REGION Network 90: VARIABLES AUXILIARES - Fin de Reset
   RUNG wire#powerrail
      Contact( #Mx_ET09 )
      wire#w1
      Coil( #EstadoVI.Fin_Reset )
   END_RUNG
   RUNG wire#powerrail
      Contact( #Mx_ET00 )
      Contact( #EstadoZona.PerReset_CBx )
      I_Contact( #pHsMx_1 )
      I_Contact( #pHsMx_2 )
      I_Contact( #pHsMx_3 )
      I_Contact( #pHsMx_4 )
   END_RUNG wire#w1
   // the same network as SCL:
   #EstadoVI.Fin_Reset := #Mx_ET09 OR (#Mx_ET00 AND #EstadoZona.PerReset_CBx AND NOT #pHsMx_1 AND NOT #pHsMx_2 AND NOT #pHsMx_3 AND NOT #pHsMx_4);
END_REGION

REGION Network 91: VARIABLES AUXILIARES - Fin de Paro Blando
   RUNG wire#powerrail
      I_Contact( #Avance_TR1 )
      I_Contact( #Avance_TR2 )
      I_Contact( #Avance_T1 )
      I_Contact( #Avance_T2 )
      I_Contact( #Avance_T3 )
      I_Contact( #Avance_T4 )
      Contact( #EstadoZona.ParoBlando_CBx )
      Coil( #EstadoVI.Fin_Paro_Blando )
   END_RUNG
   // the same network as SCL:
   #EstadoVI.Fin_Paro_Blando := NOT #Avance_TR1 AND NOT #Avance_TR2 AND NOT #Avance_T1 AND NOT #Avance_T2 AND NOT #Avance_T3 AND NOT #Avance_T4 AND #EstadoZona.ParoBlando_CBx;
END_REGION

REGION Network 92: VARIABLES AUXILIARES - Permiso de Entrada - PTF_MAnt_Mx
   RUNG wire#powerrail
      Contact( #Mx_ET20 )
      wire#w1
      Contact( #Avance_TR1 )
      Contact( #Pos_TROK )
      Contact( #Pos_TPOK )
      Contact( #EstadoZona.Marcha_CBx )
      I_Contact( #EstadoVI.Error_Mx )
      I_Contact( #Error_Tx )
      Coil( #PTF_MAnt_Mx )
   END_RUNG
   RUNG wire#powerrail
      Contact( #Mx_ET60 )
      wire#w2
      Contact( #Simultaneo_Mx )
   END_RUNG wire#w1
   RUNG wire#powerrail
      Contact( #Mx_ET61 )
   END_RUNG wire#w2
   // the same network as SCL:
   #PTF_MAnt_Mx := (#Mx_ET20 OR ((#Mx_ET60 OR #Mx_ET61) AND #Simultaneo_Mx)) AND #Avance_TR1 AND #Pos_TROK AND #Pos_TPOK AND #EstadoZona.Marcha_CBx AND NOT #EstadoVI.Error_Mx AND NOT #Error_Tx;
END_REGION

REGION Network 93: INTERLOCK FSS - Permiso de DesCarga E1 - MA_DepositOK_E1
   RUNG wire#powerrail
      Contact( #Mx_ET10 )
      wire#w1
      Contact( #Avance_T1 )
      wire#w2
      Contact( #Pos_TROK )
      Contact( #Pos_TPOK )
      Contact( #EstadoZona.Marcha_CBx )
      I_Contact( #EstadoVI.Error_Mx )
      I_Contact( #Error_Tx )
      Coil( #MA_DepositOK_E1 )
   END_RUNG
   RUNG wire#w1
      Contact( #CNT_pHsMx_E1.QD )
   END_RUNG wire#w2
   RUNG wire#powerrail
      Contact( #Mx_ET11 )
   END_RUNG wire#w2
   RUNG wire#powerrail
      Contact( #Mx_ET01 )
      I_Contact( #Selec_E3 )
      I_Contact( #pHsMx_1 )
      I_Contact( #pHsMx_2 )
      I_Contact( #pHsMx_3 )
      I_Contact( #pHsMx_4 )
      Contact( #ConfigFB.NoEntrar_E1 )
   END_RUNG wire#w2
   // the same network as SCL:
   #MA_DepositOK_E1 := ((#Mx_ET10 AND (#Avance_T1 OR #CNT_pHsMx_E1.QD)) OR #Mx_ET11 OR (#Mx_ET01 AND NOT #Selec_E3 AND NOT #pHsMx_1 AND NOT #pHsMx_2 AND NOT #pHsMx_3 AND NOT #pHsMx_4 AND #ConfigFB.NoEntrar_E1)) AND #Pos_TROK AND #Pos_TPOK AND #EstadoZona.Marcha_CBx AND NOT #EstadoVI.Error_Mx AND NOT #Error_Tx;
END_REGION

REGION Network 94: INTERLOCK FSS - Permiso de DesCarga E1 - MA_DepositOK_E3
   RUNG wire#powerrail
      Contact( #Mx_ET30 )
      wire#w1
      Contact( #Avance_T1 )
      wire#w2
      Contact( #Pos_TROK )
      Contact( #Pos_TPOK )
      Contact( #EstadoZona.Marcha_CBx )
      I_Contact( #EstadoVI.Error_Mx )
      I_Contact( #Error_Tx )
      Coil( #MA_DepositOK_E3 )
   END_RUNG
   RUNG wire#w1
      Contact( #CNT_pHsMx_E3.QD )
   END_RUNG wire#w2
   RUNG wire#powerrail
      Contact( #Mx_ET31 )
   END_RUNG wire#w2
   RUNG wire#powerrail
      Contact( #Mx_ET01 )
      I_Contact( #Selec_E1 )
      I_Contact( #pHsMx_1 )
      I_Contact( #pHsMx_2 )
      I_Contact( #pHsMx_3 )
      I_Contact( #pHsMx_4 )
      Contact( #ConfigFB.NoEntrar_E3 )
   END_RUNG wire#w2
   // the same network as SCL:
   #MA_DepositOK_E3 := ((#Mx_ET30 AND (#Avance_T1 OR #CNT_pHsMx_E3.QD)) OR #Mx_ET31 OR (#Mx_ET01 AND NOT #Selec_E1 AND NOT #pHsMx_1 AND NOT #pHsMx_2 AND NOT #pHsMx_3 AND NOT #pHsMx_4 AND #ConfigFB.NoEntrar_E3)) AND #Pos_TROK AND #Pos_TPOK AND #EstadoZona.Marcha_CBx AND NOT #EstadoVI.Error_Mx AND NOT #Error_Tx;
END_REGION

REGION Network 95: VARIABLES AUXILIARES - Aviso de Salida - AVTF_Mx_MSig - Grande y Pequeña
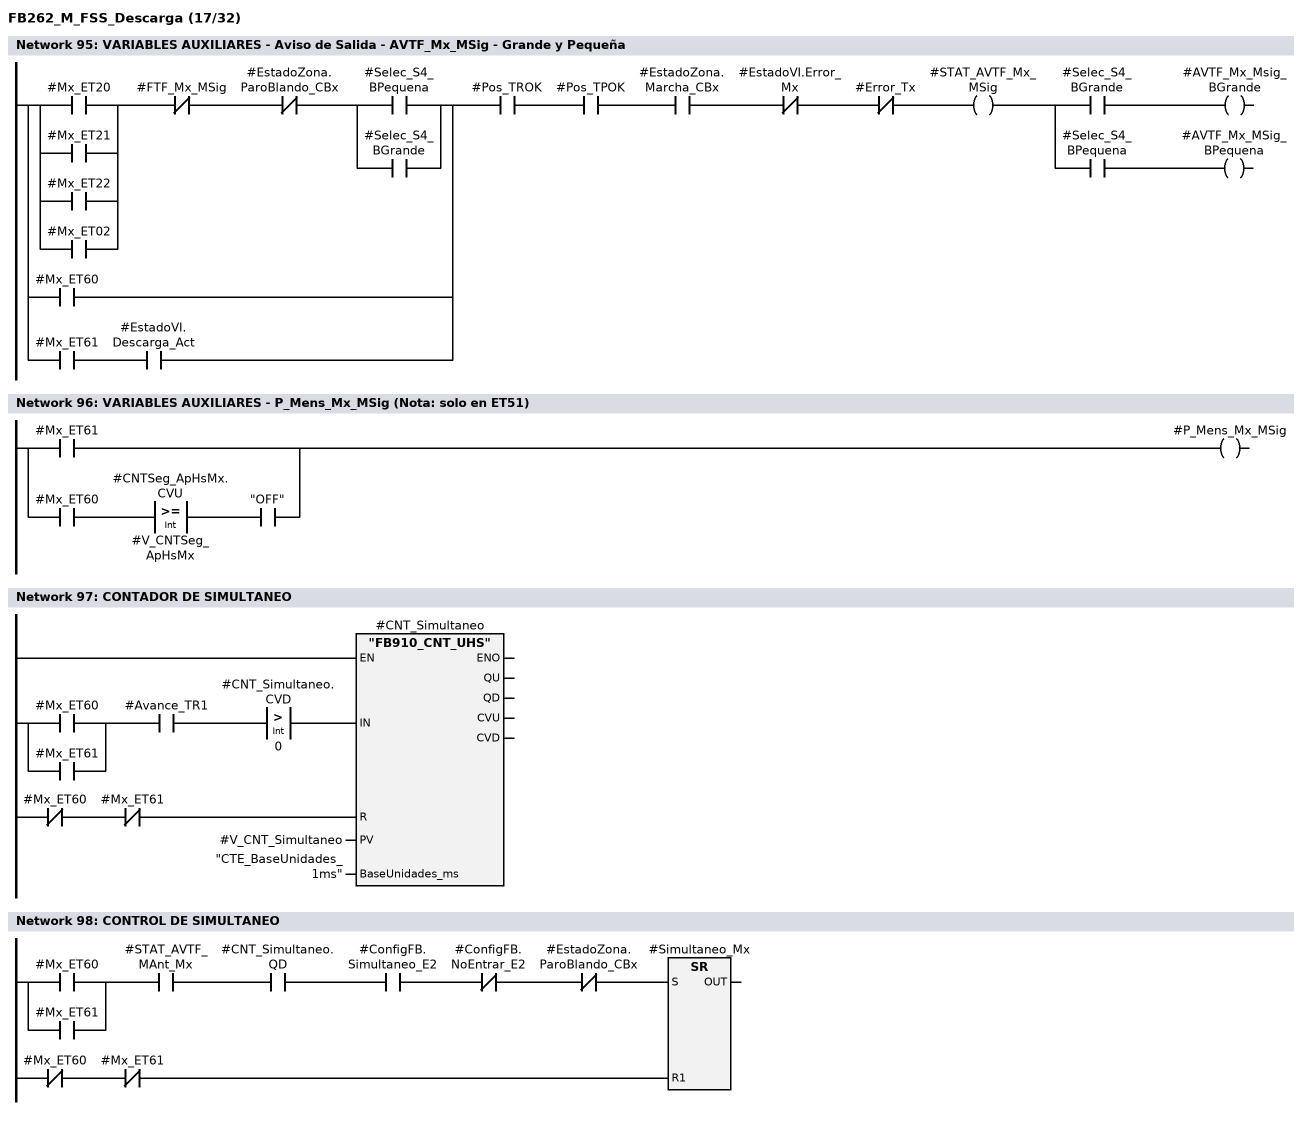
   RUNG wire#powerrail
      Contact( #Mx_ET20 )
      wire#w1
      I_Contact( #FTF_Mx_MSig )
      I_Contact( #EstadoZona.ParoBlando_CBx )
      wire#w2
      Contact( #Selec_S4_BPequena )
      wire#w3
      Contact( #Pos_TROK )
      Contact( #Pos_TPOK )
      Contact( #EstadoZona.Marcha_CBx )
      I_Contact( #EstadoVI.Error_Mx )
      I_Contact( #Error_Tx )
      Coil( #STAT_AVTF_Mx_MSig )
      wire#w4
      Contact( #Selec_S4_BGrande )
      Coil( #AVTF_Mx_Msig_BGrande )
   END_RUNG
   RUNG wire#powerrail
      Contact( #Mx_ET21 )
   END_RUNG wire#w1
   RUNG wire#powerrail
      Contact( #Mx_ET22 )
   END_RUNG wire#w1
   RUNG wire#powerrail
      Contact( #Mx_ET02 )
   END_RUNG wire#w1
   RUNG wire#w2
      Contact( #Selec_S4_BGrande )
   END_RUNG wire#w3
   RUNG wire#powerrail
      Contact( #Mx_ET60 )
   END_RUNG wire#w3
   RUNG wire#powerrail
      Contact( #Mx_ET61 )
      Contact( #EstadoVI.Descarga_Act )
   END_RUNG wire#w3
   RUNG wire#w4
      Contact( #Selec_S4_BPequena )
      Coil( #AVTF_Mx_MSig_BPequena )
   END_RUNG
   // the same network as SCL:
   #STAT_AVTF_Mx_MSig := (((#Mx_ET20 OR #Mx_ET21 OR #Mx_ET22 OR #Mx_ET02) AND NOT #FTF_Mx_MSig AND NOT #EstadoZona.ParoBlando_CBx AND (#Selec_S4_BPequena OR #Selec_S4_BGrande)) OR #Mx_ET60 OR (#Mx_ET61 AND #EstadoVI.Descarga_Act)) AND #Pos_TROK AND #Pos_TPOK AND #EstadoZona.Marcha_CBx AND NOT #EstadoVI.Error_Mx AND NOT #Error_Tx;
   #AVTF_Mx_Msig_BGrande := #STAT_AVTF_Mx_MSig AND #Selec_S4_BGrande;
   #AVTF_Mx_MSig_BPequena := #STAT_AVTF_Mx_MSig AND #Selec_S4_BPequena;
END_REGION

REGION Network 96: VARIABLES AUXILIARES - P_Mens_Mx_MSig (Nota: solo en ET51)
   RUNG wire#powerrail
      Contact( #Mx_ET61 )
      wire#w1
      Coil( #P_Mens_Mx_MSig )
   END_RUNG
   RUNG wire#powerrail
      Contact( #Mx_ET60 )
      { S7_Templates := "SrcType := Int" } GE_Contact(in1 := #CNTSeg_ApHsMx.CVU, in2 := #V_CNTSeg_ApHsMx)
      Contact( "OFF" )
   END_RUNG wire#w1
   // the same network as SCL:
   #P_Mens_Mx_MSig := #Mx_ET61 OR (#Mx_ET60 AND (#CNTSeg_ApHsMx.CVU >= #V_CNTSeg_ApHsMx) AND "OFF");
END_REGION

REGION Network 97: CONTADOR DE SIMULTANEO
   RUNG wire#powerrail
      #CNT_Simultaneo(IN := wire#w2, R := wire#w3, PV := #V_CNT_Simultaneo, BaseUnidades_ms := "CTE_BaseUnidades_1ms", QU =>, QD =>, CVU =>, CVD =>)
   END_RUNG
   RUNG wire#powerrail
      Contact( #Mx_ET60 )
      wire#w1
      Contact( #Avance_TR1 )
      { S7_Templates := "SrcType := Int" } GT_Contact(in1 := #CNT_Simultaneo.CVD, in2 := 0)
   END_RUNG wire#w2
   RUNG wire#powerrail
      Contact( #Mx_ET61 )
   END_RUNG wire#w1
   RUNG wire#powerrail
      I_Contact( #Mx_ET60 )
      I_Contact( #Mx_ET61 )
   END_RUNG wire#w3
   // the same network as SCL:
   #CNT_Simultaneo(IN := (#Mx_ET60 OR #Mx_ET61) AND #Avance_TR1 AND (#CNT_Simultaneo.CVD > 0),   // "FB910_CNT_UHS"
                   R := NOT #Mx_ET60 AND NOT #Mx_ET61,
                   PV := #V_CNT_Simultaneo,
                   BaseUnidades_ms := "CTE_BaseUnidades_1ms");
END_REGION

REGION Network 98: CONTROL DE SIMULTANEO
   RUNG wire#powerrail
      Contact( #Mx_ET60 )
      wire#w1
      Contact( #STAT_AVTF_MAnt_Mx )
      Contact( #CNT_Simultaneo.QD )
      Contact( #ConfigFB.Simultaneo_E2 )
      I_Contact( #ConfigFB.NoEntrar_E2 )
      I_Contact( #EstadoZona.ParoBlando_CBx )
      S_SR(operand := #Simultaneo_Mx, r1 := wire#w2)
   END_RUNG
   RUNG wire#powerrail
      Contact( #Mx_ET61 )
   END_RUNG wire#w1
   RUNG wire#powerrail
      I_Contact( #Mx_ET60 )
      I_Contact( #Mx_ET61 )
   END_RUNG wire#w2
   // the same network as SCL:
   IF (#Mx_ET60 OR #Mx_ET61) AND #STAT_AVTF_MAnt_Mx AND #CNT_Simultaneo.QD AND #ConfigFB.Simultaneo_E2 AND NOT #ConfigFB.NoEntrar_E2 AND NOT #EstadoZona.ParoBlando_CBx THEN
       #Simultaneo_Mx := TRUE;   // SR flip-flop
   END_IF;
   IF NOT #Mx_ET60 AND NOT #Mx_ET61 THEN #Simultaneo_Mx := FALSE; END_IF;
END_REGION

REGION Network 99: MENSAJES - PRESENCIA
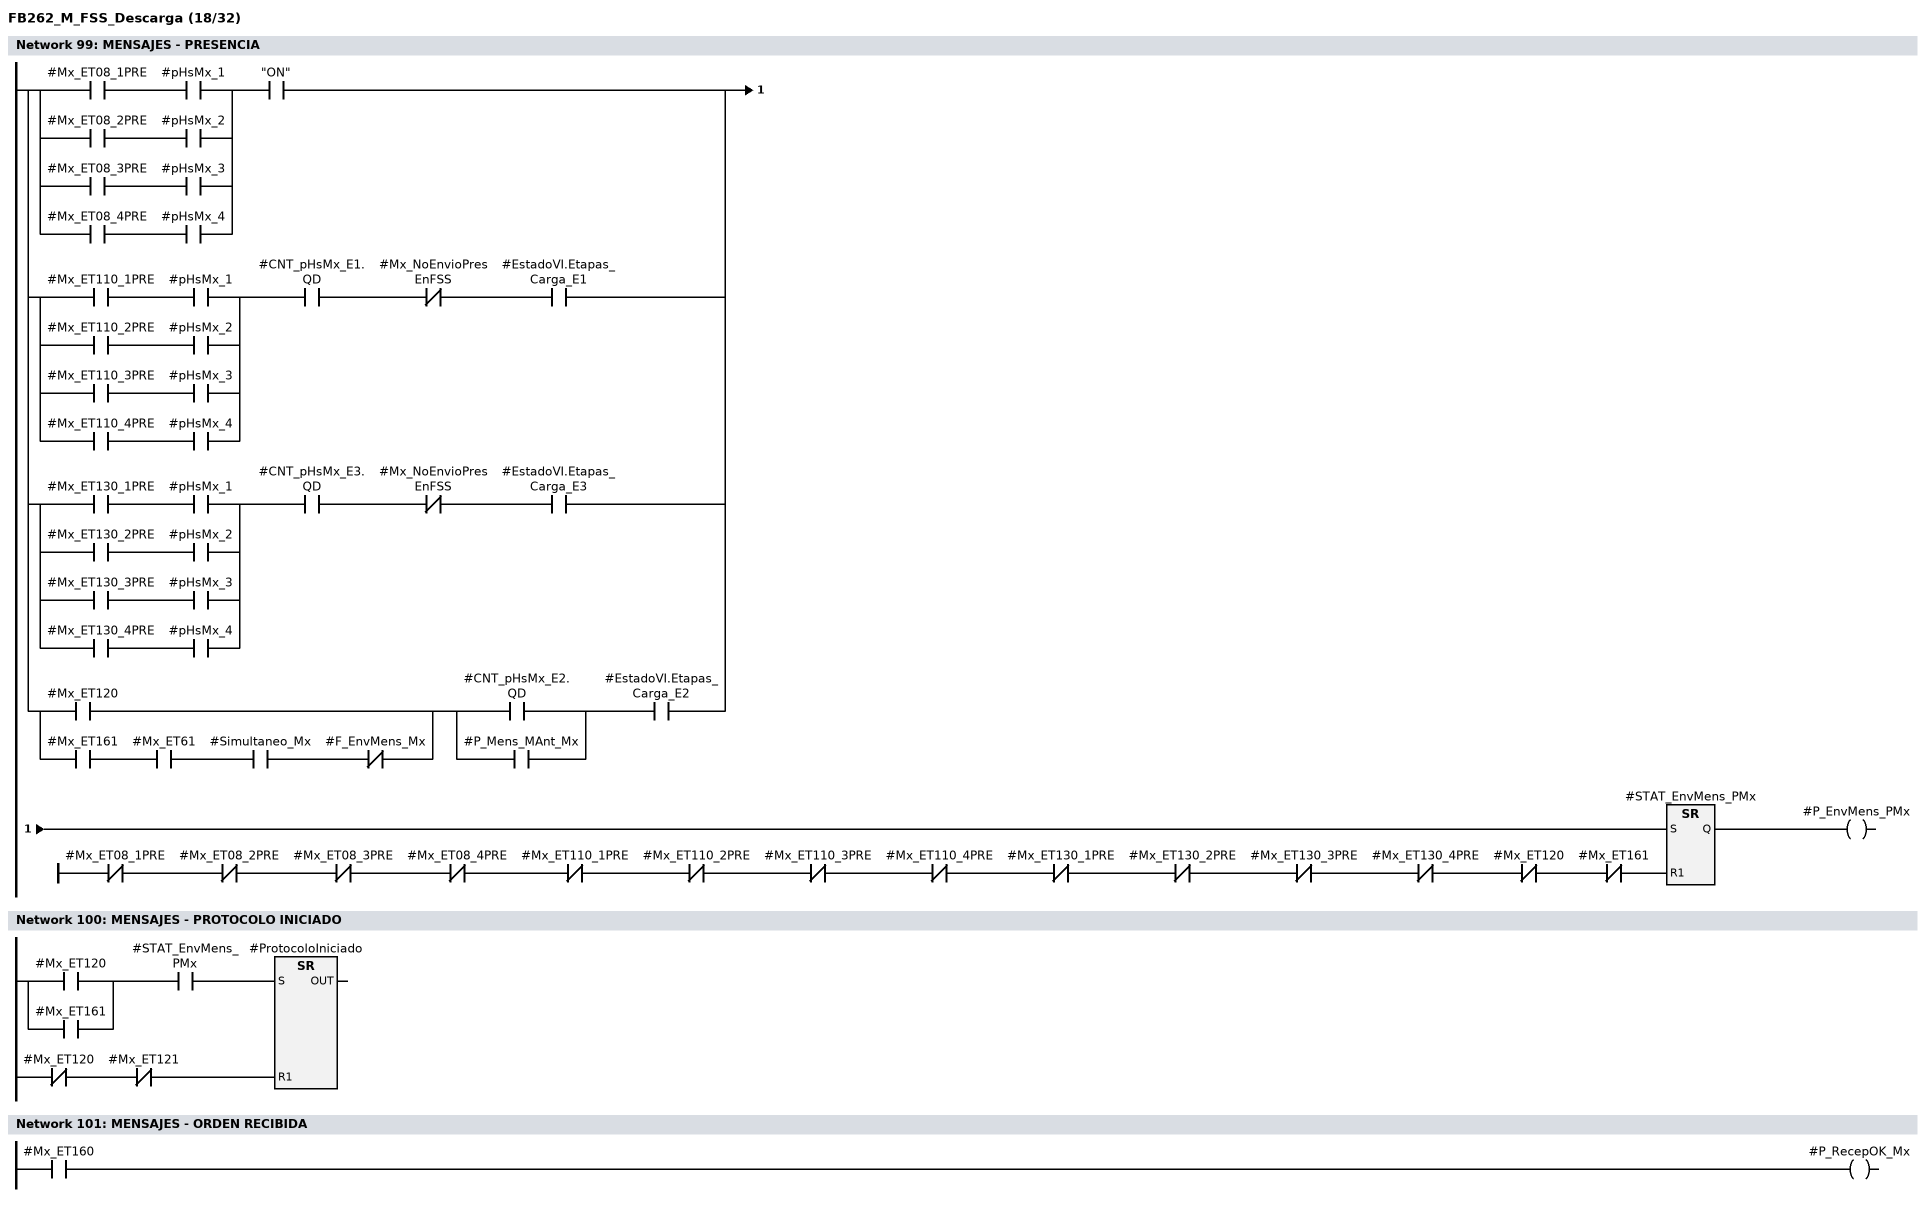
   RUNG wire#powerrail
      Contact( #Mx_ET08_1PRE )
      Contact( #pHsMx_1 )
      wire#w1
      Contact( "ON" )
      wire#w2
      S_SR(operand := #STAT_EnvMens_PMx, r1 := wire#w7)
      Coil( #P_EnvMens_PMx )
   END_RUNG
   RUNG wire#powerrail
      Contact( #Mx_ET08_2PRE )
      Contact( #pHsMx_2 )
   END_RUNG wire#w1
   RUNG wire#powerrail
      Contact( #Mx_ET08_3PRE )
      Contact( #pHsMx_3 )
   END_RUNG wire#w1
   RUNG wire#powerrail
      Contact( #Mx_ET08_4PRE )
      Contact( #pHsMx_4 )
   END_RUNG wire#w1
   RUNG wire#powerrail
      Contact( #Mx_ET110_1PRE )
      Contact( #pHsMx_1 )
      wire#w3
      Contact( #CNT_pHsMx_E1.QD )
      I_Contact( #Mx_NoEnvioPresEnFSS )
      Contact( #EstadoVI.Etapas_Carga_E1 )
   END_RUNG wire#w2
   RUNG wire#powerrail
      Contact( #Mx_ET110_2PRE )
      Contact( #pHsMx_2 )
   END_RUNG wire#w3
   RUNG wire#powerrail
      Contact( #Mx_ET110_3PRE )
      Contact( #pHsMx_3 )
   END_RUNG wire#w3
   RUNG wire#powerrail
      Contact( #Mx_ET110_4PRE )
      Contact( #pHsMx_4 )
   END_RUNG wire#w3
   RUNG wire#powerrail
      Contact( #Mx_ET130_1PRE )
      Contact( #pHsMx_1 )
      wire#w4
      Contact( #CNT_pHsMx_E3.QD )
      I_Contact( #Mx_NoEnvioPresEnFSS )
      Contact( #EstadoVI.Etapas_Carga_E3 )
   END_RUNG wire#w2
   RUNG wire#powerrail
      Contact( #Mx_ET130_2PRE )
      Contact( #pHsMx_2 )
   END_RUNG wire#w4
   RUNG wire#powerrail
      Contact( #Mx_ET130_3PRE )
      Contact( #pHsMx_3 )
   END_RUNG wire#w4
   RUNG wire#powerrail
      Contact( #Mx_ET130_4PRE )
      Contact( #pHsMx_4 )
   END_RUNG wire#w4
   RUNG wire#powerrail
      Contact( #Mx_ET120 )
      wire#w5
      Contact( #CNT_pHsMx_E2.QD )
      wire#w6
      Contact( #EstadoVI.Etapas_Carga_E2 )
   END_RUNG wire#w2
   RUNG wire#powerrail
      Contact( #Mx_ET161 )
      Contact( #Mx_ET61 )
      Contact( #Simultaneo_Mx )
      I_Contact( #F_EnvMens_Mx )
   END_RUNG wire#w5
   RUNG wire#w5
      Contact( #P_Mens_MAnt_Mx )
   END_RUNG wire#w6
   RUNG wire#powerrail
      I_Contact( #Mx_ET08_1PRE )
      I_Contact( #Mx_ET08_2PRE )
      I_Contact( #Mx_ET08_3PRE )
      I_Contact( #Mx_ET08_4PRE )
      I_Contact( #Mx_ET110_1PRE )
      I_Contact( #Mx_ET110_2PRE )
      I_Contact( #Mx_ET110_3PRE )
      I_Contact( #Mx_ET110_4PRE )
      I_Contact( #Mx_ET130_1PRE )
      I_Contact( #Mx_ET130_2PRE )
      I_Contact( #Mx_ET130_3PRE )
      I_Contact( #Mx_ET130_4PRE )
      I_Contact( #Mx_ET120 )
      I_Contact( #Mx_ET161 )
   END_RUNG wire#w7
   // the same network as SCL:
   IF (((#Mx_ET08_1PRE AND #pHsMx_1) OR (#Mx_ET08_2PRE AND #pHsMx_2) OR (#Mx_ET08_3PRE AND #pHsMx_3) OR (#Mx_ET08_4PRE AND #pHsMx_4)) AND "ON") OR (((#Mx_ET110_1PRE AND #pHsMx_1) OR (#Mx_ET110_2PRE AND #pHsMx_2) OR (#Mx_ET110_3PRE AND #pHsMx_3) OR (#Mx_ET110_4PRE AND #pHsMx_4)) AND #CNT_pHsMx_E1.QD AND NOT #Mx_NoEnvioPresEnFSS AND #EstadoVI.Etapas_Carga_E1) OR (((#Mx_ET130_1PRE AND #pHsMx_1) OR (#Mx_ET130_2PRE AND #pHsMx_2) OR (#Mx_ET130_3PRE AND #pHsMx_3) OR (#Mx_ET130_4PRE AND #pHsMx_4)) AND #CNT_pHsMx_E3.QD AND NOT #Mx_NoEnvioPresEnFSS AND #EstadoVI.Etapas_Carga_E3) OR ((#Mx_ET120 OR (#Mx_ET161 AND #Mx_ET61 AND #Simultaneo_Mx AND NOT #F_EnvMens_Mx)) AND (#CNT_pHsMx_E2.QD OR #P_Mens_MAnt_Mx) AND #EstadoVI.Etapas_Carga_E2) THEN
       #STAT_EnvMens_PMx := TRUE;   // SR flip-flop
   END_IF;
   IF NOT #Mx_ET08_1PRE AND NOT #Mx_ET08_2PRE AND NOT #Mx_ET08_3PRE AND NOT #Mx_ET08_4PRE AND NOT #Mx_ET110_1PRE AND NOT #Mx_ET110_2PRE AND NOT #Mx_ET110_3PRE AND NOT #Mx_ET110_4PRE AND NOT #Mx_ET130_1PRE AND NOT #Mx_ET130_2PRE AND NOT #Mx_ET130_3PRE AND NOT #Mx_ET130_4PRE AND NOT #Mx_ET120 AND NOT #Mx_ET161 THEN
       #STAT_EnvMens_PMx := FALSE;
   END_IF;
   #P_EnvMens_PMx := #STAT_EnvMens_PMx;
END_REGION

REGION Network 100: MENSAJES - PROTOCOLO INICIADO
   RUNG wire#powerrail
      Contact( #Mx_ET120 )
      wire#w1
      Contact( #STAT_EnvMens_PMx )
      S_SR(operand := #ProtocoloIniciado, r1 := wire#w2)
   END_RUNG
   RUNG wire#powerrail
      Contact( #Mx_ET161 )
   END_RUNG wire#w1
   RUNG wire#powerrail
      I_Contact( #Mx_ET120 )
      I_Contact( #Mx_ET121 )
   END_RUNG wire#w2
   // the same network as SCL:
   IF (#Mx_ET120 OR #Mx_ET161) AND #STAT_EnvMens_PMx THEN
       #ProtocoloIniciado := TRUE;   // SR flip-flop
   END_IF;
   IF NOT #Mx_ET120 AND NOT #Mx_ET121 THEN #ProtocoloIniciado := FALSE; END_IF;
END_REGION

REGION Network 101: MENSAJES - ORDEN RECIBIDA
   RUNG wire#powerrail
      Contact( #Mx_ET160 )
      Coil( #P_RecepOK_Mx )
   END_RUNG
   // the same network as SCL:
   #P_RecepOK_Mx := #Mx_ET160;
END_REGION

REGION Network 102: VARIABLES INTERNAS - AVANCE DE CARGA >> DESDE FSS
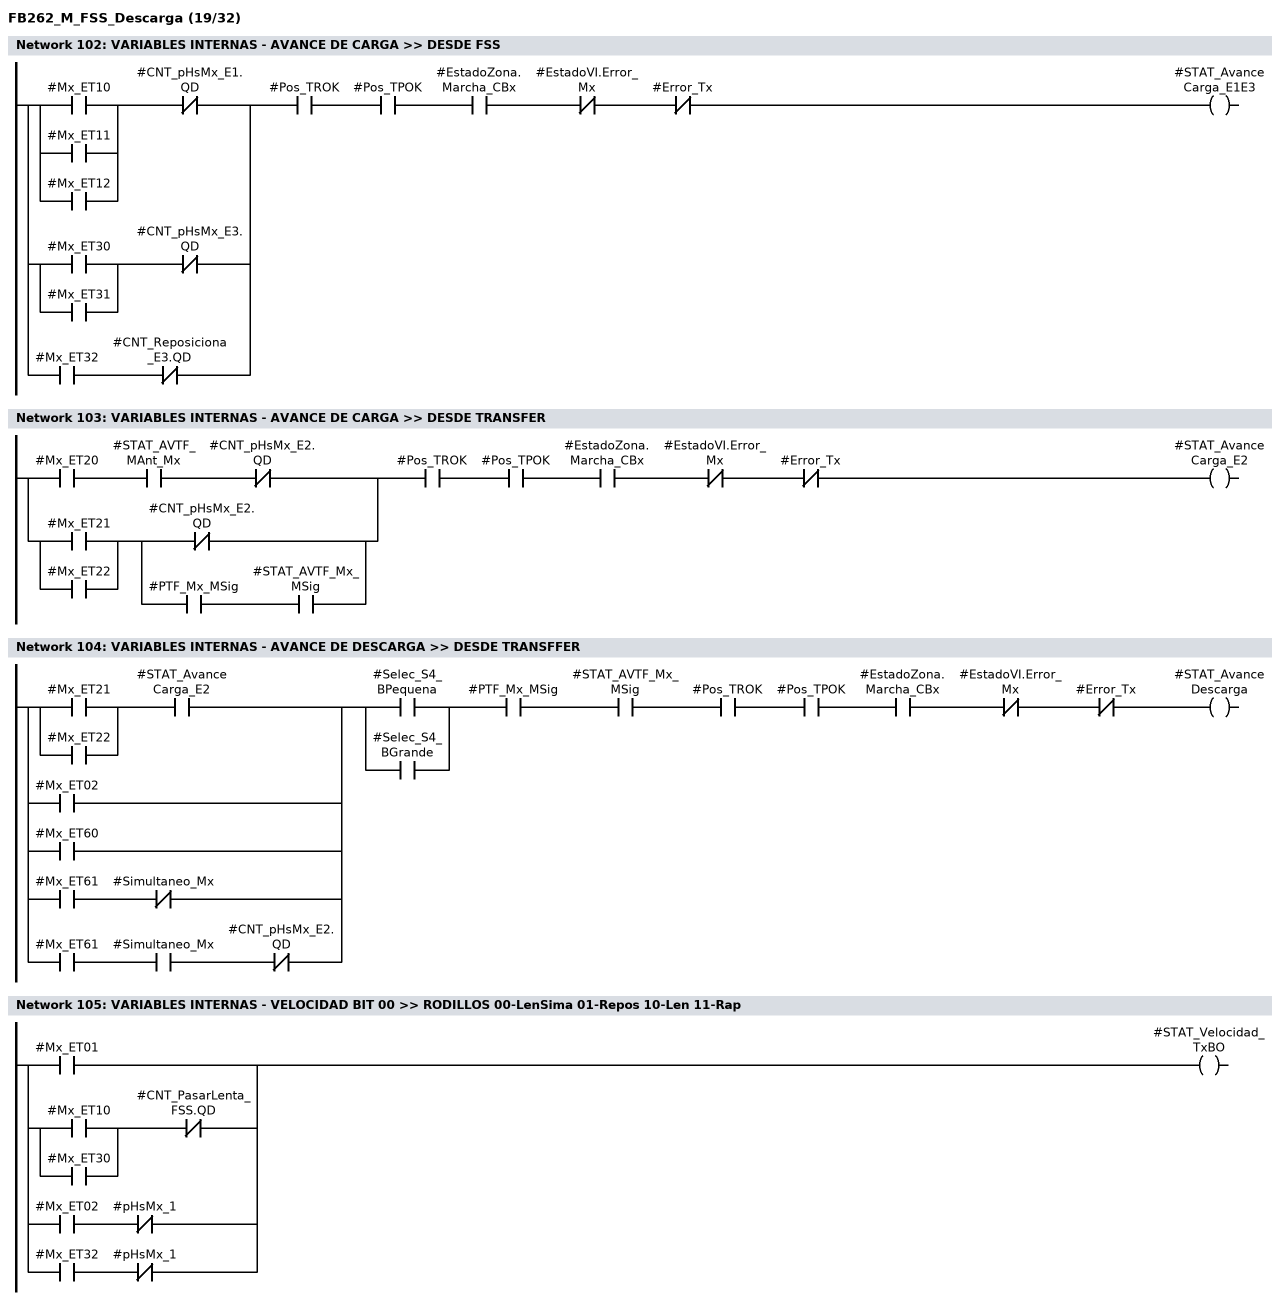
   RUNG wire#powerrail
      Contact( #Mx_ET10 )
      wire#w1
      I_Contact( #CNT_pHsMx_E1.QD )
      wire#w2
      Contact( #Pos_TROK )
      Contact( #Pos_TPOK )
      Contact( #EstadoZona.Marcha_CBx )
      I_Contact( #EstadoVI.Error_Mx )
      I_Contact( #Error_Tx )
      Coil( #STAT_AvanceCarga_E1E3 )
   END_RUNG
   RUNG wire#powerrail
      Contact( #Mx_ET11 )
   END_RUNG wire#w1
   RUNG wire#powerrail
      Contact( #Mx_ET12 )
   END_RUNG wire#w1
   RUNG wire#powerrail
      Contact( #Mx_ET30 )
      wire#w3
      I_Contact( #CNT_pHsMx_E3.QD )
   END_RUNG wire#w2
   RUNG wire#powerrail
      Contact( #Mx_ET31 )
   END_RUNG wire#w3
   RUNG wire#powerrail
      Contact( #Mx_ET32 )
      I_Contact( #CNT_Reposiciona_E3.QD )
   END_RUNG wire#w2
   // the same network as SCL:
   #STAT_AvanceCarga_E1E3 := (((#Mx_ET10 OR #Mx_ET11 OR #Mx_ET12) AND NOT #CNT_pHsMx_E1.QD) OR ((#Mx_ET30 OR #Mx_ET31) AND NOT #CNT_pHsMx_E3.QD) OR (#Mx_ET32 AND NOT #CNT_Reposiciona_E3.QD)) AND #Pos_TROK AND #Pos_TPOK AND #EstadoZona.Marcha_CBx AND NOT #EstadoVI.Error_Mx AND NOT #Error_Tx;
END_REGION

REGION Network 103: VARIABLES INTERNAS - AVANCE DE CARGA >> DESDE TRANSFER
   RUNG wire#powerrail
      Contact( #Mx_ET20 )
      Contact( #STAT_AVTF_MAnt_Mx )
      I_Contact( #CNT_pHsMx_E2.QD )
      wire#w1
      Contact( #Pos_TROK )
      Contact( #Pos_TPOK )
      Contact( #EstadoZona.Marcha_CBx )
      I_Contact( #EstadoVI.Error_Mx )
      I_Contact( #Error_Tx )
      Coil( #STAT_AvanceCarga_E2 )
   END_RUNG
   RUNG wire#powerrail
      Contact( #Mx_ET21 )
      wire#w2
      I_Contact( #CNT_pHsMx_E2.QD )
   END_RUNG wire#w1
   RUNG wire#powerrail
      Contact( #Mx_ET22 )
   END_RUNG wire#w2
   RUNG wire#w2
      Contact( #PTF_Mx_MSig )
      Contact( #STAT_AVTF_Mx_MSig )
   END_RUNG wire#w1
   // the same network as SCL:
   #STAT_AvanceCarga_E2 := ((#Mx_ET20 AND #STAT_AVTF_MAnt_Mx AND NOT #CNT_pHsMx_E2.QD) OR ((#Mx_ET21 OR #Mx_ET22) AND (NOT #CNT_pHsMx_E2.QD OR (#PTF_Mx_MSig AND #STAT_AVTF_Mx_MSig)))) AND #Pos_TROK AND #Pos_TPOK AND #EstadoZona.Marcha_CBx AND NOT #EstadoVI.Error_Mx AND NOT #Error_Tx;
END_REGION

REGION Network 104: VARIABLES INTERNAS - AVANCE DE DESCARGA >> DESDE TRANSFFER
   RUNG wire#powerrail
      Contact( #Mx_ET21 )
      wire#w1
      Contact( #STAT_AvanceCarga_E2 )
      wire#w2
      Contact( #Selec_S4_BPequena )
      wire#w3
      Contact( #PTF_Mx_MSig )
      Contact( #STAT_AVTF_Mx_MSig )
      Contact( #Pos_TROK )
      Contact( #Pos_TPOK )
      Contact( #EstadoZona.Marcha_CBx )
      I_Contact( #EstadoVI.Error_Mx )
      I_Contact( #Error_Tx )
      Coil( #STAT_AvanceDescarga )
   END_RUNG
   RUNG wire#powerrail
      Contact( #Mx_ET22 )
   END_RUNG wire#w1
   RUNG wire#powerrail
      Contact( #Mx_ET02 )
   END_RUNG wire#w2
   RUNG wire#powerrail
      Contact( #Mx_ET60 )
   END_RUNG wire#w2
   RUNG wire#powerrail
      Contact( #Mx_ET61 )
      I_Contact( #Simultaneo_Mx )
   END_RUNG wire#w2
   RUNG wire#powerrail
      Contact( #Mx_ET61 )
      Contact( #Simultaneo_Mx )
      I_Contact( #CNT_pHsMx_E2.QD )
   END_RUNG wire#w2
   RUNG wire#w2
      Contact( #Selec_S4_BGrande )
   END_RUNG wire#w3
   // the same network as SCL:
   #STAT_AvanceDescarga := (((#Mx_ET21 OR #Mx_ET22) AND #STAT_AvanceCarga_E2) OR #Mx_ET02 OR #Mx_ET60 OR (#Mx_ET61 AND NOT #Simultaneo_Mx) OR (#Mx_ET61 AND #Simultaneo_Mx AND NOT #CNT_pHsMx_E2.QD)) AND (#Selec_S4_BPequena OR #Selec_S4_BGrande) AND #PTF_Mx_MSig AND #STAT_AVTF_Mx_MSig AND #Pos_TROK AND #Pos_TPOK AND #EstadoZona.Marcha_CBx AND NOT #EstadoVI.Error_Mx AND NOT #Error_Tx;
END_REGION

REGION Network 105: VARIABLES INTERNAS - VELOCIDAD BIT 00 >> RODILLOS 00-LenSima 01-Repos 10-Len 11-Rap
   RUNG wire#powerrail
      Contact( #Mx_ET01 )
      wire#w1
      Coil( #STAT_Velocidad_TxBO )
   END_RUNG
   RUNG wire#powerrail
      Contact( #Mx_ET10 )
      wire#w2
      I_Contact( #CNT_PasarLenta_FSS.QD )
   END_RUNG wire#w1
   RUNG wire#powerrail
      Contact( #Mx_ET30 )
   END_RUNG wire#w2
   RUNG wire#powerrail
      Contact( #Mx_ET02 )
      I_Contact( #pHsMx_1 )
   END_RUNG wire#w1
   RUNG wire#powerrail
      Contact( #Mx_ET32 )
      I_Contact( #pHsMx_1 )
   END_RUNG wire#w1
   // the same network as SCL:
   #STAT_Velocidad_TxBO := #Mx_ET01 OR ((#Mx_ET10 OR #Mx_ET30) AND NOT #CNT_PasarLenta_FSS.QD) OR (#Mx_ET02 AND NOT #pHsMx_1) OR (#Mx_ET32 AND NOT #pHsMx_1);
END_REGION

REGION Network 106: VARIABLES INTERNAS - VELOCIDAD BIT 01 >> RODILLOS 00-LenSima 01-Repos 10-Len 11-Rap
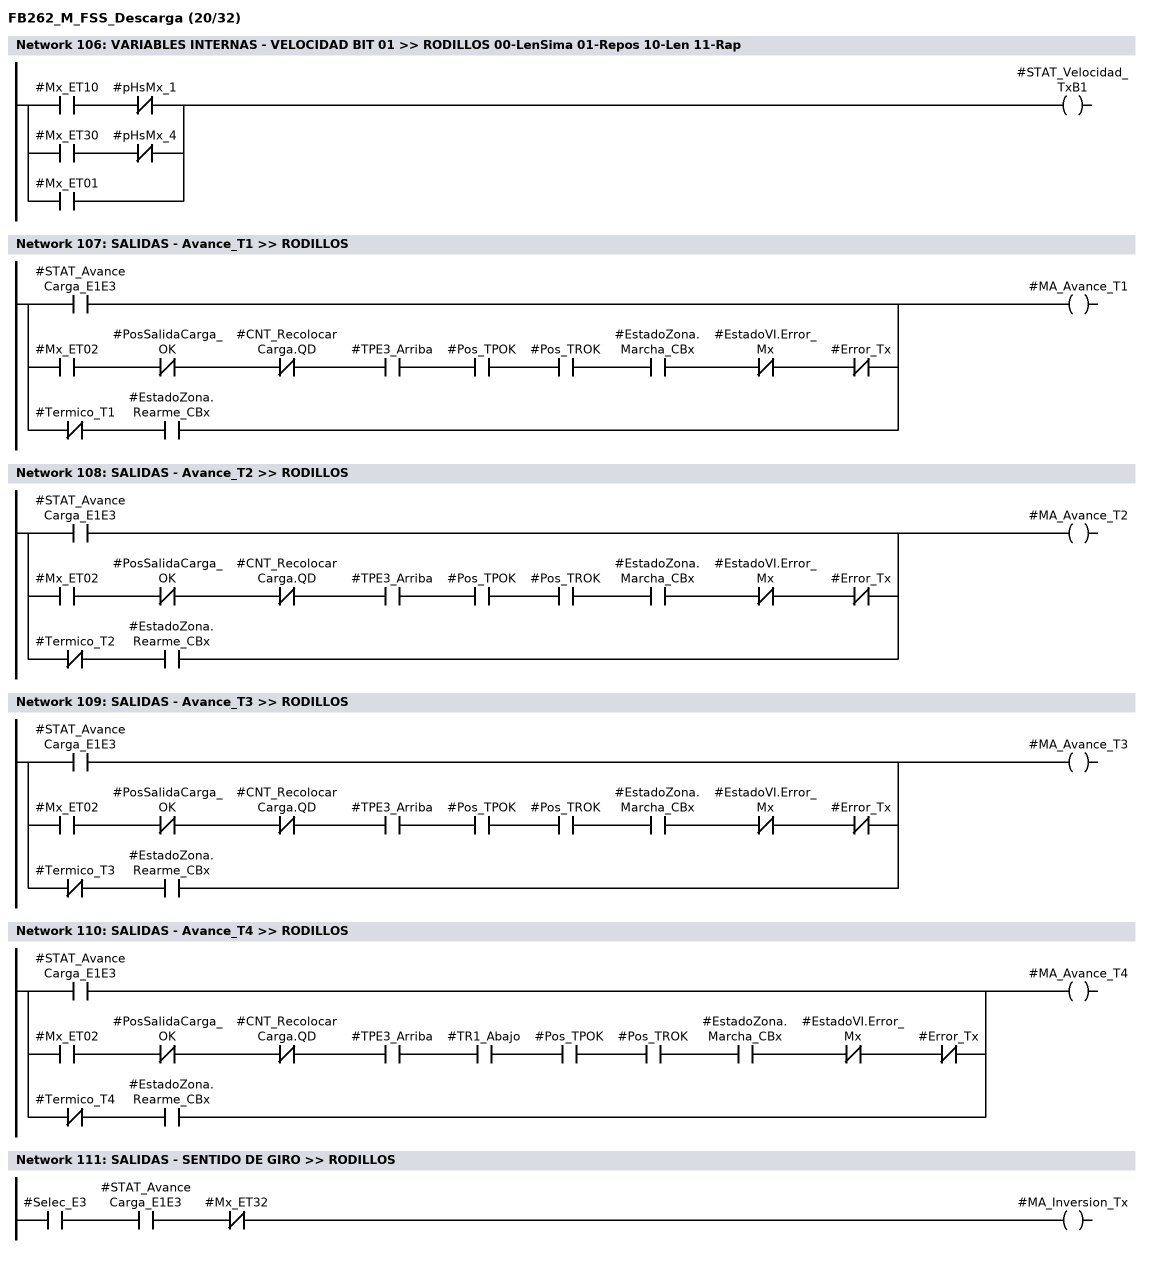
   RUNG wire#powerrail
      Contact( #Mx_ET10 )
      I_Contact( #pHsMx_1 )
      wire#w1
      Coil( #STAT_Velocidad_TxB1 )
   END_RUNG
   RUNG wire#powerrail
      Contact( #Mx_ET30 )
      I_Contact( #pHsMx_4 )
   END_RUNG wire#w1
   RUNG wire#powerrail
      Contact( #Mx_ET01 )
   END_RUNG wire#w1
   // the same network as SCL:
   #STAT_Velocidad_TxB1 := (#Mx_ET10 AND NOT #pHsMx_1) OR (#Mx_ET30 AND NOT #pHsMx_4) OR #Mx_ET01;
END_REGION

REGION Network 107: SALIDAS - Avance_T1 >> RODILLOS
   RUNG wire#powerrail
      Contact( #STAT_AvanceCarga_E1E3 )
      wire#w1
      Coil( #MA_Avance_T1 )
   END_RUNG
   RUNG wire#powerrail
      Contact( #Mx_ET02 )
      I_Contact( #PosSalidaCarga_OK )
      I_Contact( #CNT_RecolocarCarga.QD )
      Contact( #TPE3_Arriba )
      Contact( #Pos_TPOK )
      Contact( #Pos_TROK )
      Contact( #EstadoZona.Marcha_CBx )
      I_Contact( #EstadoVI.Error_Mx )
      I_Contact( #Error_Tx )
   END_RUNG wire#w1
   RUNG wire#powerrail
      I_Contact( #Termico_T1 )
      Contact( #EstadoZona.Rearme_CBx )
   END_RUNG wire#w1
   // the same network as SCL:
   #MA_Avance_T1 := #STAT_AvanceCarga_E1E3 OR (#Mx_ET02 AND NOT #PosSalidaCarga_OK AND NOT #CNT_RecolocarCarga.QD AND #TPE3_Arriba AND #Pos_TPOK AND #Pos_TROK AND #EstadoZona.Marcha_CBx AND NOT #EstadoVI.Error_Mx AND NOT #Error_Tx) OR (NOT #Termico_T1 AND #EstadoZona.Rearme_CBx);
END_REGION

REGION Network 108: SALIDAS - Avance_T2 >> RODILLOS
   RUNG wire#powerrail
      Contact( #STAT_AvanceCarga_E1E3 )
      wire#w1
      Coil( #MA_Avance_T2 )
   END_RUNG
   RUNG wire#powerrail
      Contact( #Mx_ET02 )
      I_Contact( #PosSalidaCarga_OK )
      I_Contact( #CNT_RecolocarCarga.QD )
      Contact( #TPE3_Arriba )
      Contact( #Pos_TPOK )
      Contact( #Pos_TROK )
      Contact( #EstadoZona.Marcha_CBx )
      I_Contact( #EstadoVI.Error_Mx )
      I_Contact( #Error_Tx )
   END_RUNG wire#w1
   RUNG wire#powerrail
      I_Contact( #Termico_T2 )
      Contact( #EstadoZona.Rearme_CBx )
   END_RUNG wire#w1
   // the same network as SCL:
   #MA_Avance_T2 := #STAT_AvanceCarga_E1E3 OR (#Mx_ET02 AND NOT #PosSalidaCarga_OK AND NOT #CNT_RecolocarCarga.QD AND #TPE3_Arriba AND #Pos_TPOK AND #Pos_TROK AND #EstadoZona.Marcha_CBx AND NOT #EstadoVI.Error_Mx AND NOT #Error_Tx) OR (NOT #Termico_T2 AND #EstadoZona.Rearme_CBx);
END_REGION

REGION Network 109: SALIDAS - Avance_T3 >> RODILLOS
   RUNG wire#powerrail
      Contact( #STAT_AvanceCarga_E1E3 )
      wire#w1
      Coil( #MA_Avance_T3 )
   END_RUNG
   RUNG wire#powerrail
      Contact( #Mx_ET02 )
      I_Contact( #PosSalidaCarga_OK )
      I_Contact( #CNT_RecolocarCarga.QD )
      Contact( #TPE3_Arriba )
      Contact( #Pos_TPOK )
      Contact( #Pos_TROK )
      Contact( #EstadoZona.Marcha_CBx )
      I_Contact( #EstadoVI.Error_Mx )
      I_Contact( #Error_Tx )
   END_RUNG wire#w1
   RUNG wire#powerrail
      I_Contact( #Termico_T3 )
      Contact( #EstadoZona.Rearme_CBx )
   END_RUNG wire#w1
   // the same network as SCL:
   #MA_Avance_T3 := #STAT_AvanceCarga_E1E3 OR (#Mx_ET02 AND NOT #PosSalidaCarga_OK AND NOT #CNT_RecolocarCarga.QD AND #TPE3_Arriba AND #Pos_TPOK AND #Pos_TROK AND #EstadoZona.Marcha_CBx AND NOT #EstadoVI.Error_Mx AND NOT #Error_Tx) OR (NOT #Termico_T3 AND #EstadoZona.Rearme_CBx);
END_REGION

REGION Network 110: SALIDAS - Avance_T4 >> RODILLOS
   RUNG wire#powerrail
      Contact( #STAT_AvanceCarga_E1E3 )
      wire#w1
      Coil( #MA_Avance_T4 )
   END_RUNG
   RUNG wire#powerrail
      Contact( #Mx_ET02 )
      I_Contact( #PosSalidaCarga_OK )
      I_Contact( #CNT_RecolocarCarga.QD )
      Contact( #TPE3_Arriba )
      Contact( #TR1_Abajo )
      Contact( #Pos_TPOK )
      Contact( #Pos_TROK )
      Contact( #EstadoZona.Marcha_CBx )
      I_Contact( #EstadoVI.Error_Mx )
      I_Contact( #Error_Tx )
   END_RUNG wire#w1
   RUNG wire#powerrail
      I_Contact( #Termico_T4 )
      Contact( #EstadoZona.Rearme_CBx )
   END_RUNG wire#w1
   // the same network as SCL:
   #MA_Avance_T4 := #STAT_AvanceCarga_E1E3 OR (#Mx_ET02 AND NOT #PosSalidaCarga_OK AND NOT #CNT_RecolocarCarga.QD AND #TPE3_Arriba AND #TR1_Abajo AND #Pos_TPOK AND #Pos_TROK AND #EstadoZona.Marcha_CBx AND NOT #EstadoVI.Error_Mx AND NOT #Error_Tx) OR (NOT #Termico_T4 AND #EstadoZona.Rearme_CBx);
END_REGION

REGION Network 111: SALIDAS - SENTIDO DE GIRO >> RODILLOS
   RUNG wire#powerrail
      Contact( #Selec_E3 )
      Contact( #STAT_AvanceCarga_E1E3 )
      I_Contact( #Mx_ET32 )
      Coil( #MA_Inversion_Tx )
   END_RUNG
   // the same network as SCL:
   #MA_Inversion_Tx := #Selec_E3 AND #STAT_AvanceCarga_E1E3 AND NOT #Mx_ET32;
END_REGION

REGION Network 112: SALIDAS - VELOCIDAD ANALOGICA >> RODILLOS
   // 25T229A_03 
   // Plantilla_Avance_E1S3_SinVariador_1Mesas.
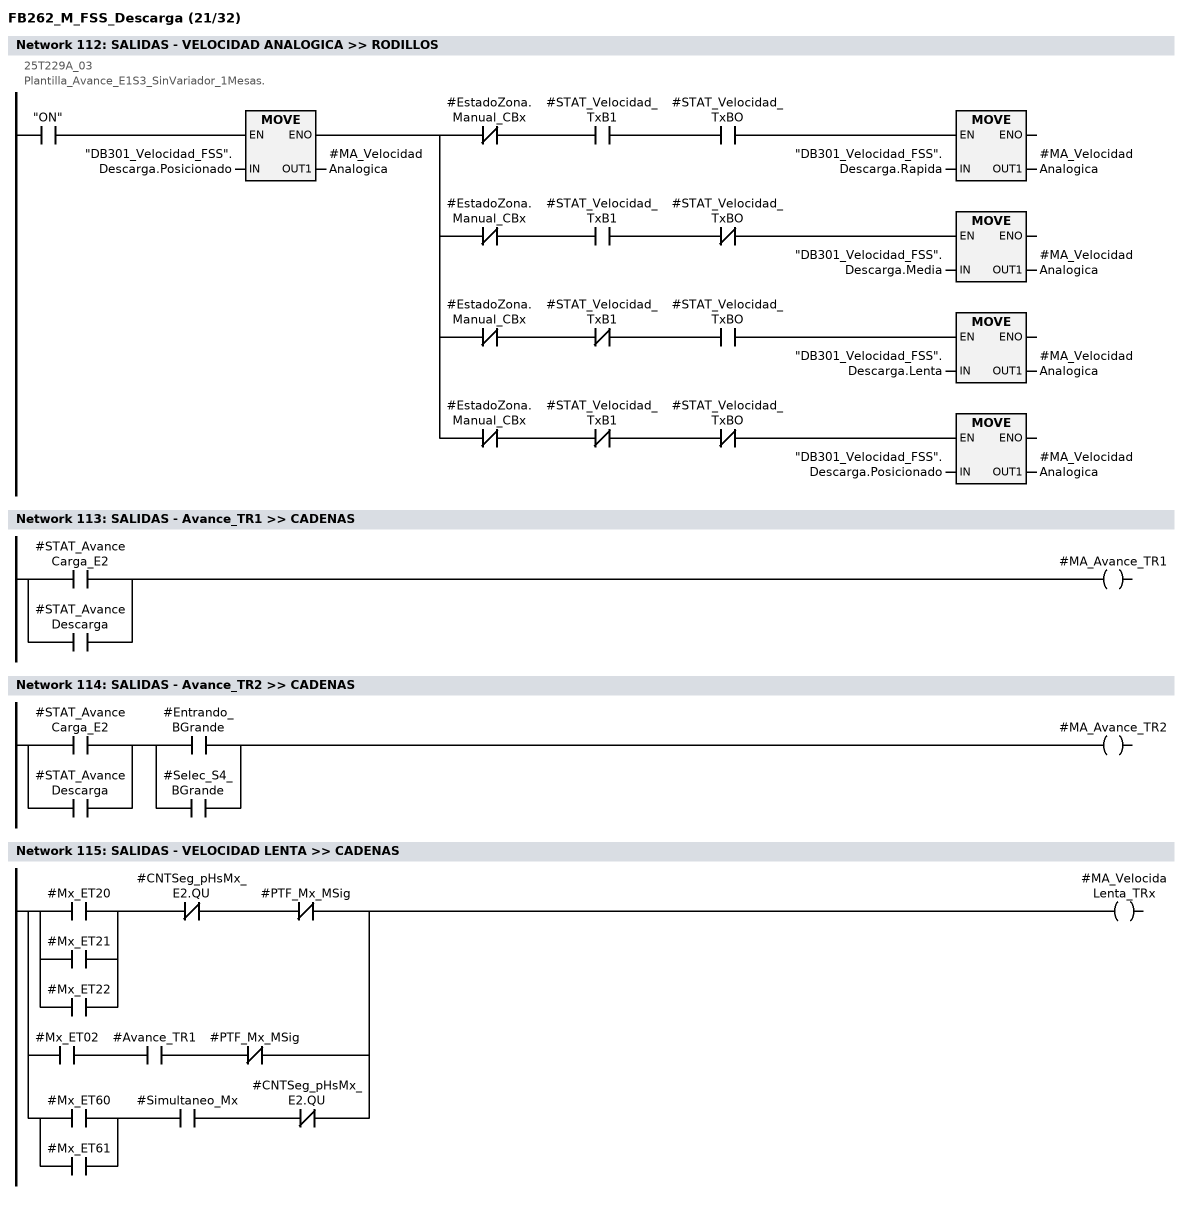
   RUNG wire#powerrail
      Contact( "ON" )
      { S7_GenerateENO := "TRUE" } Move(in := "DB301_Velocidad_FSS".Descarga.Posicionado, out1 => #MA_VelocidadAnalogica)
      wire#w1
      I_Contact( #EstadoZona.Manual_CBx )
      Contact( #STAT_Velocidad_TxB1 )
      Contact( #STAT_Velocidad_TxBO )
      { S7_GenerateENO := "TRUE" } Move(in := "DB301_Velocidad_FSS".Descarga.Rapida, out1 => #MA_VelocidadAnalogica)
   END_RUNG
   RUNG wire#w1
      I_Contact( #EstadoZona.Manual_CBx )
      Contact( #STAT_Velocidad_TxB1 )
      I_Contact( #STAT_Velocidad_TxBO )
      { S7_GenerateENO := "TRUE" } Move(in := "DB301_Velocidad_FSS".Descarga.Media, out1 => #MA_VelocidadAnalogica)
   END_RUNG
   RUNG wire#w1
      I_Contact( #EstadoZona.Manual_CBx )
      I_Contact( #STAT_Velocidad_TxB1 )
      Contact( #STAT_Velocidad_TxBO )
      { S7_GenerateENO := "TRUE" } Move(in := "DB301_Velocidad_FSS".Descarga.Lenta, out1 => #MA_VelocidadAnalogica)
   END_RUNG
   RUNG wire#w1
      I_Contact( #EstadoZona.Manual_CBx )
      I_Contact( #STAT_Velocidad_TxB1 )
      I_Contact( #STAT_Velocidad_TxBO )
      { S7_GenerateENO := "TRUE" } Move(in := "DB301_Velocidad_FSS".Descarga.Posicionado, out1 => #MA_VelocidadAnalogica)
   END_RUNG
   // the same network as SCL:
   // ENO of a box is taken as its EN; it also drops when the box reports an error
   IF "ON" THEN #MA_VelocidadAnalogica := "DB301_Velocidad_FSS".Descarga.Posicionado; END_IF;
   IF "ON" AND NOT #EstadoZona.Manual_CBx AND #STAT_Velocidad_TxB1 AND #STAT_Velocidad_TxBO THEN
       #MA_VelocidadAnalogica := "DB301_Velocidad_FSS".Descarga.Rapida;
   END_IF;
   IF "ON" AND NOT #EstadoZona.Manual_CBx AND #STAT_Velocidad_TxB1 AND NOT #STAT_Velocidad_TxBO THEN
       #MA_VelocidadAnalogica := "DB301_Velocidad_FSS".Descarga.Media;
   END_IF;
   IF "ON" AND NOT #EstadoZona.Manual_CBx AND NOT #STAT_Velocidad_TxB1 AND #STAT_Velocidad_TxBO THEN
       #MA_VelocidadAnalogica := "DB301_Velocidad_FSS".Descarga.Lenta;
   END_IF;
   IF "ON" AND NOT #EstadoZona.Manual_CBx AND NOT #STAT_Velocidad_TxB1 AND NOT #STAT_Velocidad_TxBO THEN
       #MA_VelocidadAnalogica := "DB301_Velocidad_FSS".Descarga.Posicionado;
   END_IF;
END_REGION

REGION Network 113: SALIDAS - Avance_TR1 >> CADENAS
   RUNG wire#powerrail
      Contact( #STAT_AvanceCarga_E2 )
      wire#w1
      Coil( #MA_Avance_TR1 )
   END_RUNG
   RUNG wire#powerrail
      Contact( #STAT_AvanceDescarga )
   END_RUNG wire#w1
   // the same network as SCL:
   #MA_Avance_TR1 := #STAT_AvanceCarga_E2 OR #STAT_AvanceDescarga;
END_REGION

REGION Network 114: SALIDAS - Avance_TR2 >> CADENAS
   RUNG wire#powerrail
      Contact( #STAT_AvanceCarga_E2 )
      wire#w1
      Contact( #Entrando_BGrande )
      wire#w2
      Coil( #MA_Avance_TR2 )
   END_RUNG
   RUNG wire#powerrail
      Contact( #STAT_AvanceDescarga )
   END_RUNG wire#w1
   RUNG wire#w1
      Contact( #Selec_S4_BGrande )
   END_RUNG wire#w2
   // the same network as SCL:
   #MA_Avance_TR2 := (#STAT_AvanceCarga_E2 OR #STAT_AvanceDescarga) AND (#Entrando_BGrande OR #Selec_S4_BGrande);
END_REGION

REGION Network 115: SALIDAS - VELOCIDAD LENTA >> CADENAS
   RUNG wire#powerrail
      Contact( #Mx_ET20 )
      wire#w1
      I_Contact( #CNTSeg_pHsMx_E2.QU )
      I_Contact( #PTF_Mx_MSig )
      wire#w2
      Coil( #MA_VelocidaLenta_TRx )
   END_RUNG
   RUNG wire#powerrail
      Contact( #Mx_ET21 )
   END_RUNG wire#w1
   RUNG wire#powerrail
      Contact( #Mx_ET22 )
   END_RUNG wire#w1
   RUNG wire#powerrail
      Contact( #Mx_ET02 )
      Contact( #Avance_TR1 )
      I_Contact( #PTF_Mx_MSig )
   END_RUNG wire#w2
   RUNG wire#powerrail
      Contact( #Mx_ET60 )
      wire#w3
      Contact( #Simultaneo_Mx )
      I_Contact( #CNTSeg_pHsMx_E2.QU )
   END_RUNG wire#w2
   RUNG wire#powerrail
      Contact( #Mx_ET61 )
   END_RUNG wire#w3
   // the same network as SCL:
   #MA_VelocidaLenta_TRx := ((#Mx_ET20 OR #Mx_ET21 OR #Mx_ET22) AND NOT #CNTSeg_pHsMx_E2.QU AND NOT #PTF_Mx_MSig) OR (#Mx_ET02 AND #Avance_TR1 AND NOT #PTF_Mx_MSig) OR ((#Mx_ET60 OR #Mx_ET61) AND #Simultaneo_Mx AND NOT #CNTSeg_pHsMx_E2.QU);
END_REGION

REGION Network 116: SALIDAS - SUBIR TRANSTER TR1 (Neumatica)
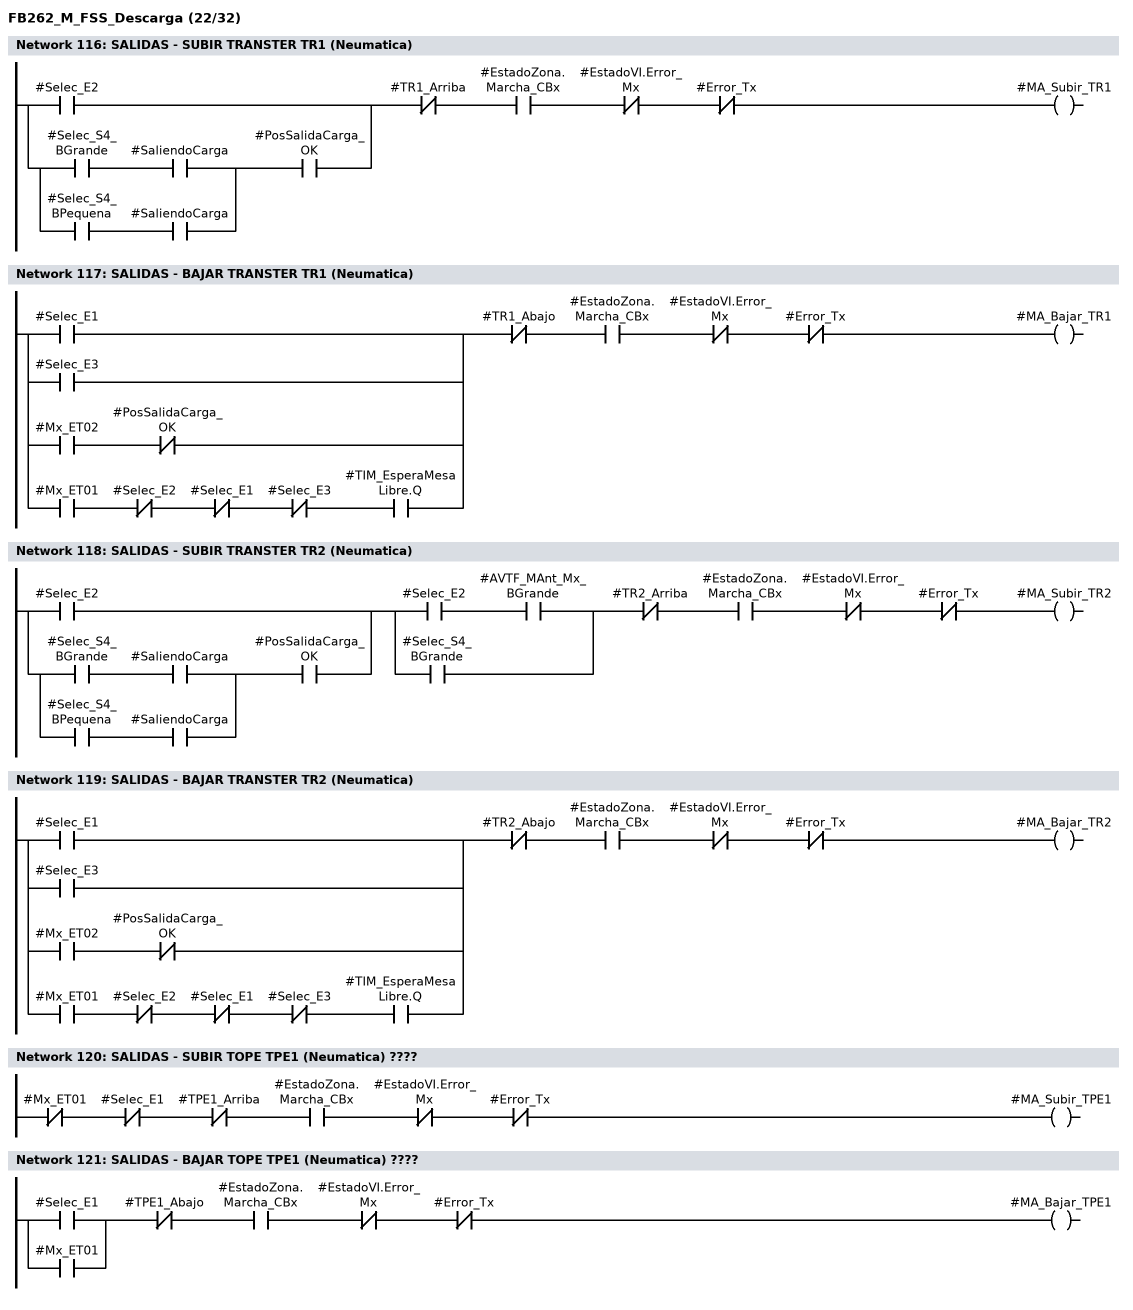
   RUNG wire#powerrail
      Contact( #Selec_E2 )
      wire#w1
      I_Contact( #TR1_Arriba )
      Contact( #EstadoZona.Marcha_CBx )
      I_Contact( #EstadoVI.Error_Mx )
      I_Contact( #Error_Tx )
      Coil( #MA_Subir_TR1 )
   END_RUNG
   RUNG wire#powerrail
      Contact( #Selec_S4_BGrande )
      Contact( #SaliendoCarga )
      wire#w2
      Contact( #PosSalidaCarga_OK )
   END_RUNG wire#w1
   RUNG wire#powerrail
      Contact( #Selec_S4_BPequena )
      Contact( #SaliendoCarga )
   END_RUNG wire#w2
   // the same network as SCL:
   #MA_Subir_TR1 := (#Selec_E2 OR (((#Selec_S4_BGrande AND #SaliendoCarga) OR (#Selec_S4_BPequena AND #SaliendoCarga)) AND #PosSalidaCarga_OK)) AND NOT #TR1_Arriba AND #EstadoZona.Marcha_CBx AND NOT #EstadoVI.Error_Mx AND NOT #Error_Tx;
END_REGION

REGION Network 117: SALIDAS - BAJAR TRANSTER TR1 (Neumatica)
   RUNG wire#powerrail
      Contact( #Selec_E1 )
      wire#w1
      I_Contact( #TR1_Abajo )
      Contact( #EstadoZona.Marcha_CBx )
      I_Contact( #EstadoVI.Error_Mx )
      I_Contact( #Error_Tx )
      Coil( #MA_Bajar_TR1 )
   END_RUNG
   RUNG wire#powerrail
      Contact( #Selec_E3 )
   END_RUNG wire#w1
   RUNG wire#powerrail
      Contact( #Mx_ET02 )
      I_Contact( #PosSalidaCarga_OK )
   END_RUNG wire#w1
   RUNG wire#powerrail
      Contact( #Mx_ET01 )
      I_Contact( #Selec_E2 )
      I_Contact( #Selec_E1 )
      I_Contact( #Selec_E3 )
      Contact( #TIM_EsperaMesaLibre.Q )
   END_RUNG wire#w1
   // the same network as SCL:
   #MA_Bajar_TR1 := (#Selec_E1 OR #Selec_E3 OR (#Mx_ET02 AND NOT #PosSalidaCarga_OK) OR (#Mx_ET01 AND NOT #Selec_E2 AND NOT #Selec_E1 AND NOT #Selec_E3 AND #TIM_EsperaMesaLibre.Q)) AND NOT #TR1_Abajo AND #EstadoZona.Marcha_CBx AND NOT #EstadoVI.Error_Mx AND NOT #Error_Tx;
END_REGION

REGION Network 118: SALIDAS - SUBIR TRANSTER TR2 (Neumatica)
   RUNG wire#powerrail
      Contact( #Selec_E2 )
      wire#w1
      Contact( #Selec_E2 )
      Contact( #AVTF_MAnt_Mx_BGrande )
      wire#w3
      I_Contact( #TR2_Arriba )
      Contact( #EstadoZona.Marcha_CBx )
      I_Contact( #EstadoVI.Error_Mx )
      I_Contact( #Error_Tx )
      Coil( #MA_Subir_TR2 )
   END_RUNG
   RUNG wire#powerrail
      Contact( #Selec_S4_BGrande )
      Contact( #SaliendoCarga )
      wire#w2
      Contact( #PosSalidaCarga_OK )
   END_RUNG wire#w1
   RUNG wire#powerrail
      Contact( #Selec_S4_BPequena )
      Contact( #SaliendoCarga )
   END_RUNG wire#w2
   RUNG wire#w1
      Contact( #Selec_S4_BGrande )
   END_RUNG wire#w3
   // the same network as SCL:
   #MA_Subir_TR2 := (#Selec_E2 OR (((#Selec_S4_BGrande AND #SaliendoCarga) OR (#Selec_S4_BPequena AND #SaliendoCarga)) AND #PosSalidaCarga_OK)) AND ((#Selec_E2 AND #AVTF_MAnt_Mx_BGrande) OR #Selec_S4_BGrande) AND NOT #TR2_Arriba AND #EstadoZona.Marcha_CBx AND NOT #EstadoVI.Error_Mx AND NOT #Error_Tx;
END_REGION

REGION Network 119: SALIDAS - BAJAR TRANSTER TR2 (Neumatica)
   RUNG wire#powerrail
      Contact( #Selec_E1 )
      wire#w1
      I_Contact( #TR2_Abajo )
      Contact( #EstadoZona.Marcha_CBx )
      I_Contact( #EstadoVI.Error_Mx )
      I_Contact( #Error_Tx )
      Coil( #MA_Bajar_TR2 )
   END_RUNG
   RUNG wire#powerrail
      Contact( #Selec_E3 )
   END_RUNG wire#w1
   RUNG wire#powerrail
      Contact( #Mx_ET02 )
      I_Contact( #PosSalidaCarga_OK )
   END_RUNG wire#w1
   RUNG wire#powerrail
      Contact( #Mx_ET01 )
      I_Contact( #Selec_E2 )
      I_Contact( #Selec_E1 )
      I_Contact( #Selec_E3 )
      Contact( #TIM_EsperaMesaLibre.Q )
   END_RUNG wire#w1
   // the same network as SCL:
   #MA_Bajar_TR2 := (#Selec_E1 OR #Selec_E3 OR (#Mx_ET02 AND NOT #PosSalidaCarga_OK) OR (#Mx_ET01 AND NOT #Selec_E2 AND NOT #Selec_E1 AND NOT #Selec_E3 AND #TIM_EsperaMesaLibre.Q)) AND NOT #TR2_Abajo AND #EstadoZona.Marcha_CBx AND NOT #EstadoVI.Error_Mx AND NOT #Error_Tx;
END_REGION

REGION Network 120: SALIDAS - SUBIR TOPE TPE1 (Neumatica) ????
   RUNG wire#powerrail
      I_Contact( #Mx_ET01 )
      I_Contact( #Selec_E1 )
      I_Contact( #TPE1_Arriba )
      Contact( #EstadoZona.Marcha_CBx )
      I_Contact( #EstadoVI.Error_Mx )
      I_Contact( #Error_Tx )
      Coil( #MA_Subir_TPE1 )
   END_RUNG
   // the same network as SCL:
   #MA_Subir_TPE1 := NOT #Mx_ET01 AND NOT #Selec_E1 AND NOT #TPE1_Arriba AND #EstadoZona.Marcha_CBx AND NOT #EstadoVI.Error_Mx AND NOT #Error_Tx;
END_REGION

REGION Network 121: SALIDAS - BAJAR TOPE TPE1 (Neumatica) ????
   RUNG wire#powerrail
      Contact( #Selec_E1 )
      wire#w1
      I_Contact( #TPE1_Abajo )
      Contact( #EstadoZona.Marcha_CBx )
      I_Contact( #EstadoVI.Error_Mx )
      I_Contact( #Error_Tx )
      Coil( #MA_Bajar_TPE1 )
   END_RUNG
   RUNG wire#powerrail
      Contact( #Mx_ET01 )
   END_RUNG wire#w1
   // the same network as SCL:
   #MA_Bajar_TPE1 := (#Selec_E1 OR #Mx_ET01) AND NOT #TPE1_Abajo AND #EstadoZona.Marcha_CBx AND NOT #EstadoVI.Error_Mx AND NOT #Error_Tx;
END_REGION

REGION Network 122: SALIDAS - SUBIR TOPE TPE3 (Neumatica) ????
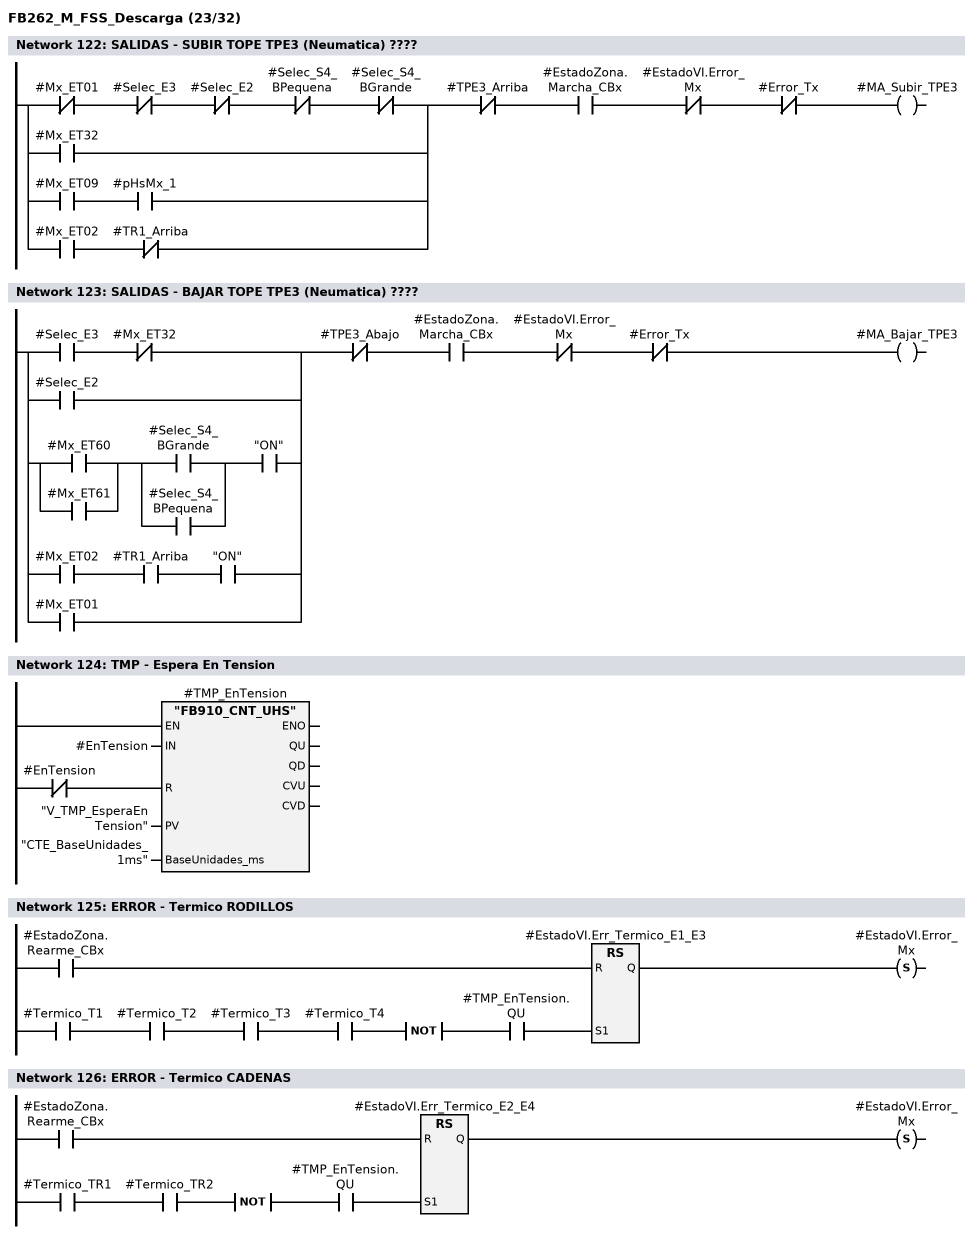
   RUNG wire#powerrail
      I_Contact( #Mx_ET01 )
      I_Contact( #Selec_E3 )
      I_Contact( #Selec_E2 )
      I_Contact( #Selec_S4_BPequena )
      I_Contact( #Selec_S4_BGrande )
      wire#w1
      I_Contact( #TPE3_Arriba )
      Contact( #EstadoZona.Marcha_CBx )
      I_Contact( #EstadoVI.Error_Mx )
      I_Contact( #Error_Tx )
      Coil( #MA_Subir_TPE3 )
   END_RUNG
   RUNG wire#powerrail
      Contact( #Mx_ET32 )
   END_RUNG wire#w1
   RUNG wire#powerrail
      Contact( #Mx_ET09 )
      Contact( #pHsMx_1 )
   END_RUNG wire#w1
   RUNG wire#powerrail
      Contact( #Mx_ET02 )
      I_Contact( #TR1_Arriba )
   END_RUNG wire#w1
   // the same network as SCL:
   #MA_Subir_TPE3 := ((NOT #Mx_ET01 AND NOT #Selec_E3 AND NOT #Selec_E2 AND NOT #Selec_S4_BPequena AND NOT #Selec_S4_BGrande) OR #Mx_ET32 OR (#Mx_ET09 AND #pHsMx_1) OR (#Mx_ET02 AND NOT #TR1_Arriba)) AND NOT #TPE3_Arriba AND #EstadoZona.Marcha_CBx AND NOT #EstadoVI.Error_Mx AND NOT #Error_Tx;
END_REGION

REGION Network 123: SALIDAS - BAJAR TOPE TPE3 (Neumatica) ????
   RUNG wire#powerrail
      Contact( #Selec_E3 )
      I_Contact( #Mx_ET32 )
      wire#w1
      I_Contact( #TPE3_Abajo )
      Contact( #EstadoZona.Marcha_CBx )
      I_Contact( #EstadoVI.Error_Mx )
      I_Contact( #Error_Tx )
      Coil( #MA_Bajar_TPE3 )
   END_RUNG
   RUNG wire#powerrail
      Contact( #Selec_E2 )
   END_RUNG wire#w1
   RUNG wire#powerrail
      Contact( #Mx_ET60 )
      wire#w2
      Contact( #Selec_S4_BGrande )
      wire#w3
      Contact( "ON" )
   END_RUNG wire#w1
   RUNG wire#powerrail
      Contact( #Mx_ET61 )
   END_RUNG wire#w2
   RUNG wire#w2
      Contact( #Selec_S4_BPequena )
   END_RUNG wire#w3
   RUNG wire#powerrail
      Contact( #Mx_ET02 )
      Contact( #TR1_Arriba )
      Contact( "ON" )
   END_RUNG wire#w1
   RUNG wire#powerrail
      Contact( #Mx_ET01 )
   END_RUNG wire#w1
   // the same network as SCL:
   #MA_Bajar_TPE3 := ((#Selec_E3 AND NOT #Mx_ET32) OR #Selec_E2 OR ((#Mx_ET60 OR #Mx_ET61) AND (#Selec_S4_BGrande OR #Selec_S4_BPequena) AND "ON") OR (#Mx_ET02 AND #TR1_Arriba AND "ON") OR #Mx_ET01) AND NOT #TPE3_Abajo AND #EstadoZona.Marcha_CBx AND NOT #EstadoVI.Error_Mx AND NOT #Error_Tx;
END_REGION

REGION Network 124: TMP - Espera En Tension
   RUNG wire#powerrail
      #TMP_EnTension(R := wire#w1, IN := #EnTension, PV := "V_TMP_EsperaEnTension", BaseUnidades_ms := "CTE_BaseUnidades_1ms", QU =>, QD =>, CVU =>, CVD =>)
   END_RUNG
   RUNG wire#powerrail
      I_Contact( #EnTension )
   END_RUNG wire#w1
   // the same network as SCL:
   #TMP_EnTension(IN := #EnTension,   // "FB910_CNT_UHS"
                  R := NOT #EnTension,
                  PV := "V_TMP_EsperaEnTension",
                  BaseUnidades_ms := "CTE_BaseUnidades_1ms");
END_REGION

REGION Network 125: ERROR - Termico RODILLOS
   RUNG wire#powerrail
      Contact( #EstadoZona.Rearme_CBx )
      S_RS(operand := #EstadoVI.Err_Termico_E1_E3, s1 := wire#w1)
      S_Coil( #EstadoVI.Error_Mx )
   END_RUNG
   RUNG wire#powerrail
      Contact( #Termico_T1 )
      Contact( #Termico_T2 )
      Contact( #Termico_T3 )
      Contact( #Termico_T4 )
      Not()
      Contact( #TMP_EnTension.QU )
   END_RUNG wire#w1
   // the same network as SCL:
   IF #EstadoZona.Rearme_CBx THEN
       #EstadoVI.Err_Termico_E1_E3 := FALSE;   // RS flip-flop
   END_IF;
   IF NOT (#Termico_T1 AND #Termico_T2 AND #Termico_T3 AND #Termico_T4) AND #TMP_EnTension.QU THEN
       #EstadoVI.Err_Termico_E1_E3 := TRUE;
   END_IF;
   IF #EstadoVI.Err_Termico_E1_E3 THEN #EstadoVI.Error_Mx := TRUE; END_IF;
END_REGION

REGION Network 126: ERROR - Termico CADENAS
   RUNG wire#powerrail
      Contact( #EstadoZona.Rearme_CBx )
      S_RS(operand := #EstadoVI.Err_Termico_E2_E4, s1 := wire#w1)
      S_Coil( #EstadoVI.Error_Mx )
   END_RUNG
   RUNG wire#powerrail
      Contact( #Termico_TR1 )
      Contact( #Termico_TR2 )
      Not()
      Contact( #TMP_EnTension.QU )
   END_RUNG wire#w1
   // the same network as SCL:
   IF #EstadoZona.Rearme_CBx THEN
       #EstadoVI.Err_Termico_E2_E4 := FALSE;   // RS flip-flop
   END_IF;
   IF NOT (#Termico_TR1 AND #Termico_TR2) AND #TMP_EnTension.QU THEN
       #EstadoVI.Err_Termico_E2_E4 := TRUE;
   END_IF;
   IF #EstadoVI.Err_Termico_E2_E4 THEN #EstadoVI.Error_Mx := TRUE; END_IF;
END_REGION

REGION Network 127: ERROR - Mesa Ocupada
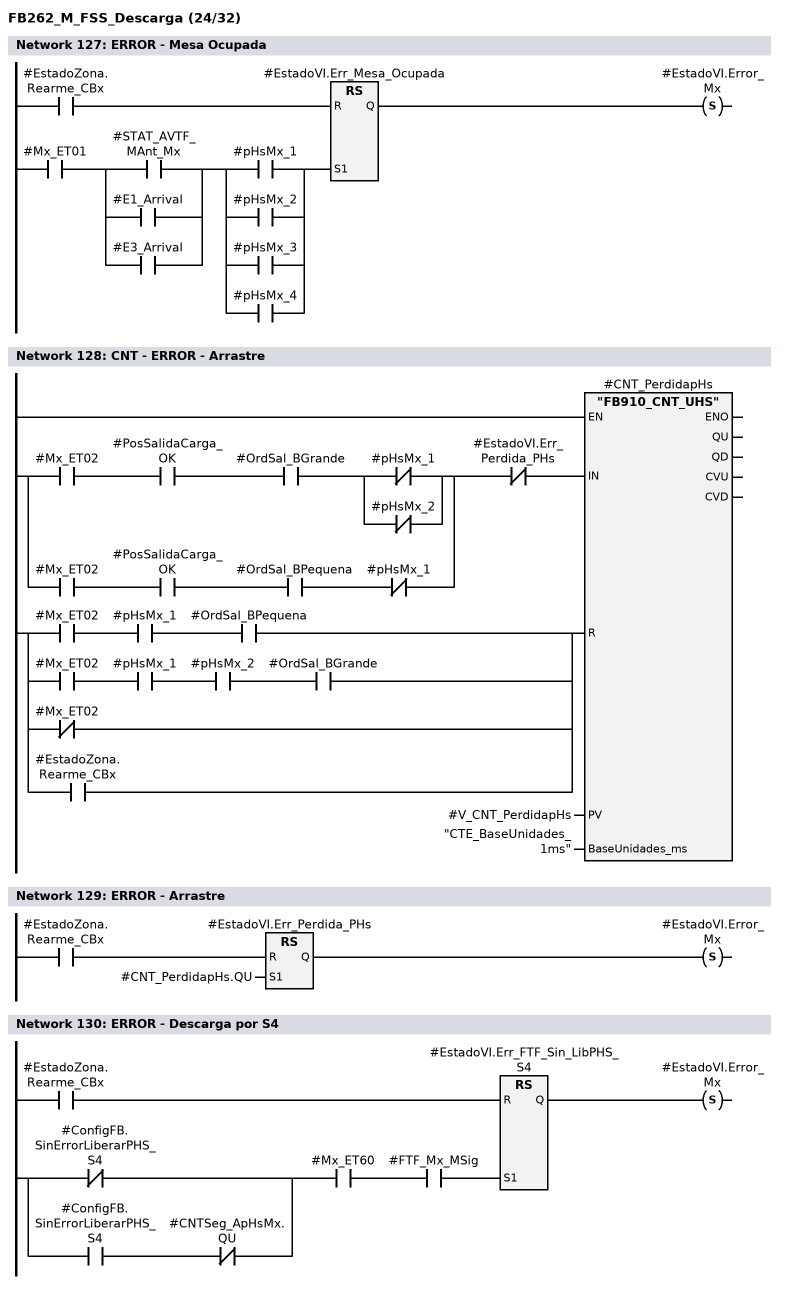
   RUNG wire#powerrail
      Contact( #EstadoZona.Rearme_CBx )
      S_RS(operand := #EstadoVI.Err_Mesa_Ocupada, s1 := wire#w3)
      S_Coil( #EstadoVI.Error_Mx )
   END_RUNG
   RUNG wire#powerrail
      Contact( #Mx_ET01 )
      wire#w1
      Contact( #STAT_AVTF_MAnt_Mx )
      wire#w2
      Contact( #pHsMx_1 )
   END_RUNG wire#w3
   RUNG wire#w1
      Contact( #E1_Arrival )
   END_RUNG wire#w2
   RUNG wire#w1
      Contact( #E3_Arrival )
   END_RUNG wire#w2
   RUNG wire#w2
      Contact( #pHsMx_2 )
   END_RUNG wire#w3
   RUNG wire#w2
      Contact( #pHsMx_3 )
   END_RUNG wire#w3
   RUNG wire#w2
      Contact( #pHsMx_4 )
   END_RUNG wire#w3
   // the same network as SCL:
   IF #EstadoZona.Rearme_CBx THEN
       #EstadoVI.Err_Mesa_Ocupada := FALSE;   // RS flip-flop
   END_IF;
   IF #Mx_ET01 AND (#STAT_AVTF_MAnt_Mx OR #E1_Arrival OR #E3_Arrival) AND (#pHsMx_1 OR #pHsMx_2 OR #pHsMx_3 OR #pHsMx_4) THEN
       #EstadoVI.Err_Mesa_Ocupada := TRUE;
   END_IF;
   IF #EstadoVI.Err_Mesa_Ocupada THEN #EstadoVI.Error_Mx := TRUE; END_IF;
END_REGION

REGION Network 128: CNT - ERROR - Arrastre
   RUNG wire#powerrail
      #CNT_PerdidapHs(IN := wire#w3, R := wire#w4, PV := #V_CNT_PerdidapHs, BaseUnidades_ms := "CTE_BaseUnidades_1ms", QU =>, QD =>, CVU =>, CVD =>)
   END_RUNG
   RUNG wire#powerrail
      Contact( #Mx_ET02 )
      Contact( #PosSalidaCarga_OK )
      Contact( #OrdSal_BGrande )
      wire#w1
      I_Contact( #pHsMx_1 )
      wire#w2
      I_Contact( #EstadoVI.Err_Perdida_PHs )
   END_RUNG wire#w3
   RUNG wire#w1
      I_Contact( #pHsMx_2 )
   END_RUNG wire#w2
   RUNG wire#powerrail
      Contact( #Mx_ET02 )
      Contact( #PosSalidaCarga_OK )
      Contact( #OrdSal_BPequena )
      I_Contact( #pHsMx_1 )
   END_RUNG wire#w2
   RUNG wire#powerrail
      Contact( #Mx_ET02 )
      Contact( #pHsMx_1 )
      Contact( #OrdSal_BPequena )
   END_RUNG wire#w4
   RUNG wire#powerrail
      Contact( #Mx_ET02 )
      Contact( #pHsMx_1 )
      Contact( #pHsMx_2 )
      Contact( #OrdSal_BGrande )
   END_RUNG wire#w4
   RUNG wire#powerrail
      I_Contact( #Mx_ET02 )
   END_RUNG wire#w4
   RUNG wire#powerrail
      Contact( #EstadoZona.Rearme_CBx )
   END_RUNG wire#w4
   // the same network as SCL:
   #CNT_PerdidapHs(IN := ((#Mx_ET02 AND #PosSalidaCarga_OK AND #OrdSal_BGrande AND (NOT #pHsMx_1 OR NOT #pHsMx_2)) OR (#Mx_ET02 AND #PosSalidaCarga_OK AND #OrdSal_BPequena AND NOT #pHsMx_1)) AND NOT #EstadoVI.Err_Perdida_PHs,   // "FB910_CNT_UHS"
                   R := (#Mx_ET02 AND #pHsMx_1 AND #OrdSal_BPequena) OR (#Mx_ET02 AND #pHsMx_1 AND #pHsMx_2 AND #OrdSal_BGrande) OR NOT #Mx_ET02 OR #EstadoZona.Rearme_CBx,
                   PV := #V_CNT_PerdidapHs,
                   BaseUnidades_ms := "CTE_BaseUnidades_1ms");
END_REGION

REGION Network 129: ERROR - Arrastre
   RUNG wire#powerrail
      Contact( #EstadoZona.Rearme_CBx )
      S_RS(operand := #EstadoVI.Err_Perdida_PHs, s1 := #CNT_PerdidapHs.QU)
      S_Coil( #EstadoVI.Error_Mx )
   END_RUNG
   // the same network as SCL:
   IF #EstadoZona.Rearme_CBx THEN
       #EstadoVI.Err_Perdida_PHs := FALSE;   // RS flip-flop
   END_IF;
   IF #CNT_PerdidapHs.QU THEN #EstadoVI.Err_Perdida_PHs := TRUE; END_IF;
   IF #EstadoVI.Err_Perdida_PHs THEN #EstadoVI.Error_Mx := TRUE; END_IF;
END_REGION

REGION Network 130: ERROR - Descarga por S4
   RUNG wire#powerrail
      Contact( #EstadoZona.Rearme_CBx )
      S_RS(operand := #EstadoVI.Err_FTF_Sin_LibPHS_S4, s1 := wire#w2)
      S_Coil( #EstadoVI.Error_Mx )
   END_RUNG
   RUNG wire#powerrail
      I_Contact( #ConfigFB.SinErrorLiberarPHS_S4 )
      wire#w1
      Contact( #Mx_ET60 )
      Contact( #FTF_Mx_MSig )
   END_RUNG wire#w2
   RUNG wire#powerrail
      Contact( #ConfigFB.SinErrorLiberarPHS_S4 )
      I_Contact( #CNTSeg_ApHsMx.QU )
   END_RUNG wire#w1
   // the same network as SCL:
   IF #EstadoZona.Rearme_CBx THEN
       #EstadoVI.Err_FTF_Sin_LibPHS_S4 := FALSE;   // RS flip-flop
   END_IF;
   IF (NOT #ConfigFB.SinErrorLiberarPHS_S4 OR (#ConfigFB.SinErrorLiberarPHS_S4 AND NOT #CNTSeg_ApHsMx.QU)) AND #Mx_ET60 AND #FTF_Mx_MSig THEN
       #EstadoVI.Err_FTF_Sin_LibPHS_S4 := TRUE;
   END_IF;
   IF #EstadoVI.Err_FTF_Sin_LibPHS_S4 THEN #EstadoVI.Error_Mx := TRUE; END_IF;
END_REGION

REGION Network 131: TMP - ERROR - TimeOut Avance Tx >>> DESCARGA FSS Y REPOSICONADO
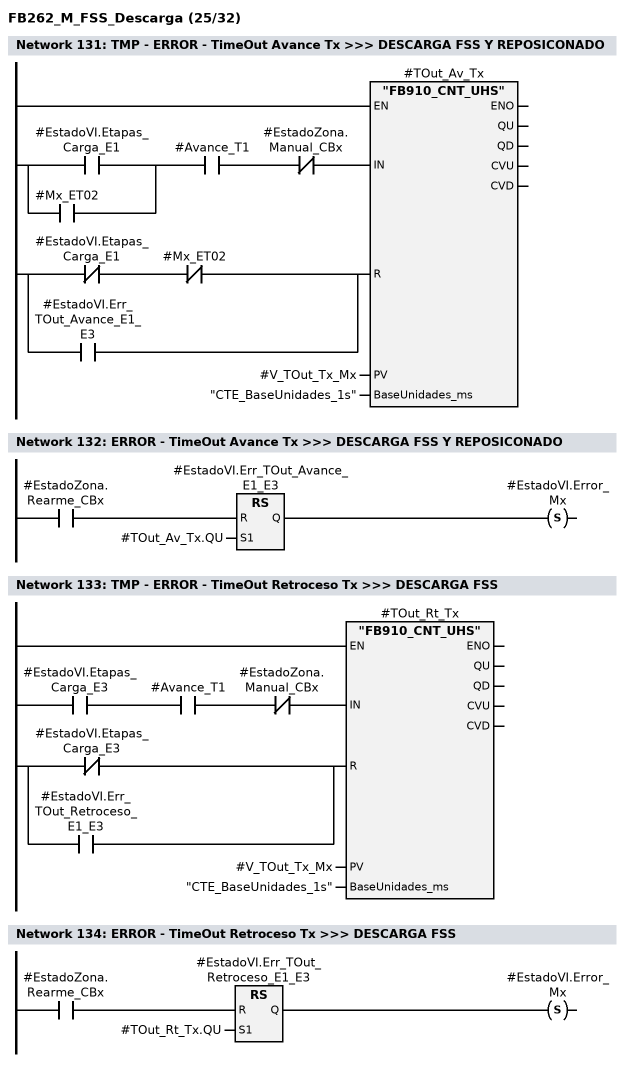
   RUNG wire#powerrail
      #TOut_Av_Tx(IN := wire#w2, R := wire#w3, PV := #V_TOut_Tx_Mx, BaseUnidades_ms := "CTE_BaseUnidades_1s", QU =>, QD =>, CVU =>, CVD =>)
   END_RUNG
   RUNG wire#powerrail
      Contact( #EstadoVI.Etapas_Carga_E1 )
      wire#w1
      Contact( #Avance_T1 )
      I_Contact( #EstadoZona.Manual_CBx )
   END_RUNG wire#w2
   RUNG wire#powerrail
      Contact( #Mx_ET02 )
   END_RUNG wire#w1
   RUNG wire#powerrail
      I_Contact( #EstadoVI.Etapas_Carga_E1 )
      I_Contact( #Mx_ET02 )
   END_RUNG wire#w3
   RUNG wire#powerrail
      Contact( #EstadoVI.Err_TOut_Avance_E1_E3 )
   END_RUNG wire#w3
   // the same network as SCL:
   #TOut_Av_Tx(IN := (#EstadoVI.Etapas_Carga_E1 OR #Mx_ET02) AND #Avance_T1 AND NOT #EstadoZona.Manual_CBx,   // "FB910_CNT_UHS"
               R := (NOT #EstadoVI.Etapas_Carga_E1 AND NOT #Mx_ET02) OR #EstadoVI.Err_TOut_Avance_E1_E3,
               PV := #V_TOut_Tx_Mx,
               BaseUnidades_ms := "CTE_BaseUnidades_1s");
END_REGION

REGION Network 132: ERROR - TimeOut Avance Tx >>> DESCARGA FSS Y REPOSICONADO
   RUNG wire#powerrail
      Contact( #EstadoZona.Rearme_CBx )
      S_RS(operand := #EstadoVI.Err_TOut_Avance_E1_E3, s1 := #TOut_Av_Tx.QU)
      S_Coil( #EstadoVI.Error_Mx )
   END_RUNG
   // the same network as SCL:
   IF #EstadoZona.Rearme_CBx THEN
       #EstadoVI.Err_TOut_Avance_E1_E3 := FALSE;   // RS flip-flop
   END_IF;
   IF #TOut_Av_Tx.QU THEN #EstadoVI.Err_TOut_Avance_E1_E3 := TRUE; END_IF;
   IF #EstadoVI.Err_TOut_Avance_E1_E3 THEN #EstadoVI.Error_Mx := TRUE; END_IF;
END_REGION

REGION Network 133: TMP - ERROR - TimeOut Retroceso Tx >>> DESCARGA FSS
   RUNG wire#powerrail
      #TOut_Rt_Tx(IN := wire#w1, R := wire#w2, PV := #V_TOut_Tx_Mx, BaseUnidades_ms := "CTE_BaseUnidades_1s", QU =>, QD =>, CVU =>, CVD =>)
   END_RUNG
   RUNG wire#powerrail
      Contact( #EstadoVI.Etapas_Carga_E3 )
      Contact( #Avance_T1 )
      I_Contact( #EstadoZona.Manual_CBx )
   END_RUNG wire#w1
   RUNG wire#powerrail
      I_Contact( #EstadoVI.Etapas_Carga_E3 )
   END_RUNG wire#w2
   RUNG wire#powerrail
      Contact( #EstadoVI.Err_TOut_Retroceso_E1_E3 )
   END_RUNG wire#w2
   // the same network as SCL:
   #TOut_Rt_Tx(IN := #EstadoVI.Etapas_Carga_E3 AND #Avance_T1 AND NOT #EstadoZona.Manual_CBx,   // "FB910_CNT_UHS"
               R := NOT #EstadoVI.Etapas_Carga_E3 OR #EstadoVI.Err_TOut_Retroceso_E1_E3,
               PV := #V_TOut_Tx_Mx,
               BaseUnidades_ms := "CTE_BaseUnidades_1s");
END_REGION

REGION Network 134: ERROR - TimeOut Retroceso Tx >>> DESCARGA FSS
   RUNG wire#powerrail
      Contact( #EstadoZona.Rearme_CBx )
      S_RS(operand := #EstadoVI.Err_TOut_Retroceso_E1_E3, s1 := #TOut_Rt_Tx.QU)
      S_Coil( #EstadoVI.Error_Mx )
   END_RUNG
   // the same network as SCL:
   IF #EstadoZona.Rearme_CBx THEN
       #EstadoVI.Err_TOut_Retroceso_E1_E3 := FALSE;   // RS flip-flop
   END_IF;
   IF #TOut_Rt_Tx.QU THEN #EstadoVI.Err_TOut_Retroceso_E1_E3 := TRUE; END_IF;
   IF #EstadoVI.Err_TOut_Retroceso_E1_E3 THEN #EstadoVI.Error_Mx := TRUE; END_IF;
END_REGION

REGION Network 135: TMP - ERROR - TimeOut Avance TRx >>> ENTRADA
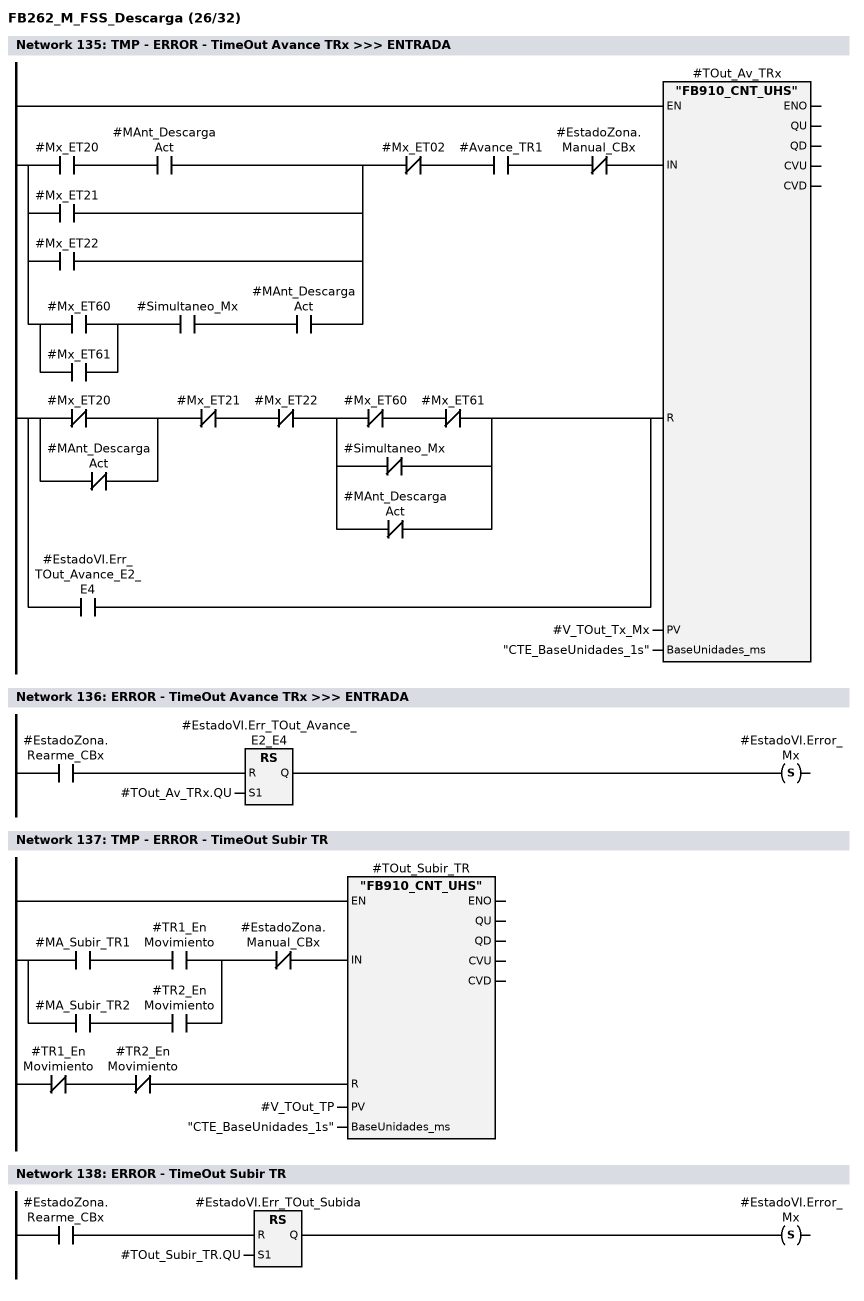
   RUNG wire#powerrail
      #TOut_Av_TRx(IN := wire#w3, R := wire#w6, PV := #V_TOut_Tx_Mx, BaseUnidades_ms := "CTE_BaseUnidades_1s", QU =>, QD =>, CVU =>, CVD =>)
   END_RUNG
   RUNG wire#powerrail
      Contact( #Mx_ET20 )
      Contact( #MAnt_DescargaAct )
      wire#w1
      I_Contact( #Mx_ET02 )
      Contact( #Avance_TR1 )
      I_Contact( #EstadoZona.Manual_CBx )
   END_RUNG wire#w3
   RUNG wire#powerrail
      Contact( #Mx_ET21 )
   END_RUNG wire#w1
   RUNG wire#powerrail
      Contact( #Mx_ET22 )
   END_RUNG wire#w1
   RUNG wire#powerrail
      Contact( #Mx_ET60 )
      wire#w2
      Contact( #Simultaneo_Mx )
      Contact( #MAnt_DescargaAct )
   END_RUNG wire#w1
   RUNG wire#powerrail
      Contact( #Mx_ET61 )
   END_RUNG wire#w2
   RUNG wire#powerrail
      I_Contact( #Mx_ET20 )
      wire#w4
      I_Contact( #Mx_ET21 )
      I_Contact( #Mx_ET22 )
      wire#w5
      I_Contact( #Mx_ET60 )
      I_Contact( #Mx_ET61 )
   END_RUNG wire#w6
   RUNG wire#powerrail
      I_Contact( #MAnt_DescargaAct )
   END_RUNG wire#w4
   RUNG wire#w5
      I_Contact( #Simultaneo_Mx )
   END_RUNG wire#w6
   RUNG wire#w5
      I_Contact( #MAnt_DescargaAct )
   END_RUNG wire#w6
   RUNG wire#powerrail
      Contact( #EstadoVI.Err_TOut_Avance_E2_E4 )
   END_RUNG wire#w6
   // the same network as SCL:
   #TOut_Av_TRx(IN := ((#Mx_ET20 AND #MAnt_DescargaAct) OR #Mx_ET21 OR #Mx_ET22 OR ((#Mx_ET60 OR #Mx_ET61) AND #Simultaneo_Mx AND #MAnt_DescargaAct)) AND NOT #Mx_ET02 AND #Avance_TR1 AND NOT #EstadoZona.Manual_CBx,   // "FB910_CNT_UHS"
                R := ((NOT #Mx_ET20 OR NOT #MAnt_DescargaAct) AND NOT #Mx_ET21 AND NOT #Mx_ET22 AND ((NOT #Mx_ET60 AND NOT #Mx_ET61) OR NOT #Simultaneo_Mx OR NOT #MAnt_DescargaAct)) OR #EstadoVI.Err_TOut_Avance_E2_E4,
                PV := #V_TOut_Tx_Mx,
                BaseUnidades_ms := "CTE_BaseUnidades_1s");
END_REGION

REGION Network 136: ERROR - TimeOut Avance TRx >>> ENTRADA
   RUNG wire#powerrail
      Contact( #EstadoZona.Rearme_CBx )
      S_RS(operand := #EstadoVI.Err_TOut_Avance_E2_E4, s1 := #TOut_Av_TRx.QU)
      S_Coil( #EstadoVI.Error_Mx )
   END_RUNG
   // the same network as SCL:
   IF #EstadoZona.Rearme_CBx THEN
       #EstadoVI.Err_TOut_Avance_E2_E4 := FALSE;   // RS flip-flop
   END_IF;
   IF #TOut_Av_TRx.QU THEN #EstadoVI.Err_TOut_Avance_E2_E4 := TRUE; END_IF;
   IF #EstadoVI.Err_TOut_Avance_E2_E4 THEN #EstadoVI.Error_Mx := TRUE; END_IF;
END_REGION

REGION Network 137: TMP - ERROR - TimeOut Subir TR
   RUNG wire#powerrail
      #TOut_Subir_TR(IN := wire#w2, R := wire#w3, PV := #V_TOut_TP, BaseUnidades_ms := "CTE_BaseUnidades_1s", QU =>, QD =>, CVU =>, CVD =>)
   END_RUNG
   RUNG wire#powerrail
      Contact( #MA_Subir_TR1 )
      Contact( #TR1_EnMovimiento )
      wire#w1
      I_Contact( #EstadoZona.Manual_CBx )
   END_RUNG wire#w2
   RUNG wire#powerrail
      Contact( #MA_Subir_TR2 )
      Contact( #TR2_EnMovimiento )
   END_RUNG wire#w1
   RUNG wire#powerrail
      I_Contact( #TR1_EnMovimiento )
      I_Contact( #TR2_EnMovimiento )
   END_RUNG wire#w3
   // the same network as SCL:
   #TOut_Subir_TR(IN := ((#MA_Subir_TR1 AND #TR1_EnMovimiento) OR (#MA_Subir_TR2 AND #TR2_EnMovimiento)) AND NOT #EstadoZona.Manual_CBx,   // "FB910_CNT_UHS"
                  R := NOT #TR1_EnMovimiento AND NOT #TR2_EnMovimiento,
                  PV := #V_TOut_TP,
                  BaseUnidades_ms := "CTE_BaseUnidades_1s");
END_REGION

REGION Network 138: ERROR - TimeOut Subir TR
   RUNG wire#powerrail
      Contact( #EstadoZona.Rearme_CBx )
      S_RS(operand := #EstadoVI.Err_TOut_Subida, s1 := #TOut_Subir_TR.QU)
      S_Coil( #EstadoVI.Error_Mx )
   END_RUNG
   // the same network as SCL:
   IF #EstadoZona.Rearme_CBx THEN
       #EstadoVI.Err_TOut_Subida := FALSE;   // RS flip-flop
   END_IF;
   IF #TOut_Subir_TR.QU THEN #EstadoVI.Err_TOut_Subida := TRUE; END_IF;
   IF #EstadoVI.Err_TOut_Subida THEN #EstadoVI.Error_Mx := TRUE; END_IF;
END_REGION

REGION Network 139: TMP - ERROR - TimeOut Bajar TR
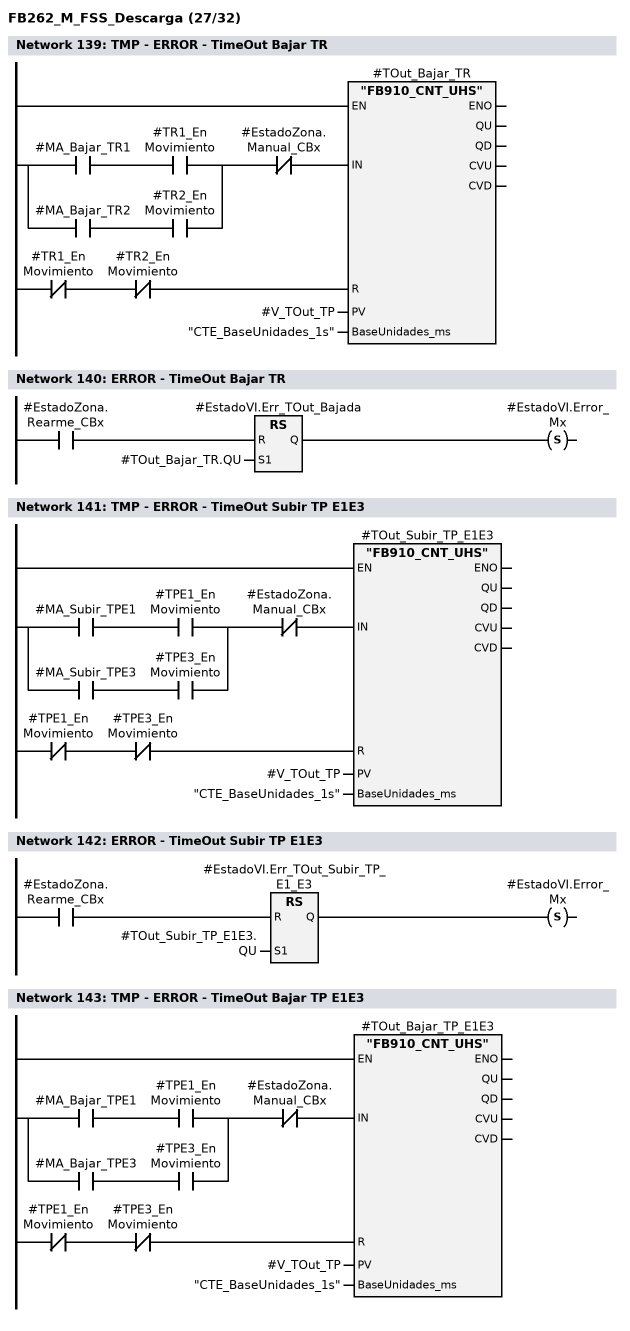
   RUNG wire#powerrail
      #TOut_Bajar_TR(IN := wire#w2, R := wire#w3, PV := #V_TOut_TP, BaseUnidades_ms := "CTE_BaseUnidades_1s", QU =>, QD =>, CVU =>, CVD =>)
   END_RUNG
   RUNG wire#powerrail
      Contact( #MA_Bajar_TR1 )
      Contact( #TR1_EnMovimiento )
      wire#w1
      I_Contact( #EstadoZona.Manual_CBx )
   END_RUNG wire#w2
   RUNG wire#powerrail
      Contact( #MA_Bajar_TR2 )
      Contact( #TR2_EnMovimiento )
   END_RUNG wire#w1
   RUNG wire#powerrail
      I_Contact( #TR1_EnMovimiento )
      I_Contact( #TR2_EnMovimiento )
   END_RUNG wire#w3
   // the same network as SCL:
   #TOut_Bajar_TR(IN := ((#MA_Bajar_TR1 AND #TR1_EnMovimiento) OR (#MA_Bajar_TR2 AND #TR2_EnMovimiento)) AND NOT #EstadoZona.Manual_CBx,   // "FB910_CNT_UHS"
                  R := NOT #TR1_EnMovimiento AND NOT #TR2_EnMovimiento,
                  PV := #V_TOut_TP,
                  BaseUnidades_ms := "CTE_BaseUnidades_1s");
END_REGION

REGION Network 140: ERROR - TimeOut Bajar TR
   RUNG wire#powerrail
      Contact( #EstadoZona.Rearme_CBx )
      S_RS(operand := #EstadoVI.Err_TOut_Bajada, s1 := #TOut_Bajar_TR.QU)
      S_Coil( #EstadoVI.Error_Mx )
   END_RUNG
   // the same network as SCL:
   IF #EstadoZona.Rearme_CBx THEN
       #EstadoVI.Err_TOut_Bajada := FALSE;   // RS flip-flop
   END_IF;
   IF #TOut_Bajar_TR.QU THEN #EstadoVI.Err_TOut_Bajada := TRUE; END_IF;
   IF #EstadoVI.Err_TOut_Bajada THEN #EstadoVI.Error_Mx := TRUE; END_IF;
END_REGION

REGION Network 141: TMP - ERROR - TimeOut Subir TP E1E3
   RUNG wire#powerrail
      #TOut_Subir_TP_E1E3(IN := wire#w2, R := wire#w3, PV := #V_TOut_TP, BaseUnidades_ms := "CTE_BaseUnidades_1s", QU =>, QD =>, CVU =>, CVD =>)
   END_RUNG
   RUNG wire#powerrail
      Contact( #MA_Subir_TPE1 )
      Contact( #TPE1_EnMovimiento )
      wire#w1
      I_Contact( #EstadoZona.Manual_CBx )
   END_RUNG wire#w2
   RUNG wire#powerrail
      Contact( #MA_Subir_TPE3 )
      Contact( #TPE3_EnMovimiento )
   END_RUNG wire#w1
   RUNG wire#powerrail
      I_Contact( #TPE1_EnMovimiento )
      I_Contact( #TPE3_EnMovimiento )
   END_RUNG wire#w3
   // the same network as SCL:
   #TOut_Subir_TP_E1E3(IN := ((#MA_Subir_TPE1 AND #TPE1_EnMovimiento) OR (#MA_Subir_TPE3 AND #TPE3_EnMovimiento)) AND NOT #EstadoZona.Manual_CBx,   // "FB910_CNT_UHS"
                       R := NOT #TPE1_EnMovimiento AND NOT #TPE3_EnMovimiento,
                       PV := #V_TOut_TP,
                       BaseUnidades_ms := "CTE_BaseUnidades_1s");
END_REGION

REGION Network 142: ERROR - TimeOut Subir TP E1E3
   RUNG wire#powerrail
      Contact( #EstadoZona.Rearme_CBx )
      S_RS(operand := #EstadoVI.Err_TOut_Subir_TP_E1_E3, s1 := #TOut_Subir_TP_E1E3.QU)
      S_Coil( #EstadoVI.Error_Mx )
   END_RUNG
   // the same network as SCL:
   IF #EstadoZona.Rearme_CBx THEN
       #EstadoVI.Err_TOut_Subir_TP_E1_E3 := FALSE;   // RS flip-flop
   END_IF;
   IF #TOut_Subir_TP_E1E3.QU THEN #EstadoVI.Err_TOut_Subir_TP_E1_E3 := TRUE; END_IF;
   IF #EstadoVI.Err_TOut_Subir_TP_E1_E3 THEN #EstadoVI.Error_Mx := TRUE; END_IF;
END_REGION

REGION Network 143: TMP - ERROR - TimeOut Bajar TP E1E3
   RUNG wire#powerrail
      #TOut_Bajar_TP_E1E3(IN := wire#w2, R := wire#w3, PV := #V_TOut_TP, BaseUnidades_ms := "CTE_BaseUnidades_1s", QU =>, QD =>, CVU =>, CVD =>)
   END_RUNG
   RUNG wire#powerrail
      Contact( #MA_Bajar_TPE1 )
      Contact( #TPE1_EnMovimiento )
      wire#w1
      I_Contact( #EstadoZona.Manual_CBx )
   END_RUNG wire#w2
   RUNG wire#powerrail
      Contact( #MA_Bajar_TPE3 )
      Contact( #TPE3_EnMovimiento )
   END_RUNG wire#w1
   RUNG wire#powerrail
      I_Contact( #TPE1_EnMovimiento )
      I_Contact( #TPE3_EnMovimiento )
   END_RUNG wire#w3
   // the same network as SCL:
   #TOut_Bajar_TP_E1E3(IN := ((#MA_Bajar_TPE1 AND #TPE1_EnMovimiento) OR (#MA_Bajar_TPE3 AND #TPE3_EnMovimiento)) AND NOT #EstadoZona.Manual_CBx,   // "FB910_CNT_UHS"
                       R := NOT #TPE1_EnMovimiento AND NOT #TPE3_EnMovimiento,
                       PV := #V_TOut_TP,
                       BaseUnidades_ms := "CTE_BaseUnidades_1s");
END_REGION

REGION Network 144: ERROR - TimeOut Bajar TP E1E3
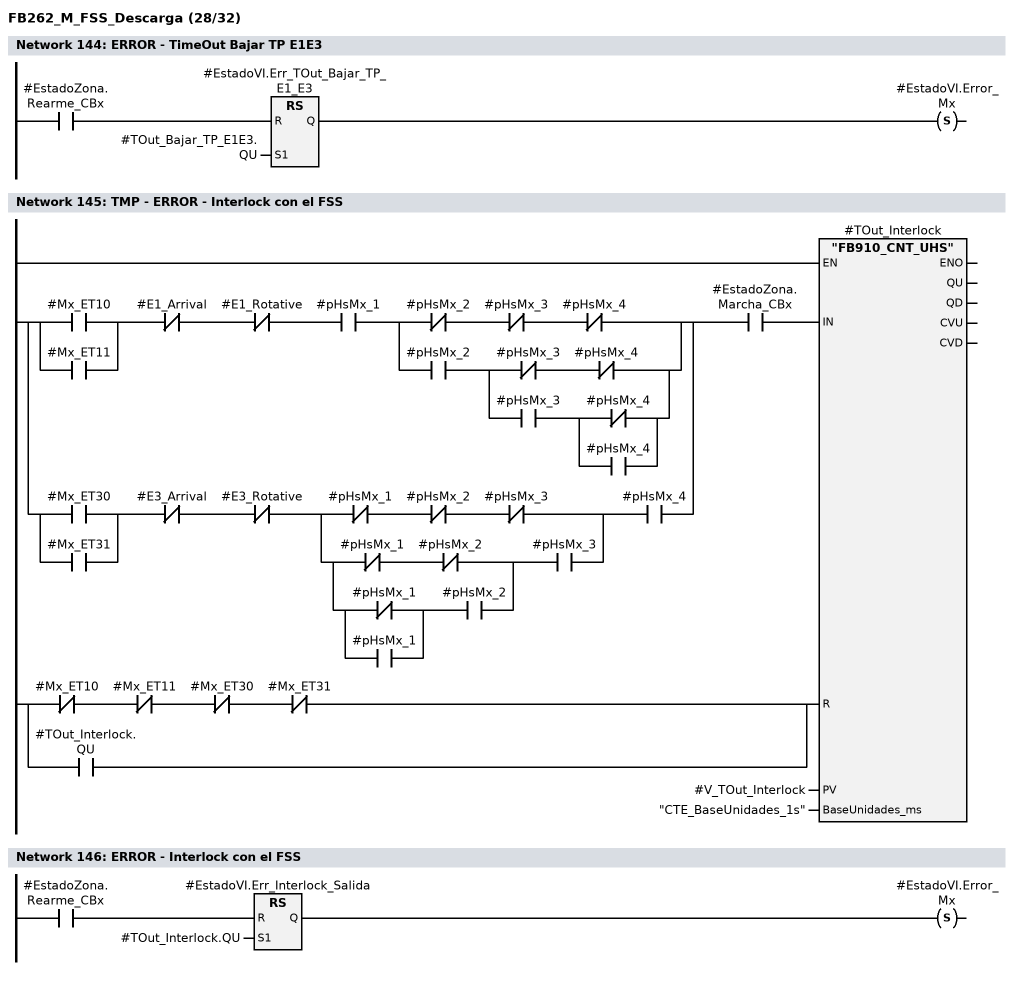
   RUNG wire#powerrail
      Contact( #EstadoZona.Rearme_CBx )
      S_RS(operand := #EstadoVI.Err_TOut_Bajar_TP_E1_E3, s1 := #TOut_Bajar_TP_E1E3.QU)
      S_Coil( #EstadoVI.Error_Mx )
   END_RUNG
   // the same network as SCL:
   IF #EstadoZona.Rearme_CBx THEN
       #EstadoVI.Err_TOut_Bajar_TP_E1_E3 := FALSE;   // RS flip-flop
   END_IF;
   IF #TOut_Bajar_TP_E1E3.QU THEN #EstadoVI.Err_TOut_Bajar_TP_E1_E3 := TRUE; END_IF;
   IF #EstadoVI.Err_TOut_Bajar_TP_E1_E3 THEN #EstadoVI.Error_Mx := TRUE; END_IF;
END_REGION

REGION Network 145: TMP - ERROR - Interlock con el FSS
   RUNG wire#powerrail
      #TOut_Interlock(IN := wire#w11, R := wire#w12, PV := #V_TOut_Interlock, BaseUnidades_ms := "CTE_BaseUnidades_1s", QU =>, QD =>, CVU =>, CVD =>)
   END_RUNG
   RUNG wire#powerrail
      Contact( #Mx_ET10 )
      wire#w1
      I_Contact( #E1_Arrival )
      I_Contact( #E1_Rotative )
      Contact( #pHsMx_1 )
      wire#w2
      I_Contact( #pHsMx_2 )
      I_Contact( #pHsMx_3 )
      I_Contact( #pHsMx_4 )
      wire#w3
      Contact( #EstadoZona.Marcha_CBx )
   END_RUNG wire#w11
   RUNG wire#powerrail
      Contact( #Mx_ET11 )
   END_RUNG wire#w1
   RUNG wire#w2
      Contact( #pHsMx_2 )
      wire#w4
      I_Contact( #pHsMx_3 )
      I_Contact( #pHsMx_4 )
   END_RUNG wire#w3
   RUNG wire#w4
      Contact( #pHsMx_3 )
      wire#w5
      I_Contact( #pHsMx_4 )
   END_RUNG wire#w3
   RUNG wire#w5
      Contact( #pHsMx_4 )
   END_RUNG wire#w3
   RUNG wire#powerrail
      Contact( #Mx_ET30 )
      wire#w6
      I_Contact( #E3_Arrival )
      I_Contact( #E3_Rotative )
      wire#w7
      I_Contact( #pHsMx_1 )
      I_Contact( #pHsMx_2 )
      I_Contact( #pHsMx_3 )
      wire#w8
      Contact( #pHsMx_4 )
   END_RUNG wire#w3
   RUNG wire#powerrail
      Contact( #Mx_ET31 )
   END_RUNG wire#w6
   RUNG wire#w7
      I_Contact( #pHsMx_1 )
      I_Contact( #pHsMx_2 )
      wire#w9
      Contact( #pHsMx_3 )
   END_RUNG wire#w8
   RUNG wire#w7
      I_Contact( #pHsMx_1 )
      wire#w10
      Contact( #pHsMx_2 )
   END_RUNG wire#w9
   RUNG wire#w7
      Contact( #pHsMx_1 )
   END_RUNG wire#w10
   RUNG wire#powerrail
      I_Contact( #Mx_ET10 )
      I_Contact( #Mx_ET11 )
      I_Contact( #Mx_ET30 )
      I_Contact( #Mx_ET31 )
   END_RUNG wire#w12
   RUNG wire#powerrail
      Contact( #TOut_Interlock.QU )
   END_RUNG wire#w12
   // the same network as SCL:
   #TOut_Interlock(IN := (((#Mx_ET10 OR #Mx_ET11) AND NOT #E1_Arrival AND NOT #E1_Rotative AND #pHsMx_1 AND ((NOT #pHsMx_2 AND NOT #pHsMx_3 AND NOT #pHsMx_4) OR (#pHsMx_2 AND ((NOT #pHsMx_3 AND NOT #pHsMx_4) OR (#pHsMx_3 AND (NOT #pHsMx_4 OR #pHsMx_4)))))) OR ((#Mx_ET30 OR #Mx_ET31) AND NOT #E3_Arrival AND NOT #E3_Rotative AND ((NOT #pHsMx_1 AND NOT #pHsMx_2 AND NOT #pHsMx_3) OR (((NOT #pHsMx_1 AND NOT #pHsMx_2) OR ((NOT #pHsMx_1 OR #pHsMx_1) AND #pHsMx_2)) AND #pHsMx_3)) AND #pHsMx_4)) AND #EstadoZona.Marcha_CBx,   // "FB910_CNT_UHS"
                   R := (NOT #Mx_ET10 AND NOT #Mx_ET11 AND NOT #Mx_ET30 AND NOT #Mx_ET31) OR #TOut_Interlock.QU,
                   PV := #V_TOut_Interlock,
                   BaseUnidades_ms := "CTE_BaseUnidades_1s");
END_REGION

REGION Network 146: ERROR - Interlock con el FSS
   RUNG wire#powerrail
      Contact( #EstadoZona.Rearme_CBx )
      S_RS(operand := #EstadoVI.Err_Interlock_Salida, s1 := #TOut_Interlock.QU)
      S_Coil( #EstadoVI.Error_Mx )
   END_RUNG
   // the same network as SCL:
   IF #EstadoZona.Rearme_CBx THEN
       #EstadoVI.Err_Interlock_Salida := FALSE;   // RS flip-flop
   END_IF;
   IF #TOut_Interlock.QU THEN #EstadoVI.Err_Interlock_Salida := TRUE; END_IF;
   IF #EstadoVI.Err_Interlock_Salida THEN #EstadoVI.Error_Mx := TRUE; END_IF;
END_REGION

REGION Network 147: ESTADOS DE LA MESA
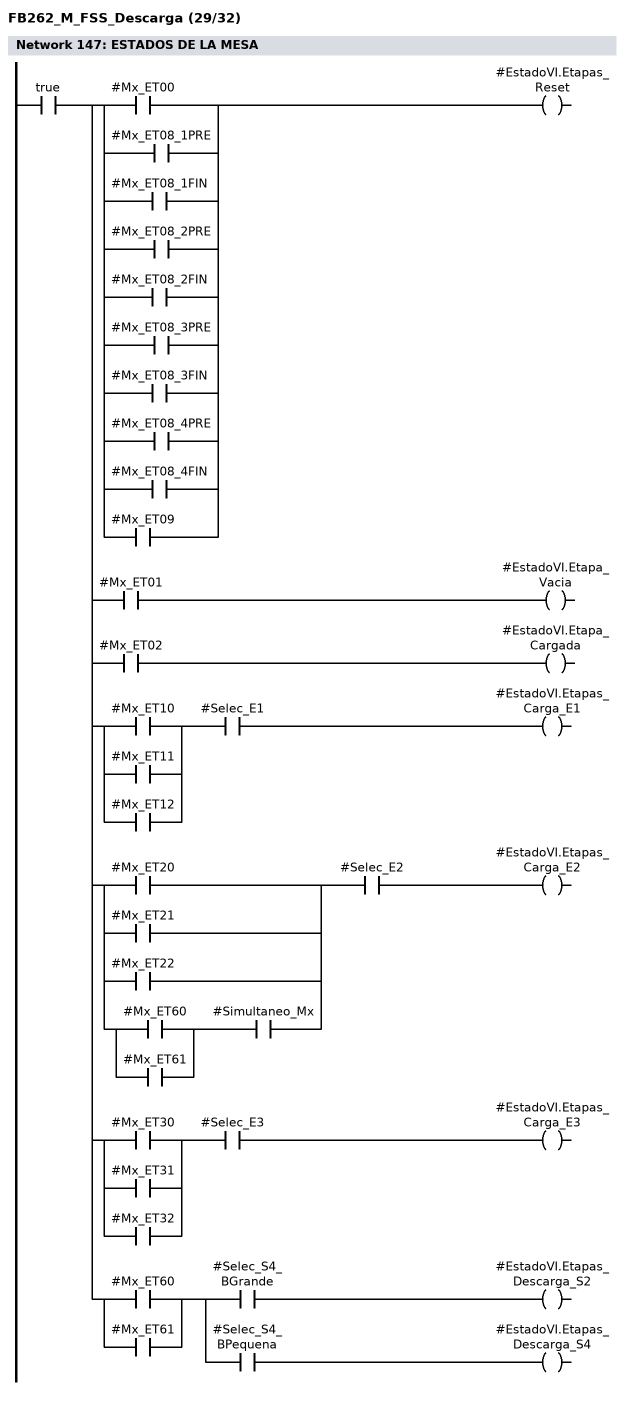
   RUNG wire#powerrail
      Contact( true )
      wire#w1
      Contact( #Mx_ET00 )
      wire#w2
      Coil( #EstadoVI.Etapas_Reset )
   END_RUNG
   RUNG wire#w1
      Contact( #Mx_ET08_1PRE )
   END_RUNG wire#w2
   RUNG wire#w1
      Contact( #Mx_ET08_1FIN )
   END_RUNG wire#w2
   RUNG wire#w1
      Contact( #Mx_ET08_2PRE )
   END_RUNG wire#w2
   RUNG wire#w1
      Contact( #Mx_ET08_2FIN )
   END_RUNG wire#w2
   RUNG wire#w1
      Contact( #Mx_ET08_3PRE )
   END_RUNG wire#w2
   RUNG wire#w1
      Contact( #Mx_ET08_3FIN )
   END_RUNG wire#w2
   RUNG wire#w1
      Contact( #Mx_ET08_4PRE )
   END_RUNG wire#w2
   RUNG wire#w1
      Contact( #Mx_ET08_4FIN )
   END_RUNG wire#w2
   RUNG wire#w1
      Contact( #Mx_ET09 )
   END_RUNG wire#w2
   RUNG wire#w1
      Contact( #Mx_ET01 )
      Coil( #EstadoVI.Etapa_Vacia )
   END_RUNG
   RUNG wire#w1
      Contact( #Mx_ET02 )
      Coil( #EstadoVI.Etapa_Cargada )
   END_RUNG
   RUNG wire#w1
      Contact( #Mx_ET10 )
      wire#w3
      Contact( #Selec_E1 )
      Coil( #EstadoVI.Etapas_Carga_E1 )
   END_RUNG
   RUNG wire#w1
      Contact( #Mx_ET11 )
   END_RUNG wire#w3
   RUNG wire#w1
      Contact( #Mx_ET12 )
   END_RUNG wire#w3
   RUNG wire#w1
      Contact( #Mx_ET20 )
      wire#w4
      Contact( #Selec_E2 )
      Coil( #EstadoVI.Etapas_Carga_E2 )
   END_RUNG
   RUNG wire#w1
      Contact( #Mx_ET21 )
   END_RUNG wire#w4
   RUNG wire#w1
      Contact( #Mx_ET22 )
   END_RUNG wire#w4
   RUNG wire#w1
      Contact( #Mx_ET60 )
      wire#w5
      Contact( #Simultaneo_Mx )
   END_RUNG wire#w4
   RUNG wire#w1
      Contact( #Mx_ET61 )
   END_RUNG wire#w5
   RUNG wire#w1
      Contact( #Mx_ET30 )
      wire#w6
      Contact( #Selec_E3 )
      Coil( #EstadoVI.Etapas_Carga_E3 )
   END_RUNG
   RUNG wire#w1
      Contact( #Mx_ET31 )
   END_RUNG wire#w6
   RUNG wire#w1
      Contact( #Mx_ET32 )
   END_RUNG wire#w6
   RUNG wire#w1
      Contact( #Mx_ET60 )
      wire#w7
      Contact( #Selec_S4_BGrande )
      Coil( #EstadoVI.Etapas_Descarga_S2 )
   END_RUNG
   RUNG wire#w1
      Contact( #Mx_ET61 )
   END_RUNG wire#w7
   RUNG wire#w7
      Contact( #Selec_S4_BPequena )
      Coil( #EstadoVI.Etapas_Descarga_S4 )
   END_RUNG
   // the same network as SCL:
   #EstadoVI.Etapas_Reset := true AND (#Mx_ET00 OR #Mx_ET08_1PRE OR #Mx_ET08_1FIN OR #Mx_ET08_2PRE OR #Mx_ET08_2FIN OR #Mx_ET08_3PRE OR #Mx_ET08_3FIN OR #Mx_ET08_4PRE OR #Mx_ET08_4FIN OR #Mx_ET09);
   #EstadoVI.Etapa_Vacia := true AND #Mx_ET01;
   #EstadoVI.Etapa_Cargada := true AND #Mx_ET02;
   #EstadoVI.Etapas_Carga_E1 := true AND (#Mx_ET10 OR #Mx_ET11 OR #Mx_ET12) AND #Selec_E1;
   #EstadoVI.Etapas_Carga_E2 := true AND (#Mx_ET20 OR #Mx_ET21 OR #Mx_ET22 OR ((#Mx_ET60 OR #Mx_ET61) AND #Simultaneo_Mx)) AND #Selec_E2;
   #EstadoVI.Etapas_Carga_E3 := true AND (#Mx_ET30 OR #Mx_ET31 OR #Mx_ET32) AND #Selec_E3;
   #_w1 := true AND (#Mx_ET60 OR #Mx_ET61);
   #EstadoVI.Etapas_Descarga_S2 := #_w1 AND #Selec_S4_BGrande;
   #EstadoVI.Etapas_Descarga_S4 := #_w1 AND #Selec_S4_BPequena;
END_REGION

REGION Network 148: ENTRADAS DE LA MESA
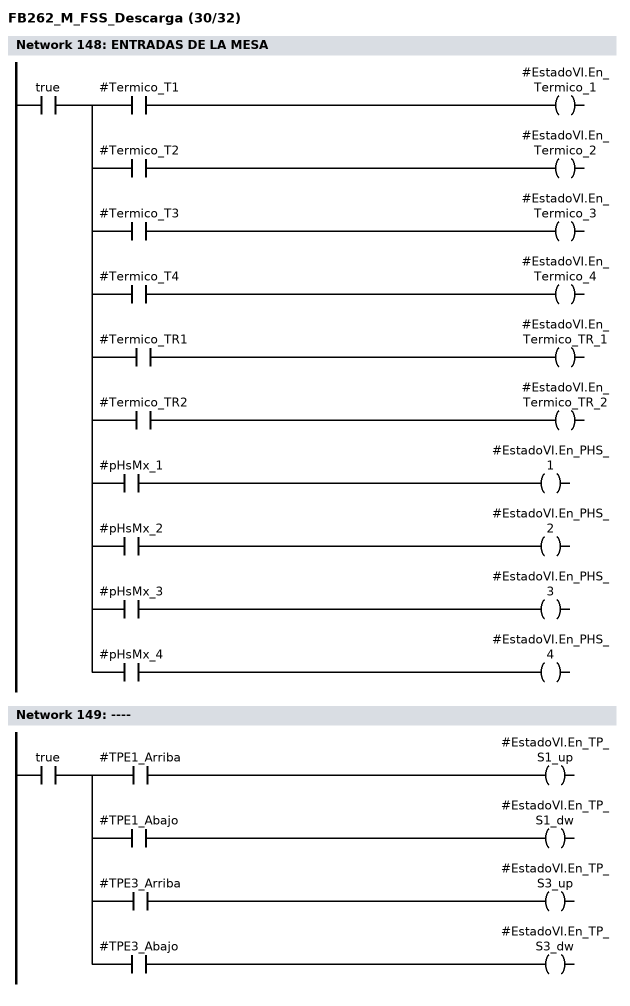
   RUNG wire#powerrail
      Contact( true )
      wire#w1
      Contact( #Termico_T1 )
      Coil( #EstadoVI.En_Termico_1 )
   END_RUNG
   RUNG wire#w1
      Contact( #Termico_T2 )
      Coil( #EstadoVI.En_Termico_2 )
   END_RUNG
   RUNG wire#w1
      Contact( #Termico_T3 )
      Coil( #EstadoVI.En_Termico_3 )
   END_RUNG
   RUNG wire#w1
      Contact( #Termico_T4 )
      Coil( #EstadoVI.En_Termico_4 )
   END_RUNG
   RUNG wire#w1
      Contact( #Termico_TR1 )
      Coil( #EstadoVI.En_Termico_TR_1 )
   END_RUNG
   RUNG wire#w1
      Contact( #Termico_TR2 )
      Coil( #EstadoVI.En_Termico_TR_2 )
   END_RUNG
   RUNG wire#w1
      Contact( #pHsMx_1 )
      Coil( #EstadoVI.En_PHS_1 )
   END_RUNG
   RUNG wire#w1
      Contact( #pHsMx_2 )
      Coil( #EstadoVI.En_PHS_2 )
   END_RUNG
   RUNG wire#w1
      Contact( #pHsMx_3 )
      Coil( #EstadoVI.En_PHS_3 )
   END_RUNG
   RUNG wire#w1
      Contact( #pHsMx_4 )
      Coil( #EstadoVI.En_PHS_4 )
   END_RUNG
   // the same network as SCL:
   #EstadoVI.En_Termico_1 := true AND #Termico_T1;
   #EstadoVI.En_Termico_2 := true AND #Termico_T2;
   #EstadoVI.En_Termico_3 := true AND #Termico_T3;
   #EstadoVI.En_Termico_4 := true AND #Termico_T4;
   #EstadoVI.En_Termico_TR_1 := true AND #Termico_TR1;
   #EstadoVI.En_Termico_TR_2 := true AND #Termico_TR2;
   #EstadoVI.En_PHS_1 := true AND #pHsMx_1;
   #EstadoVI.En_PHS_2 := true AND #pHsMx_2;
   #EstadoVI.En_PHS_3 := true AND #pHsMx_3;
   #EstadoVI.En_PHS_4 := true AND #pHsMx_4;
END_REGION

REGION Network 149: ----
   RUNG wire#powerrail
      Contact( true )
      wire#w1
      Contact( #TPE1_Arriba )
      Coil( #EstadoVI.En_TP_S1_up )
   END_RUNG
   RUNG wire#w1
      Contact( #TPE1_Abajo )
      Coil( #EstadoVI.En_TP_S1_dw )
   END_RUNG
   RUNG wire#w1
      Contact( #TPE3_Arriba )
      Coil( #EstadoVI.En_TP_S3_up )
   END_RUNG
   RUNG wire#w1
      Contact( #TPE3_Abajo )
      Coil( #EstadoVI.En_TP_S3_dw )
   END_RUNG
   // the same network as SCL:
   #EstadoVI.En_TP_S1_up := true AND #TPE1_Arriba;
   #EstadoVI.En_TP_S1_dw := true AND #TPE1_Abajo;
   #EstadoVI.En_TP_S3_up := true AND #TPE3_Arriba;
   #EstadoVI.En_TP_S3_dw := true AND #TPE3_Abajo;
END_REGION

REGION Network 150: SALIDAS de la Mesa
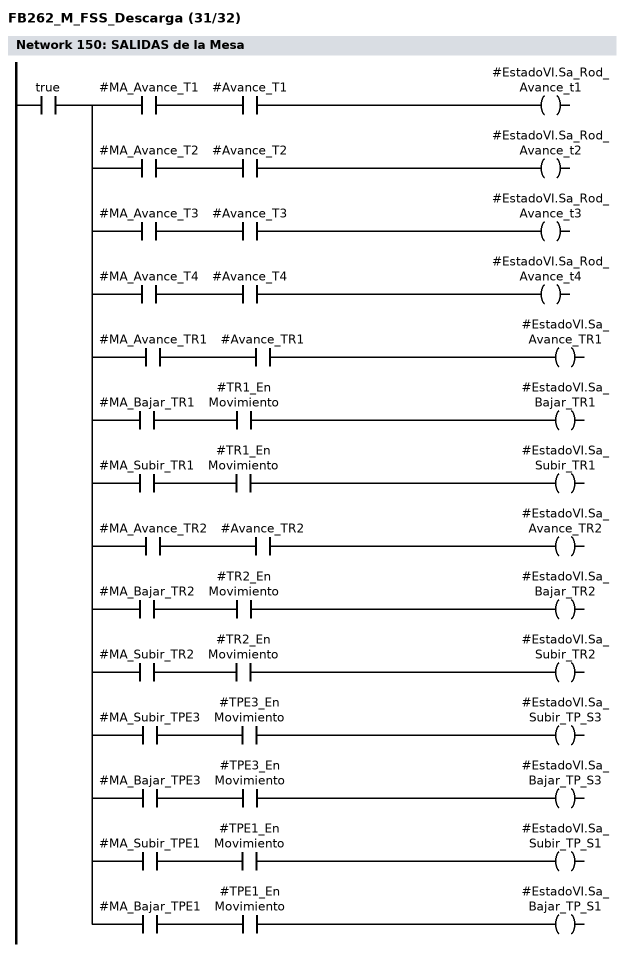
   RUNG wire#powerrail
      Contact( true )
      wire#w1
      Contact( #MA_Avance_T1 )
      Contact( #Avance_T1 )
      Coil( #EstadoVI.Sa_Rod_Avance_t1 )
   END_RUNG
   RUNG wire#w1
      Contact( #MA_Avance_T2 )
      Contact( #Avance_T2 )
      Coil( #EstadoVI.Sa_Rod_Avance_t2 )
   END_RUNG
   RUNG wire#w1
      Contact( #MA_Avance_T3 )
      Contact( #Avance_T3 )
      Coil( #EstadoVI.Sa_Rod_Avance_t3 )
   END_RUNG
   RUNG wire#w1
      Contact( #MA_Avance_T4 )
      Contact( #Avance_T4 )
      Coil( #EstadoVI.Sa_Rod_Avance_t4 )
   END_RUNG
   RUNG wire#w1
      Contact( #MA_Avance_TR1 )
      Contact( #Avance_TR1 )
      Coil( #EstadoVI.Sa_Avance_TR1 )
   END_RUNG
   RUNG wire#w1
      Contact( #MA_Bajar_TR1 )
      Contact( #TR1_EnMovimiento )
      Coil( #EstadoVI.Sa_Bajar_TR1 )
   END_RUNG
   RUNG wire#w1
      Contact( #MA_Subir_TR1 )
      Contact( #TR1_EnMovimiento )
      Coil( #EstadoVI.Sa_Subir_TR1 )
   END_RUNG
   RUNG wire#w1
      Contact( #MA_Avance_TR2 )
      Contact( #Avance_TR2 )
      Coil( #EstadoVI.Sa_Avance_TR2 )
   END_RUNG
   RUNG wire#w1
      Contact( #MA_Bajar_TR2 )
      Contact( #TR2_EnMovimiento )
      Coil( #EstadoVI.Sa_Bajar_TR2 )
   END_RUNG
   RUNG wire#w1
      Contact( #MA_Subir_TR2 )
      Contact( #TR2_EnMovimiento )
      Coil( #EstadoVI.Sa_Subir_TR2 )
   END_RUNG
   RUNG wire#w1
      Contact( #MA_Subir_TPE3 )
      Contact( #TPE3_EnMovimiento )
      Coil( #EstadoVI.Sa_Subir_TP_S3 )
   END_RUNG
   RUNG wire#w1
      Contact( #MA_Bajar_TPE3 )
      Contact( #TPE3_EnMovimiento )
      Coil( #EstadoVI.Sa_Bajar_TP_S3 )
   END_RUNG
   RUNG wire#w1
      Contact( #MA_Subir_TPE1 )
      Contact( #TPE1_EnMovimiento )
      Coil( #EstadoVI.Sa_Subir_TP_S1 )
   END_RUNG
   RUNG wire#w1
      Contact( #MA_Bajar_TPE1 )
      Contact( #TPE1_EnMovimiento )
      Coil( #EstadoVI.Sa_Bajar_TP_S1 )
   END_RUNG
   // the same network as SCL:
   #EstadoVI.Sa_Rod_Avance_t1 := true AND #MA_Avance_T1 AND #Avance_T1;
   #EstadoVI.Sa_Rod_Avance_t2 := true AND #MA_Avance_T2 AND #Avance_T2;
   #EstadoVI.Sa_Rod_Avance_t3 := true AND #MA_Avance_T3 AND #Avance_T3;
   #EstadoVI.Sa_Rod_Avance_t4 := true AND #MA_Avance_T4 AND #Avance_T4;
   #EstadoVI.Sa_Avance_TR1 := true AND #MA_Avance_TR1 AND #Avance_TR1;
   #EstadoVI.Sa_Bajar_TR1 := true AND #MA_Bajar_TR1 AND #TR1_EnMovimiento;
   #EstadoVI.Sa_Subir_TR1 := true AND #MA_Subir_TR1 AND #TR1_EnMovimiento;
   #EstadoVI.Sa_Avance_TR2 := true AND #MA_Avance_TR2 AND #Avance_TR2;
   #EstadoVI.Sa_Bajar_TR2 := true AND #MA_Bajar_TR2 AND #TR2_EnMovimiento;
   #EstadoVI.Sa_Subir_TR2 := true AND #MA_Subir_TR2 AND #TR2_EnMovimiento;
   #EstadoVI.Sa_Subir_TP_S3 := true AND #MA_Subir_TPE3 AND #TPE3_EnMovimiento;
   #EstadoVI.Sa_Bajar_TP_S3 := true AND #MA_Bajar_TPE3 AND #TPE3_EnMovimiento;
   #EstadoVI.Sa_Subir_TP_S1 := true AND #MA_Subir_TPE1 AND #TPE1_EnMovimiento;
   #EstadoVI.Sa_Bajar_TP_S1 := true AND #MA_Bajar_TPE1 AND #TPE1_EnMovimiento;
END_REGION

REGION Network 151: INTERLOCK PARA HMI
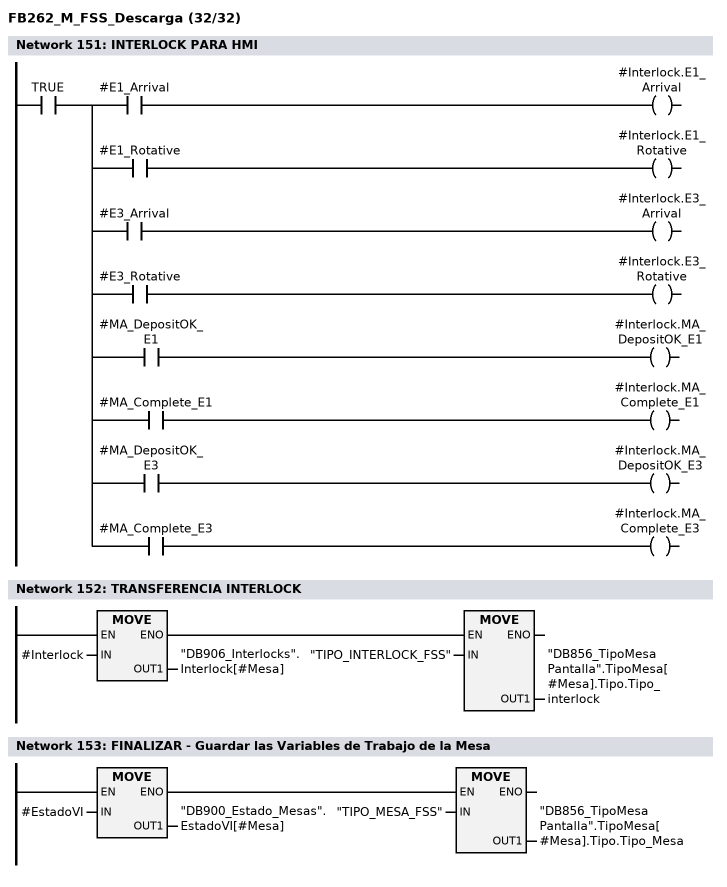
   RUNG wire#powerrail
      Contact( TRUE )
      wire#w1
      Contact( #E1_Arrival )
      Coil( #Interlock.E1_Arrival )
   END_RUNG
   RUNG wire#w1
      Contact( #E1_Rotative )
      Coil( #Interlock.E1_Rotative )
   END_RUNG
   RUNG wire#w1
      Contact( #E3_Arrival )
      Coil( #Interlock.E3_Arrival )
   END_RUNG
   RUNG wire#w1
      Contact( #E3_Rotative )
      Coil( #Interlock.E3_Rotative )
   END_RUNG
   RUNG wire#w1
      Contact( #MA_DepositOK_E1 )
      Coil( #Interlock.MA_DepositOK_E1 )
   END_RUNG
   RUNG wire#w1
      Contact( #MA_Complete_E1 )
      Coil( #Interlock.MA_Complete_E1 )
   END_RUNG
   RUNG wire#w1
      Contact( #MA_DepositOK_E3 )
      Coil( #Interlock.MA_DepositOK_E3 )
   END_RUNG
   RUNG wire#w1
      Contact( #MA_Complete_E3 )
      Coil( #Interlock.MA_Complete_E3 )
   END_RUNG
   // the same network as SCL:
   #Interlock.E1_Arrival := TRUE AND #E1_Arrival;
   #Interlock.E1_Rotative := TRUE AND #E1_Rotative;
   #Interlock.E3_Arrival := TRUE AND #E3_Arrival;
   #Interlock.E3_Rotative := TRUE AND #E3_Rotative;
   #Interlock.MA_DepositOK_E1 := TRUE AND #MA_DepositOK_E1;
   #Interlock.MA_Complete_E1 := TRUE AND #MA_Complete_E1;
   #Interlock.MA_DepositOK_E3 := TRUE AND #MA_DepositOK_E3;
   #Interlock.MA_Complete_E3 := TRUE AND #MA_Complete_E3;
END_REGION

REGION Network 152: TRANSFERENCIA INTERLOCK
   RUNG wire#powerrail
      Move(in := #Interlock, out1 => "DB906_Interlocks".Interlock[#Mesa])
      Move(in := "TIPO_INTERLOCK_FSS", out1 => "DB856_TipoMesaPantalla".TipoMesa[#Mesa].Tipo.Tipo_interlock)
   END_RUNG
   // the same network as SCL:
   "DB906_Interlocks".Interlock[#Mesa] := #Interlock;
   "DB856_TipoMesaPantalla".TipoMesa[#Mesa].Tipo.Tipo_interlock := "TIPO_INTERLOCK_FSS";
END_REGION

REGION Network 153: FINALIZAR - Guardar las Variables de Trabajo de la Mesa
   RUNG wire#powerrail
      Move(in := #EstadoVI, out1 => "DB900_Estado_Mesas".EstadoVI[#Mesa])
      Move(in := "TIPO_MESA_FSS", out1 => "DB856_TipoMesaPantalla".TipoMesa[#Mesa].Tipo.Tipo_Mesa)
   END_RUNG
   // the same network as SCL:
   "DB900_Estado_Mesas".EstadoVI[#Mesa] := #EstadoVI;
   "DB856_TipoMesaPantalla".TipoMesa[#Mesa].Tipo.Tipo_Mesa := "TIPO_MESA_FSS";
END_REGION
END_FUNCTION_BLOCK

FUNCTION_BLOCK "FB263_M_FSS_Maquetas"   // FB263, LAD
TITLE = Control del Ramal de Salidas
{ S7_Optimized_Access := 'FALSE' }
AUTHOR : TE_FSS
NAME : 20160509
VERSION : 3.4
// stored: AutoNumber false, SetENOAutomatically false
   VAR_INPUT
      Mesa : UInt;   // Existe Tension en la Mesa
      Error_Tx : Bool;   // Error en el Tx
      EnTension : Bool;   // Mesa de la FB
      Termico_Tx : Bool;   // Proteccion del Tx
      pHsMx_MQ1 : Bool;   // pHs de la Mesa >> En MQ1
      pHsMx_MQ2 : Bool;   // pHs de la Mesa >> En MQ2
      Avance_Tx : Bool;   // Avance del Tx
      TP1_Arriba : Bool;   // TP1 Arriba. Nota Movimiento E1 >> S3
      TP1_Abajo : Bool;   // TP1 Abajo. Nota Movimiento E1 >> S3
      EnMovimiento_TP1 : Bool;   // En movimiento el TP1
      MQ1_Arriba : Bool;   // MQ1 Arriba >> 1º UT de la Mesa
      MQ1_Abajo : Bool;   // MQ1 Abajo >> 1º UT de la Mesa
      EnMovimiento_MQ1 : Bool;   // MQ1 EnMovimiento >> 1º UT de la Mesa
      MQ2_Arriba : Bool;   // MQ2 Arriba >> 2º UT de la Mesa
      MQ2_Abajo : Bool;   // MQ2 Abajo >> 2º UT de la Mesa
      EnMovimiento_MQ2 : Bool;   // MQ2 EnMovimiento >> 2º UT de la Mesa
      MAnt_DescargaAct : Bool;   // E1 >> Mesa Anterior DescargaAct
      AVTF_MAnt_Mx_MQ1 : Bool;   // E1 >> Mesa Anterior AVTF
      AVTF_MAnt_Mx_MQ1_2 : Bool;   // E1 >> Mesa Anterior AVTF
      P_Mens_MAnt_Mx : Bool;   // E1 >> Mesa Anterior P_Mens
      PTF_Mx_MSig : Bool;   // S3 >> Mesa Siguiente PTF
      FTF_Mx_MSig : Bool;   // S3 >> Mesa Siguiente FTF
      MSig_CargaAct : Bool;
      Mx_ControlUTs : Bool;   // Config >> Control de UT en Mesa
      F_EnvMens_Mx : Bool;   // Fin de Envio de Mensaje
      OrdSal_MQ1 : Bool;   // Orden de Salida de MQ1
      OrdSal_MQ2 : Bool;   // Orden de Salida de MQ2
      OrdSal_MQ1_2 : Bool;   // Orden de Salida de MQ1 y MQ2
      V_CNT_pHsMx : Int := 400;   // Valor de Presencia
      V_CNT_pHsMx_FTF : Int := 200;   // Valor para activar FTF. Nota: < = V_CNT_pHsMx.
      V_CNTSeg_pHsMx : Int := 2000;   // Valor de Seguriadad para Presencia
      V_CNT_ApHsMx : Int := 200;   // Valor de Ausencia
      V_CNTSeg_ApHsMx : Int := 2000;   // Valor de Seguriadad para Ausencia
      V_CNT_Simultaneo : Int := 2000;   // Valor de Simultaneo
      V_EstabilidadCarga : Time := T#200MS;   // Valor de Estabilidad de la Carga
      V_RetardoBajarMAQ : Time := T#200MS;   // Valor de Retardo de Bajada de las Maquetas
      V_TOut_Tx_Mx : Int := 7000;   // TimeOut de Entrada por E1
      V_TOut_TP : Int := 3000;   // TimeOut de Tope
      V_TOut_MQ : Int := 3000;   // TimeOut de Maqueta
      V_CNT_PerdidapHs : Int := 1000;   // CNT de Perdida de pHs
   END_VAR
   VAR_OUTPUT
      P_EnvMens_PMx : Bool;   // Permiso de Enviar Mensaje de Presencia
      P_RecepOK_Mx : Bool;   // Recepcion OK
      PTF_MAnt_Mx : Bool;   // E1 >> Mesa Anterior PTF
      FTF_MAnt_Mx : Bool;   // E1 >> Mesa Anterior FTF
      AVTF_Mx_MSig_MQ1 : Bool;   // S3 >> Mesa Siguiente AVTF
      AVTF_Mx_MSig_MQ2 : Bool;   // S3 >> Mesa Siguiente AVTF
      AVTF_Mx_MSig_MQ1_2 : Bool;   // S3 >> Mesa Siguiente AVTF
      P_Mens_Mx_MSig : Bool;   // S3 >> Mesa Siguiente P_Mens
   END_VAR
   VAR
      Mx_ET00 : Bool;
      Mx_ET01 : Bool;
      Mx_ET02 : Bool;
      Mx_ET06 : Bool;
      Mx_ET07 : Bool;
      Mx_ET08 : Bool;
      Mx_ET09 : Bool;
      Mx_ET10 : Bool;
      Mx_ET11 : Bool;
      Mx_ET12 : Bool;
      Mx_ET110 : Bool;
      Mx_ET111 : Bool;
      Mx_ET50 : Bool;
      Mx_ET51 : Bool;
      Mx_ET150 : Bool;
      Mx_ET151 : Bool;
      SinUTs_EnMesa : Bool;   // Control UTs En Mesa >> Sin UTs
      DoblePeque_EnMesa : Bool;   // Control UTs En Mesa >> Caja Doble Pequeña
      UT01Peque_EnMesa : Bool;   // Control UTs En Mesa >> UT01 Caja Pequeña
      UT02Peque_EnMesa : Bool;   // Control UTs En Mesa >> UT02 Caja Pequeña
      OrdSalida_OK : Bool;   // Control UTs En Mesa >> Validar Orden de Salida
      Selec_Entrada : Bool;   // Select Entrada de Mesa Anterior
      Selec_Salida_MQ1 : Bool;   // Select Salida de MQ1
      Selec_Salida_MQ2 : Bool;   // Select Salida de MQ2
      Selec_Salida_MQ1_2 : Bool;   // Select Salida de MQ1 y MQ2
      AVTF_MAnt_Mx : Bool;   // Interna >> Aviso de Entrada
      AVTF_Mx_MSig : Bool;   // Interna >> Aviso de Salida
      SaliendoCarga : Bool;   // Interna >> Realizando Salida de la Mesa
      PosMQ_OK : Bool;   // Interna >> Pos. de Maquetas OK
      Simultaneo_Mx : Bool;   // Activo Simultaneo E1
      ProtocoloIniciado : Bool;   // Iniciado el Envio del Mensaje de Presencia
      CNT_pHsMx_FTF_OK : Bool;   // Enviar ya FTF
      STAT_EnvMens_PMx : Bool;   // Interna >> Envio del Mensaje de Presencia
      STAT_FTF_MAnt_Mx : Bool;   // Interna >> FTF de MAnt >> Mx
      MA_Subir_MQ1 : Bool;
      MA_Bajar_MQ1 : Bool;
      MA_Subir_MQ2 : Bool;
      MA_Bajar_MQ2 : Bool;
      TMP_EstabilidadCarga { S7_SetPoint := 'True'} : TON_TIME;   // TMP de Estabilidad de la Carga En la Entrada
      TMP_RetardoBajada_MQ1 { S7_SetPoint := 'True'} : TON_TIME;   // TMP de Retardo de Bajada de la MQ1
      TMP_RetardoBajada_MQ2 { S7_SetPoint := 'True'} : TON_TIME;   // TMP de Retardo de Bajada de la MQ2
      CNT_pHsMx { S7_SetPoint := 'True'} : "FB910_CNT_UHS";   // CNT de la Presencia
      CNTSeg_pHsMx { S7_SetPoint := 'True'} : "FB910_CNT_UHS";   // CNT de Seguridad de la Presencia
      CNT_ApHsMx { S7_SetPoint := 'True'} : "FB910_CNT_UHS";   // CNT de la Ausencia
      CNTSeg_ApHsMx { S7_SetPoint := 'True'} : "FB910_CNT_UHS";   // CNT de Seguridad de la Ausencia
      CNT_Simultaneo { S7_SetPoint := 'True'} : "FB910_CNT_UHS";   // CNT de Simultaneo
      TMP_EnTension { S7_SetPoint := 'True'} : "FB910_CNT_UHS";
      TOut_Av_Mx { S7_SetPoint := 'True'} : "FB910_CNT_UHS";   // Time Out de Entrada de E1
      TOut_Subir_TP { S7_SetPoint := 'True'} : "FB910_CNT_UHS";   // Time Out de Subida del TP
      TOut_Bajar_TP { S7_SetPoint := 'True'} : "FB910_CNT_UHS";   // Time Out de Bajada del TP
      TOut_Subir_MQ { S7_SetPoint := 'True'} : "FB910_CNT_UHS";
      TOut_Bajar_MQ { S7_SetPoint := 'True'} : "FB910_CNT_UHS";
      CNT_PerdidapHs { S7_SetPoint := 'True'} : "FB910_CNT_UHS";   // CNT de Perdida de pHs
   END_VAR
   VAR_TEMP
      EstadoZona : "EstadoZona";   // Estado de Zona de la Mesa
      EstadoVI : "EstadosMesa";   // Estado del Vehiculo Inteliguente de la Mesa
      ConfigFB : "UDT_ConfigFB";   // Configuracion de la FB de la Mesa
      V_Protrusion : Int;
      Aux_ET00 : Bool;
   END_VAR
   VAR_TEMP   // added for the SCL form of the ladder/FBD networks
      _w1 : Bool;
   END_VAR
BEGIN

REGION Network 1: INICIALIZAR - Recoger las Variables de Estado de la Mesa
   // Se recoge - Estado_CBx
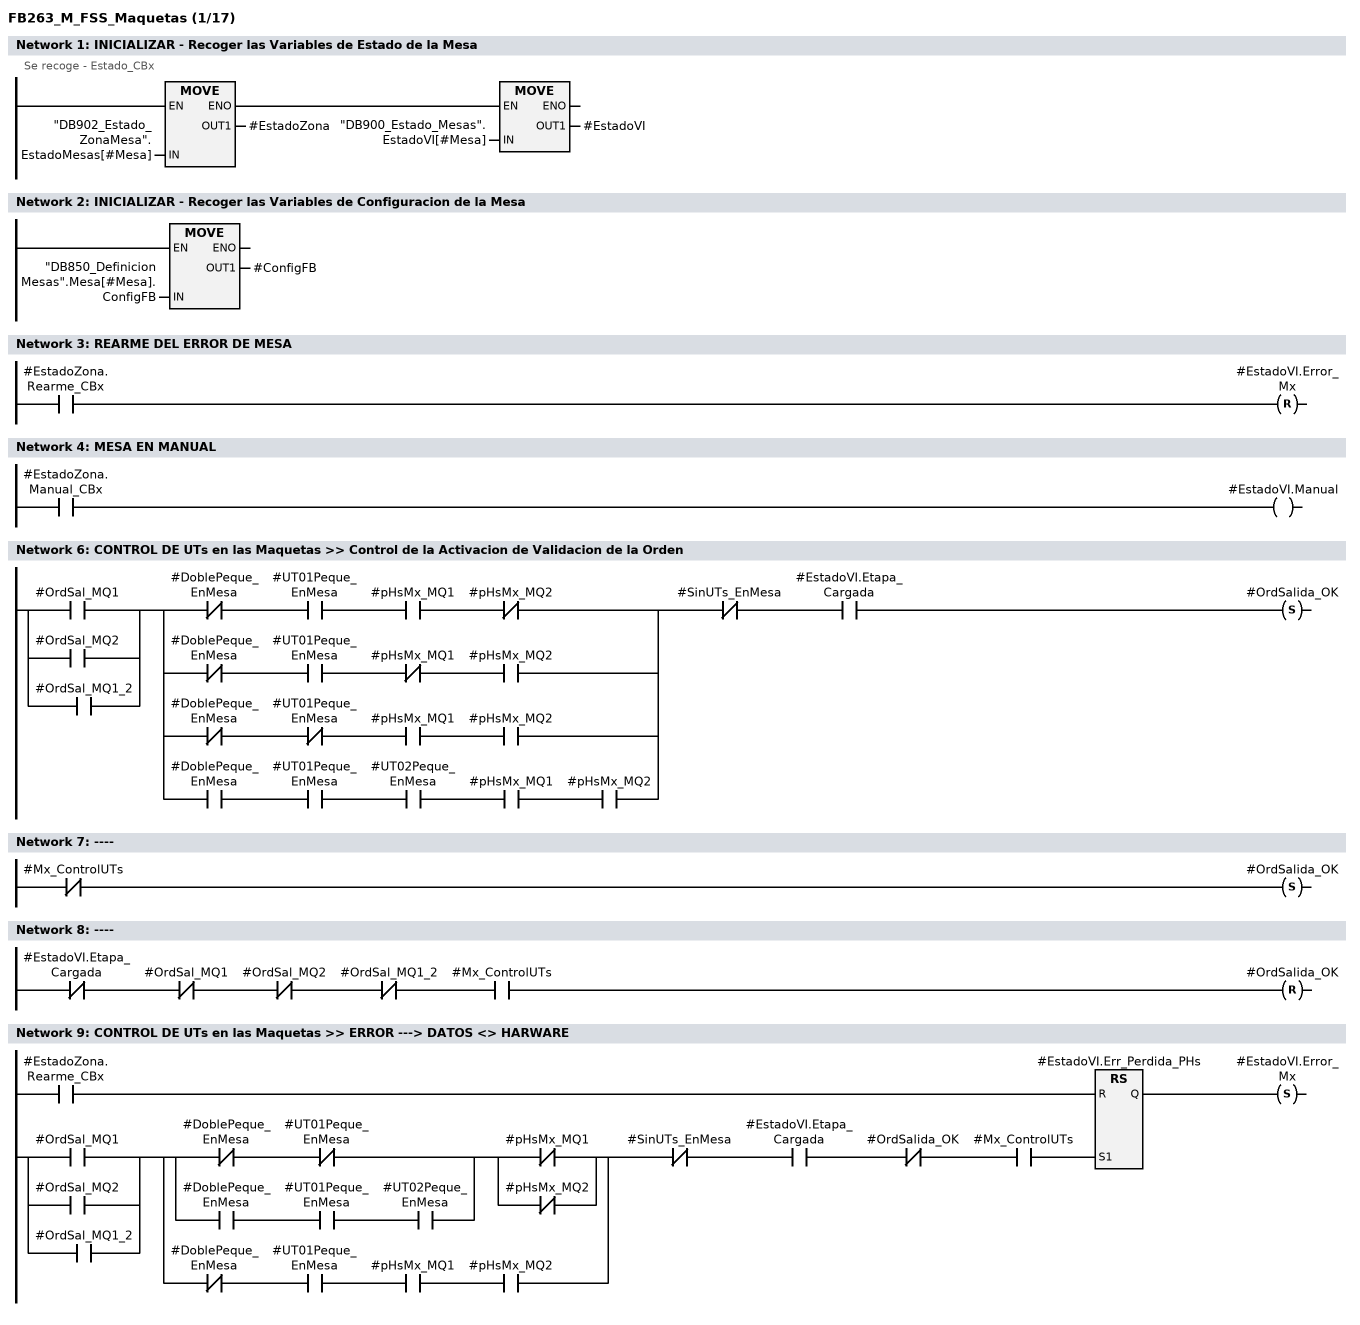
   RUNG wire#powerrail
      Move(in := "DB902_Estado_ZonaMesa".EstadoMesas[#Mesa], out1 => #EstadoZona)
      Move(in := "DB900_Estado_Mesas".EstadoVI[#Mesa], out1 => #EstadoVI)
   END_RUNG
   // the same network as SCL:
   #EstadoZona := "DB902_Estado_ZonaMesa".EstadoMesas[#Mesa];
   #EstadoVI := "DB900_Estado_Mesas".EstadoVI[#Mesa];
END_REGION

REGION Network 2: INICIALIZAR - Recoger las Variables de Configuracion de la Mesa
   RUNG wire#powerrail
      Move(in := "DB850_DefinicionMesas".Mesa[#Mesa].ConfigFB, out1 => #ConfigFB)
   END_RUNG
   // the same network as SCL:
   #ConfigFB := "DB850_DefinicionMesas".Mesa[#Mesa].ConfigFB;
END_REGION

REGION Network 3: REARME DEL ERROR DE MESA
   RUNG wire#powerrail
      Contact( #EstadoZona.Rearme_CBx )
      R_Coil( #EstadoVI.Error_Mx )
   END_RUNG
   // the same network as SCL:
   IF #EstadoZona.Rearme_CBx THEN #EstadoVI.Error_Mx := FALSE; END_IF;
END_REGION

REGION Network 4: MESA EN MANUAL
   RUNG wire#powerrail
      Contact( #EstadoZona.Manual_CBx )
      Coil( #EstadoVI.Manual )
   END_RUNG
   // the same network as SCL:
   #EstadoVI.Manual := #EstadoZona.Manual_CBx;
END_REGION

NETWORK
TITLE = CONTROL DE UTs en las Maquetas >> Recoger datos de las UTs de la Mesa
//////////////////////////////////////////////////////////////////////////////////
/// Recoger datos de las UTs de la Mesa

      CALL  "FC870_MesaSinUT"
      ( Mesa  := #Mesa,
        SinUT := #SinUTs_EnMesa
      );

      CALL  "FC777_TipoCajaPlastico_EnMesa"
      ( Mesa           := #Mesa,
        DosCajas       := #DoblePeque_EnMesa,
        CajaPeque_UT01 := #UT01Peque_EnMesa,
        CajaPeque_UT02 := #UT02Peque_EnMesa
      );



REGION Network 6: CONTROL DE UTs en las Maquetas >> Control de la Activacion de Validacion de la Orden
   RUNG wire#powerrail
      Contact( #OrdSal_MQ1 )
      wire#w1
      I_Contact( #DoblePeque_EnMesa )
      Contact( #UT01Peque_EnMesa )
      Contact( #pHsMx_MQ1 )
      I_Contact( #pHsMx_MQ2 )
      wire#w2
      I_Contact( #SinUTs_EnMesa )
      Contact( #EstadoVI.Etapa_Cargada )
      S_Coil( #OrdSalida_OK )
   END_RUNG
   RUNG wire#powerrail
      Contact( #OrdSal_MQ2 )
   END_RUNG wire#w1
   RUNG wire#powerrail
      Contact( #OrdSal_MQ1_2 )
   END_RUNG wire#w1
   RUNG wire#w1
      I_Contact( #DoblePeque_EnMesa )
      Contact( #UT01Peque_EnMesa )
      I_Contact( #pHsMx_MQ1 )
      Contact( #pHsMx_MQ2 )
   END_RUNG wire#w2
   RUNG wire#w1
      I_Contact( #DoblePeque_EnMesa )
      I_Contact( #UT01Peque_EnMesa )
      Contact( #pHsMx_MQ1 )
      Contact( #pHsMx_MQ2 )
   END_RUNG wire#w2
   RUNG wire#w1
      Contact( #DoblePeque_EnMesa )
      Contact( #UT01Peque_EnMesa )
      Contact( #UT02Peque_EnMesa )
      Contact( #pHsMx_MQ1 )
      Contact( #pHsMx_MQ2 )
   END_RUNG wire#w2
   // the same network as SCL:
   IF (#OrdSal_MQ1 OR #OrdSal_MQ2 OR #OrdSal_MQ1_2) AND ((NOT #DoblePeque_EnMesa AND #UT01Peque_EnMesa AND #pHsMx_MQ1 AND NOT #pHsMx_MQ2) OR (NOT #DoblePeque_EnMesa AND #UT01Peque_EnMesa AND NOT #pHsMx_MQ1 AND #pHsMx_MQ2) OR (NOT #DoblePeque_EnMesa AND NOT #UT01Peque_EnMesa AND #pHsMx_MQ1 AND #pHsMx_MQ2) OR (#DoblePeque_EnMesa AND #UT01Peque_EnMesa AND #UT02Peque_EnMesa AND #pHsMx_MQ1 AND #pHsMx_MQ2)) AND NOT #SinUTs_EnMesa AND #EstadoVI.Etapa_Cargada THEN
       #OrdSalida_OK := TRUE;
   END_IF;
END_REGION

REGION Network 7: ----
   RUNG wire#powerrail
      I_Contact( #Mx_ControlUTs )
      S_Coil( #OrdSalida_OK )
   END_RUNG
   // the same network as SCL:
   IF NOT #Mx_ControlUTs THEN #OrdSalida_OK := TRUE; END_IF;
END_REGION

REGION Network 8: ----
   RUNG wire#powerrail
      I_Contact( #EstadoVI.Etapa_Cargada )
      I_Contact( #OrdSal_MQ1 )
      I_Contact( #OrdSal_MQ2 )
      I_Contact( #OrdSal_MQ1_2 )
      Contact( #Mx_ControlUTs )
      R_Coil( #OrdSalida_OK )
   END_RUNG
   // the same network as SCL:
   IF NOT #EstadoVI.Etapa_Cargada AND NOT #OrdSal_MQ1 AND NOT #OrdSal_MQ2 AND NOT #OrdSal_MQ1_2 AND #Mx_ControlUTs THEN
       #OrdSalida_OK := FALSE;
   END_IF;
END_REGION

REGION Network 9: CONTROL DE UTs en las Maquetas >> ERROR ---> DATOS <> HARWARE
   RUNG wire#powerrail
      Contact( #EstadoZona.Rearme_CBx )
      S_RS(operand := #EstadoVI.Err_Perdida_PHs, s1 := wire#w4)
      S_Coil( #EstadoVI.Error_Mx )
   END_RUNG
   RUNG wire#powerrail
      Contact( #OrdSal_MQ1 )
      wire#w1
      I_Contact( #DoblePeque_EnMesa )
      I_Contact( #UT01Peque_EnMesa )
      wire#w2
      I_Contact( #pHsMx_MQ1 )
      wire#w3
      I_Contact( #SinUTs_EnMesa )
      Contact( #EstadoVI.Etapa_Cargada )
      I_Contact( #OrdSalida_OK )
      Contact( #Mx_ControlUTs )
   END_RUNG wire#w4
   RUNG wire#powerrail
      Contact( #OrdSal_MQ2 )
   END_RUNG wire#w1
   RUNG wire#powerrail
      Contact( #OrdSal_MQ1_2 )
   END_RUNG wire#w1
   RUNG wire#w1
      Contact( #DoblePeque_EnMesa )
      Contact( #UT01Peque_EnMesa )
      Contact( #UT02Peque_EnMesa )
   END_RUNG wire#w2
   RUNG wire#w2
      I_Contact( #pHsMx_MQ2 )
   END_RUNG wire#w3
   RUNG wire#w1
      I_Contact( #DoblePeque_EnMesa )
      Contact( #UT01Peque_EnMesa )
      Contact( #pHsMx_MQ1 )
      Contact( #pHsMx_MQ2 )
   END_RUNG wire#w3
   // the same network as SCL:
   IF #EstadoZona.Rearme_CBx THEN
       #EstadoVI.Err_Perdida_PHs := FALSE;   // RS flip-flop
   END_IF;
   IF (#OrdSal_MQ1 OR #OrdSal_MQ2 OR #OrdSal_MQ1_2) AND ((((NOT #DoblePeque_EnMesa AND NOT #UT01Peque_EnMesa) OR (#DoblePeque_EnMesa AND #UT01Peque_EnMesa AND #UT02Peque_EnMesa)) AND (NOT #pHsMx_MQ1 OR NOT #pHsMx_MQ2)) OR (NOT #DoblePeque_EnMesa AND #UT01Peque_EnMesa AND #pHsMx_MQ1 AND #pHsMx_MQ2)) AND NOT #SinUTs_EnMesa AND #EstadoVI.Etapa_Cargada AND NOT #OrdSalida_OK AND #Mx_ControlUTs THEN
       #EstadoVI.Err_Perdida_PHs := TRUE;
   END_IF;
   IF #EstadoVI.Err_Perdida_PHs THEN #EstadoVI.Error_Mx := TRUE; END_IF;
END_REGION

REGION Network 10: VARIABLES AUXILIARES - Aviso de Entrada - AVTF_MAnt_Mx
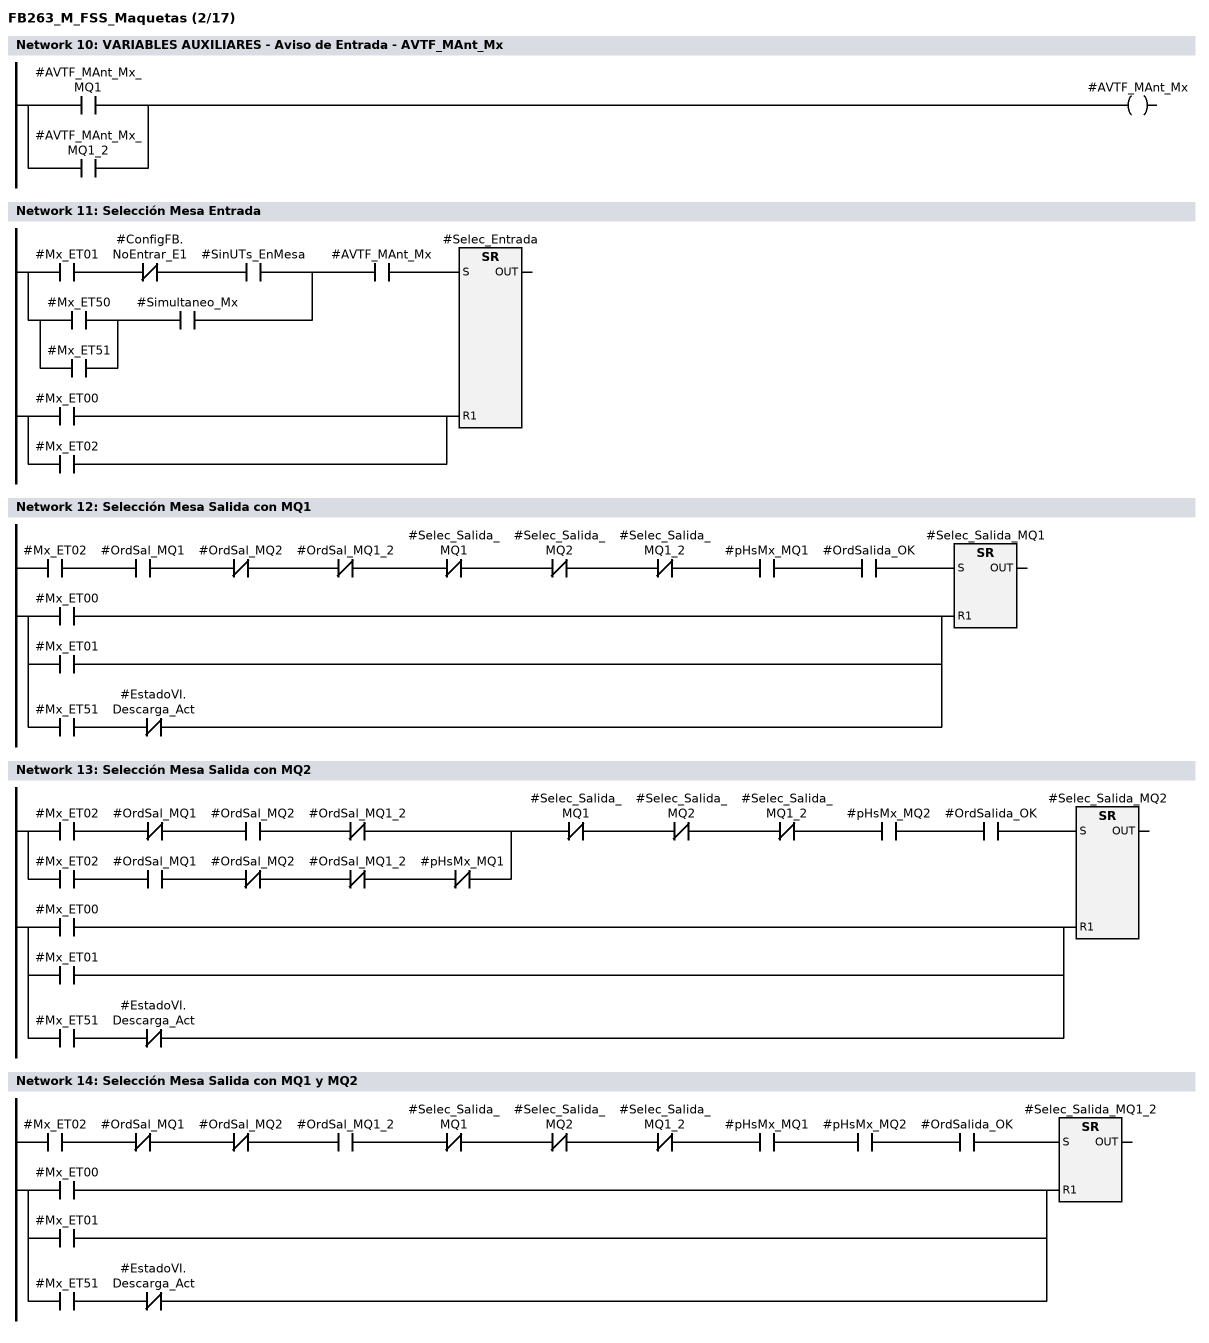
   RUNG wire#powerrail
      Contact( #AVTF_MAnt_Mx_MQ1 )
      wire#w1
      Coil( #AVTF_MAnt_Mx )
   END_RUNG
   RUNG wire#powerrail
      Contact( #AVTF_MAnt_Mx_MQ1_2 )
   END_RUNG wire#w1
   // the same network as SCL:
   #AVTF_MAnt_Mx := #AVTF_MAnt_Mx_MQ1 OR #AVTF_MAnt_Mx_MQ1_2;
END_REGION

REGION Network 11: Selección Mesa Entrada
   RUNG wire#powerrail
      Contact( #Mx_ET01 )
      I_Contact( #ConfigFB.NoEntrar_E1 )
      Contact( #SinUTs_EnMesa )
      wire#w1
      Contact( #AVTF_MAnt_Mx )
      S_SR(operand := #Selec_Entrada, r1 := wire#w3)
   END_RUNG
   RUNG wire#powerrail
      Contact( #Mx_ET50 )
      wire#w2
      Contact( #Simultaneo_Mx )
   END_RUNG wire#w1
   RUNG wire#powerrail
      Contact( #Mx_ET51 )
   END_RUNG wire#w2
   RUNG wire#powerrail
      Contact( #Mx_ET00 )
   END_RUNG wire#w3
   RUNG wire#powerrail
      Contact( #Mx_ET02 )
   END_RUNG wire#w3
   // the same network as SCL:
   IF ((#Mx_ET01 AND NOT #ConfigFB.NoEntrar_E1 AND #SinUTs_EnMesa) OR ((#Mx_ET50 OR #Mx_ET51) AND #Simultaneo_Mx)) AND #AVTF_MAnt_Mx THEN
       #Selec_Entrada := TRUE;   // SR flip-flop
   END_IF;
   IF #Mx_ET00 OR #Mx_ET02 THEN #Selec_Entrada := FALSE; END_IF;
END_REGION

REGION Network 12: Selección Mesa Salida con MQ1
   RUNG wire#powerrail
      Contact( #Mx_ET02 )
      Contact( #OrdSal_MQ1 )
      I_Contact( #OrdSal_MQ2 )
      I_Contact( #OrdSal_MQ1_2 )
      I_Contact( #Selec_Salida_MQ1 )
      I_Contact( #Selec_Salida_MQ2 )
      I_Contact( #Selec_Salida_MQ1_2 )
      Contact( #pHsMx_MQ1 )
      Contact( #OrdSalida_OK )
      S_SR(operand := #Selec_Salida_MQ1, r1 := wire#w1)
   END_RUNG
   RUNG wire#powerrail
      Contact( #Mx_ET00 )
   END_RUNG wire#w1
   RUNG wire#powerrail
      Contact( #Mx_ET01 )
   END_RUNG wire#w1
   RUNG wire#powerrail
      Contact( #Mx_ET51 )
      I_Contact( #EstadoVI.Descarga_Act )
   END_RUNG wire#w1
   // the same network as SCL:
   IF #Mx_ET02 AND #OrdSal_MQ1 AND NOT #OrdSal_MQ2 AND NOT #OrdSal_MQ1_2 AND NOT #Selec_Salida_MQ1 AND NOT #Selec_Salida_MQ2 AND NOT #Selec_Salida_MQ1_2 AND #pHsMx_MQ1 AND #OrdSalida_OK THEN
       #Selec_Salida_MQ1 := TRUE;   // SR flip-flop
   END_IF;
   IF #Mx_ET00 OR #Mx_ET01 OR (#Mx_ET51 AND NOT #EstadoVI.Descarga_Act) THEN
       #Selec_Salida_MQ1 := FALSE;
   END_IF;
END_REGION

REGION Network 13: Selección Mesa Salida con MQ2
   RUNG wire#powerrail
      Contact( #Mx_ET02 )
      I_Contact( #OrdSal_MQ1 )
      Contact( #OrdSal_MQ2 )
      I_Contact( #OrdSal_MQ1_2 )
      wire#w1
      I_Contact( #Selec_Salida_MQ1 )
      I_Contact( #Selec_Salida_MQ2 )
      I_Contact( #Selec_Salida_MQ1_2 )
      Contact( #pHsMx_MQ2 )
      Contact( #OrdSalida_OK )
      S_SR(operand := #Selec_Salida_MQ2, r1 := wire#w2)
   END_RUNG
   RUNG wire#powerrail
      Contact( #Mx_ET02 )
      Contact( #OrdSal_MQ1 )
      I_Contact( #OrdSal_MQ2 )
      I_Contact( #OrdSal_MQ1_2 )
      I_Contact( #pHsMx_MQ1 )
   END_RUNG wire#w1
   RUNG wire#powerrail
      Contact( #Mx_ET00 )
   END_RUNG wire#w2
   RUNG wire#powerrail
      Contact( #Mx_ET01 )
   END_RUNG wire#w2
   RUNG wire#powerrail
      Contact( #Mx_ET51 )
      I_Contact( #EstadoVI.Descarga_Act )
   END_RUNG wire#w2
   // the same network as SCL:
   IF ((#Mx_ET02 AND NOT #OrdSal_MQ1 AND #OrdSal_MQ2 AND NOT #OrdSal_MQ1_2) OR (#Mx_ET02 AND #OrdSal_MQ1 AND NOT #OrdSal_MQ2 AND NOT #OrdSal_MQ1_2 AND NOT #pHsMx_MQ1)) AND NOT #Selec_Salida_MQ1 AND NOT #Selec_Salida_MQ2 AND NOT #Selec_Salida_MQ1_2 AND #pHsMx_MQ2 AND #OrdSalida_OK THEN
       #Selec_Salida_MQ2 := TRUE;   // SR flip-flop
   END_IF;
   IF #Mx_ET00 OR #Mx_ET01 OR (#Mx_ET51 AND NOT #EstadoVI.Descarga_Act) THEN
       #Selec_Salida_MQ2 := FALSE;
   END_IF;
END_REGION

REGION Network 14: Selección Mesa Salida con MQ1 y MQ2
   RUNG wire#powerrail
      Contact( #Mx_ET02 )
      I_Contact( #OrdSal_MQ1 )
      I_Contact( #OrdSal_MQ2 )
      Contact( #OrdSal_MQ1_2 )
      I_Contact( #Selec_Salida_MQ1 )
      I_Contact( #Selec_Salida_MQ2 )
      I_Contact( #Selec_Salida_MQ1_2 )
      Contact( #pHsMx_MQ1 )
      Contact( #pHsMx_MQ2 )
      Contact( #OrdSalida_OK )
      S_SR(operand := #Selec_Salida_MQ1_2, r1 := wire#w1)
   END_RUNG
   RUNG wire#powerrail
      Contact( #Mx_ET00 )
   END_RUNG wire#w1
   RUNG wire#powerrail
      Contact( #Mx_ET01 )
   END_RUNG wire#w1
   RUNG wire#powerrail
      Contact( #Mx_ET51 )
      I_Contact( #EstadoVI.Descarga_Act )
   END_RUNG wire#w1
   // the same network as SCL:
   IF #Mx_ET02 AND NOT #OrdSal_MQ1 AND NOT #OrdSal_MQ2 AND #OrdSal_MQ1_2 AND NOT #Selec_Salida_MQ1 AND NOT #Selec_Salida_MQ2 AND NOT #Selec_Salida_MQ1_2 AND #pHsMx_MQ1 AND #pHsMx_MQ2 AND #OrdSalida_OK THEN
       #Selec_Salida_MQ1_2 := TRUE;   // SR flip-flop
   END_IF;
   IF #Mx_ET00 OR #Mx_ET01 OR (#Mx_ET51 AND NOT #EstadoVI.Descarga_Act) THEN
       #Selec_Salida_MQ1_2 := FALSE;
   END_IF;
END_REGION

REGION Network 15: VARIABLES AUXILIARES - Saliendo Carga de la Mesa
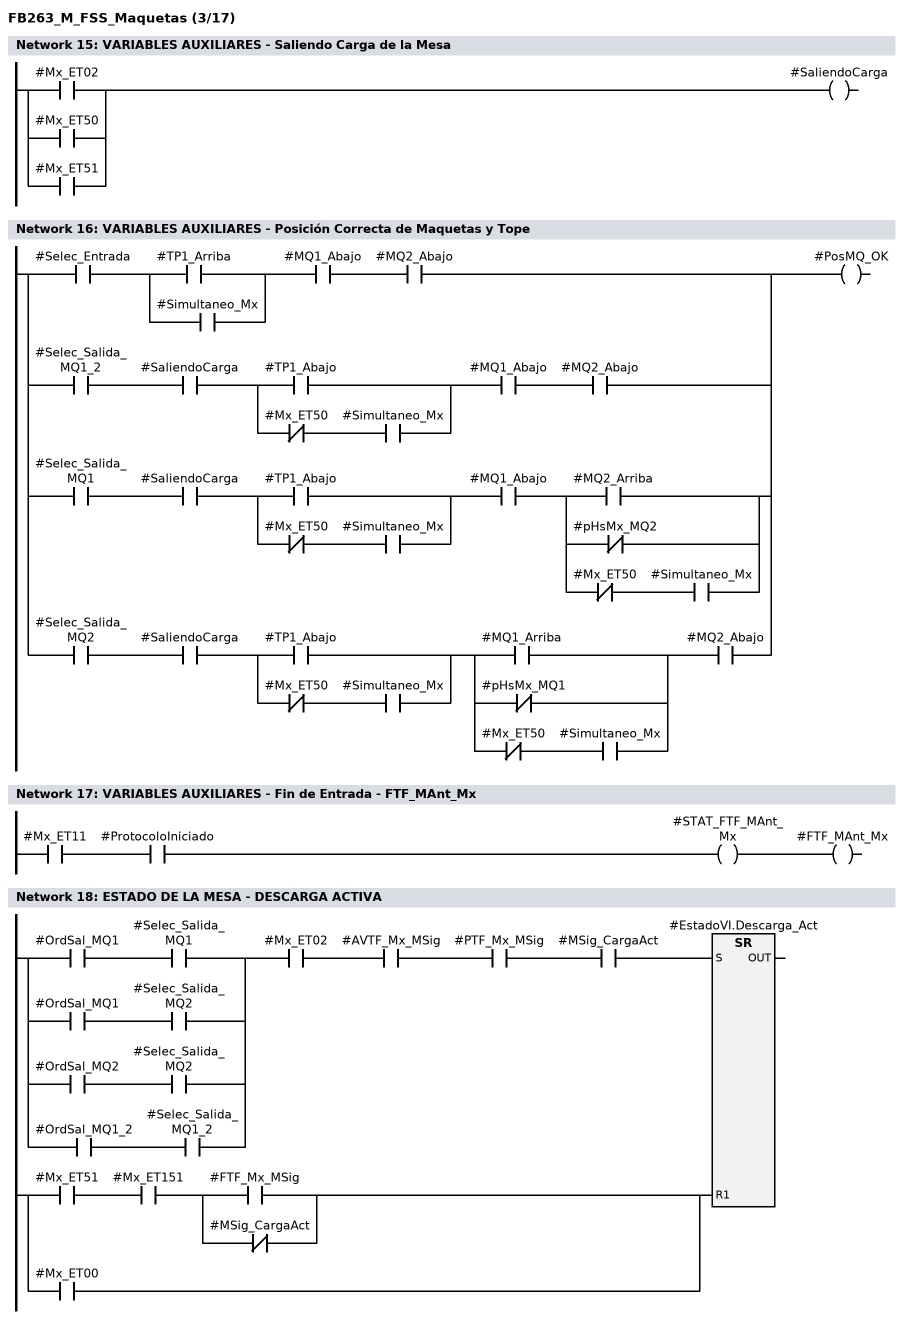
   RUNG wire#powerrail
      Contact( #Mx_ET02 )
      wire#w1
      Coil( #SaliendoCarga )
   END_RUNG
   RUNG wire#powerrail
      Contact( #Mx_ET50 )
   END_RUNG wire#w1
   RUNG wire#powerrail
      Contact( #Mx_ET51 )
   END_RUNG wire#w1
   // the same network as SCL:
   #SaliendoCarga := #Mx_ET02 OR #Mx_ET50 OR #Mx_ET51;
END_REGION

REGION Network 16: VARIABLES AUXILIARES - Posición Correcta de Maquetas y Tope
   RUNG wire#powerrail
      Contact( #Selec_Entrada )
      wire#w1
      Contact( #TP1_Arriba )
      wire#w2
      Contact( #MQ1_Abajo )
      Contact( #MQ2_Abajo )
      wire#w3
      Coil( #PosMQ_OK )
   END_RUNG
   RUNG wire#w1
      Contact( #Simultaneo_Mx )
   END_RUNG wire#w2
   RUNG wire#powerrail
      Contact( #Selec_Salida_MQ1_2 )
      Contact( #SaliendoCarga )
      wire#w4
      Contact( #TP1_Abajo )
      wire#w5
      Contact( #MQ1_Abajo )
      Contact( #MQ2_Abajo )
   END_RUNG wire#w3
   RUNG wire#w4
      I_Contact( #Mx_ET50 )
      Contact( #Simultaneo_Mx )
   END_RUNG wire#w5
   RUNG wire#powerrail
      Contact( #Selec_Salida_MQ1 )
      Contact( #SaliendoCarga )
      wire#w6
      Contact( #TP1_Abajo )
      wire#w7
      Contact( #MQ1_Abajo )
      wire#w8
      Contact( #MQ2_Arriba )
   END_RUNG wire#w3
   RUNG wire#w6
      I_Contact( #Mx_ET50 )
      Contact( #Simultaneo_Mx )
   END_RUNG wire#w7
   RUNG wire#w8
      I_Contact( #pHsMx_MQ2 )
   END_RUNG wire#w3
   RUNG wire#w8
      I_Contact( #Mx_ET50 )
      Contact( #Simultaneo_Mx )
   END_RUNG wire#w3
   RUNG wire#powerrail
      Contact( #Selec_Salida_MQ2 )
      Contact( #SaliendoCarga )
      wire#w9
      Contact( #TP1_Abajo )
      wire#w10
      Contact( #MQ1_Arriba )
      wire#w11
      Contact( #MQ2_Abajo )
   END_RUNG wire#w3
   RUNG wire#w9
      I_Contact( #Mx_ET50 )
      Contact( #Simultaneo_Mx )
   END_RUNG wire#w10
   RUNG wire#w10
      I_Contact( #pHsMx_MQ1 )
   END_RUNG wire#w11
   RUNG wire#w10
      I_Contact( #Mx_ET50 )
      Contact( #Simultaneo_Mx )
   END_RUNG wire#w11
   // the same network as SCL:
   #PosMQ_OK := (#Selec_Entrada AND (#TP1_Arriba OR #Simultaneo_Mx) AND #MQ1_Abajo AND #MQ2_Abajo) OR (#Selec_Salida_MQ1_2 AND #SaliendoCarga AND (#TP1_Abajo OR (NOT #Mx_ET50 AND #Simultaneo_Mx)) AND #MQ1_Abajo AND #MQ2_Abajo) OR (#Selec_Salida_MQ1 AND #SaliendoCarga AND (#TP1_Abajo OR (NOT #Mx_ET50 AND #Simultaneo_Mx)) AND #MQ1_Abajo AND (#MQ2_Arriba OR NOT #pHsMx_MQ2 OR (NOT #Mx_ET50 AND #Simultaneo_Mx))) OR (#Selec_Salida_MQ2 AND #SaliendoCarga AND (#TP1_Abajo OR (NOT #Mx_ET50 AND #Simultaneo_Mx)) AND (#MQ1_Arriba OR NOT #pHsMx_MQ1 OR (NOT #Mx_ET50 AND #Simultaneo_Mx)) AND #MQ2_Abajo);
END_REGION

REGION Network 17: VARIABLES AUXILIARES - Fin de Entrada - FTF_MAnt_Mx
   RUNG wire#powerrail
      Contact( #Mx_ET11 )
      Contact( #ProtocoloIniciado )
      Coil( #STAT_FTF_MAnt_Mx )
      Coil( #FTF_MAnt_Mx )
   END_RUNG
   // the same network as SCL:
   #STAT_FTF_MAnt_Mx := #Mx_ET11 AND #ProtocoloIniciado;
   #FTF_MAnt_Mx := #STAT_FTF_MAnt_Mx;
END_REGION

REGION Network 18: ESTADO DE LA MESA - DESCARGA ACTIVA
   RUNG wire#powerrail
      Contact( #OrdSal_MQ1 )
      Contact( #Selec_Salida_MQ1 )
      wire#w1
      Contact( #Mx_ET02 )
      Contact( #AVTF_Mx_MSig )
      Contact( #PTF_Mx_MSig )
      Contact( #MSig_CargaAct )
      S_SR(operand := #EstadoVI.Descarga_Act, r1 := wire#w3)
   END_RUNG
   RUNG wire#powerrail
      Contact( #OrdSal_MQ1 )
      Contact( #Selec_Salida_MQ2 )
   END_RUNG wire#w1
   RUNG wire#powerrail
      Contact( #OrdSal_MQ2 )
      Contact( #Selec_Salida_MQ2 )
   END_RUNG wire#w1
   RUNG wire#powerrail
      Contact( #OrdSal_MQ1_2 )
      Contact( #Selec_Salida_MQ1_2 )
   END_RUNG wire#w1
   RUNG wire#powerrail
      Contact( #Mx_ET51 )
      Contact( #Mx_ET151 )
      wire#w2
      Contact( #FTF_Mx_MSig )
   END_RUNG wire#w3
   RUNG wire#w2
      I_Contact( #MSig_CargaAct )
   END_RUNG wire#w3
   RUNG wire#powerrail
      Contact( #Mx_ET00 )
   END_RUNG wire#w3
   // the same network as SCL:
   IF ((#OrdSal_MQ1 AND #Selec_Salida_MQ1) OR (#OrdSal_MQ1 AND #Selec_Salida_MQ2) OR (#OrdSal_MQ2 AND #Selec_Salida_MQ2) OR (#OrdSal_MQ1_2 AND #Selec_Salida_MQ1_2)) AND #Mx_ET02 AND #AVTF_Mx_MSig AND #PTF_Mx_MSig AND #MSig_CargaAct THEN
       #EstadoVI.Descarga_Act := TRUE;   // SR flip-flop
   END_IF;
   IF (#Mx_ET51 AND #Mx_ET151 AND (#FTF_Mx_MSig OR NOT #MSig_CargaAct)) OR #Mx_ET00 THEN
       #EstadoVI.Descarga_Act := FALSE;
   END_IF;
END_REGION

REGION Network 19: ET151 - CONTROL DE SALIDA DE CARGA - PROTOCOLO
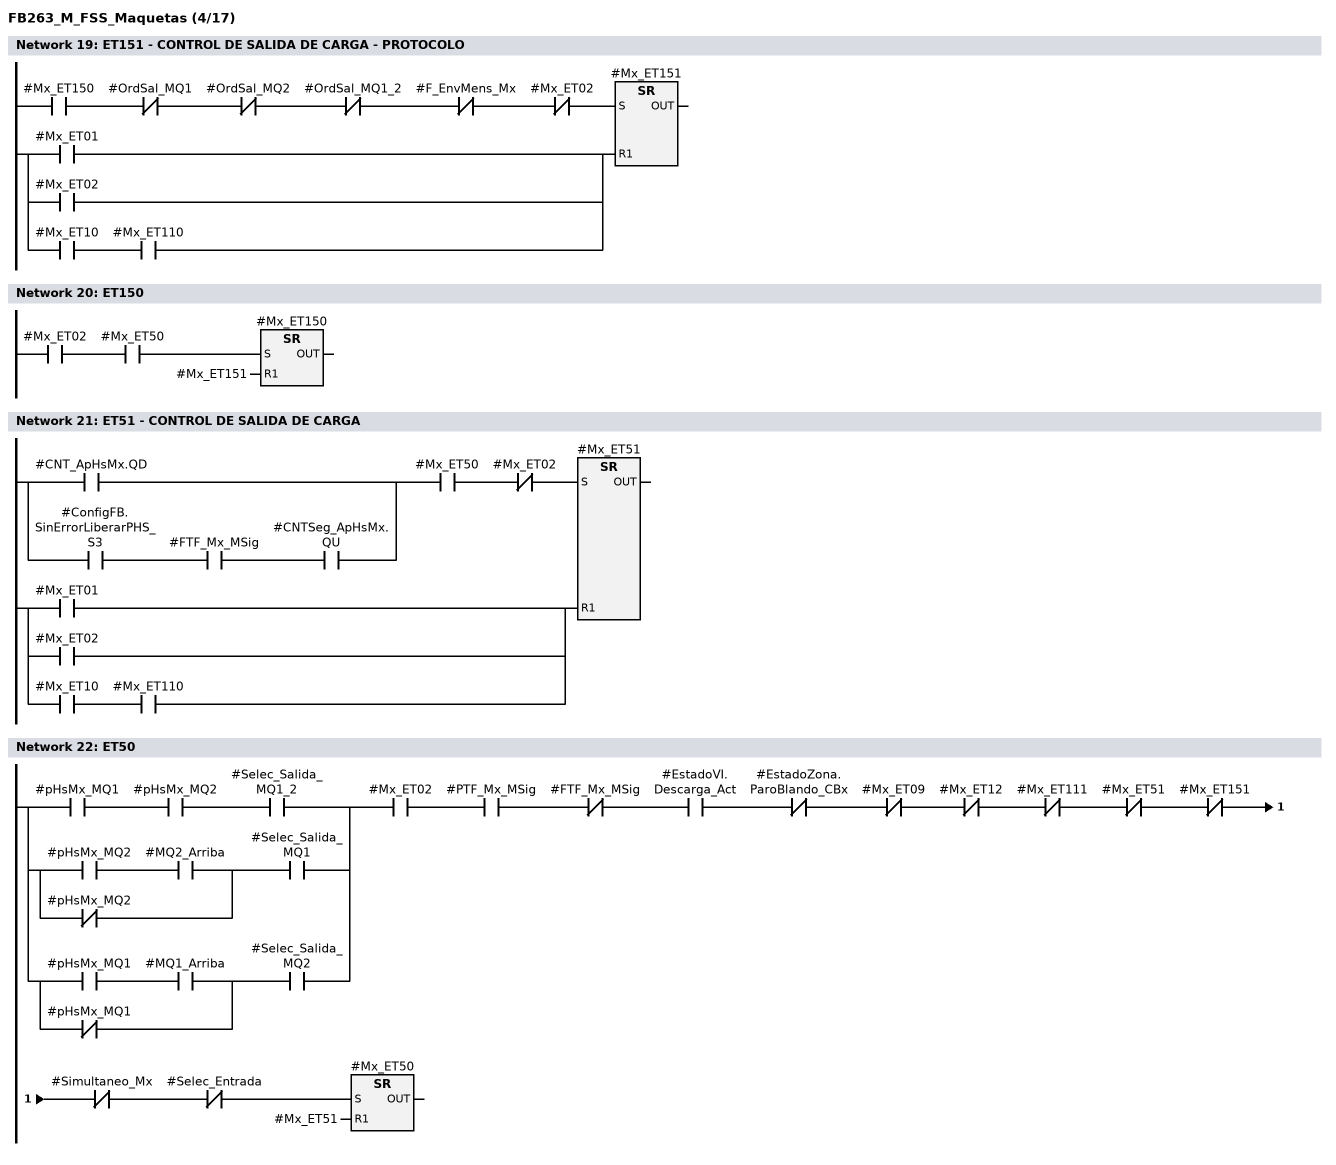
   RUNG wire#powerrail
      Contact( #Mx_ET150 )
      I_Contact( #OrdSal_MQ1 )
      I_Contact( #OrdSal_MQ2 )
      I_Contact( #OrdSal_MQ1_2 )
      I_Contact( #F_EnvMens_Mx )
      I_Contact( #Mx_ET02 )
      S_SR(operand := #Mx_ET151, r1 := wire#w1)
   END_RUNG
   RUNG wire#powerrail
      Contact( #Mx_ET01 )
   END_RUNG wire#w1
   RUNG wire#powerrail
      Contact( #Mx_ET02 )
   END_RUNG wire#w1
   RUNG wire#powerrail
      Contact( #Mx_ET10 )
      Contact( #Mx_ET110 )
   END_RUNG wire#w1
   // the same network as SCL:
   IF #Mx_ET150 AND NOT #OrdSal_MQ1 AND NOT #OrdSal_MQ2 AND NOT #OrdSal_MQ1_2 AND NOT #F_EnvMens_Mx AND NOT #Mx_ET02 THEN
       #Mx_ET151 := TRUE;   // SR flip-flop
   END_IF;
   IF #Mx_ET01 OR #Mx_ET02 OR (#Mx_ET10 AND #Mx_ET110) THEN #Mx_ET151 := FALSE; END_IF;
END_REGION

REGION Network 20: ET150
   RUNG wire#powerrail
      Contact( #Mx_ET02 )
      Contact( #Mx_ET50 )
      S_SR(operand := #Mx_ET150, r1 := #Mx_ET151)
   END_RUNG
   // the same network as SCL:
   IF #Mx_ET02 AND #Mx_ET50 THEN
       #Mx_ET150 := TRUE;   // SR flip-flop
   END_IF;
   IF #Mx_ET151 THEN #Mx_ET150 := FALSE; END_IF;
END_REGION

REGION Network 21: ET51 - CONTROL DE SALIDA DE CARGA
   RUNG wire#powerrail
      Contact( #CNT_ApHsMx.QD )
      wire#w1
      Contact( #Mx_ET50 )
      I_Contact( #Mx_ET02 )
      S_SR(operand := #Mx_ET51, r1 := wire#w2)
   END_RUNG
   RUNG wire#powerrail
      Contact( #ConfigFB.SinErrorLiberarPHS_S3 )
      Contact( #FTF_Mx_MSig )
      Contact( #CNTSeg_ApHsMx.QU )
   END_RUNG wire#w1
   RUNG wire#powerrail
      Contact( #Mx_ET01 )
   END_RUNG wire#w2
   RUNG wire#powerrail
      Contact( #Mx_ET02 )
   END_RUNG wire#w2
   RUNG wire#powerrail
      Contact( #Mx_ET10 )
      Contact( #Mx_ET110 )
   END_RUNG wire#w2
   // the same network as SCL:
   IF (#CNT_ApHsMx.QD OR (#ConfigFB.SinErrorLiberarPHS_S3 AND #FTF_Mx_MSig AND #CNTSeg_ApHsMx.QU)) AND #Mx_ET50 AND NOT #Mx_ET02 THEN
       #Mx_ET51 := TRUE;   // SR flip-flop
   END_IF;
   IF #Mx_ET01 OR #Mx_ET02 OR (#Mx_ET10 AND #Mx_ET110) THEN #Mx_ET51 := FALSE; END_IF;
END_REGION

REGION Network 22: ET50
   RUNG wire#powerrail
      Contact( #pHsMx_MQ1 )
      Contact( #pHsMx_MQ2 )
      Contact( #Selec_Salida_MQ1_2 )
      wire#w1
      Contact( #Mx_ET02 )
      Contact( #PTF_Mx_MSig )
      I_Contact( #FTF_Mx_MSig )
      Contact( #EstadoVI.Descarga_Act )
      I_Contact( #EstadoZona.ParoBlando_CBx )
      I_Contact( #Mx_ET09 )
      I_Contact( #Mx_ET12 )
      I_Contact( #Mx_ET111 )
      I_Contact( #Mx_ET51 )
      I_Contact( #Mx_ET151 )
      I_Contact( #Simultaneo_Mx )
      I_Contact( #Selec_Entrada )
      S_SR(operand := #Mx_ET50, r1 := #Mx_ET51)
   END_RUNG
   RUNG wire#powerrail
      Contact( #pHsMx_MQ2 )
      Contact( #MQ2_Arriba )
      wire#w2
      Contact( #Selec_Salida_MQ1 )
   END_RUNG wire#w1
   RUNG wire#powerrail
      I_Contact( #pHsMx_MQ2 )
   END_RUNG wire#w2
   RUNG wire#powerrail
      Contact( #pHsMx_MQ1 )
      Contact( #MQ1_Arriba )
      wire#w3
      Contact( #Selec_Salida_MQ2 )
   END_RUNG wire#w1
   RUNG wire#powerrail
      I_Contact( #pHsMx_MQ1 )
   END_RUNG wire#w3
   // the same network as SCL:
   IF ((#pHsMx_MQ1 AND #pHsMx_MQ2 AND #Selec_Salida_MQ1_2) OR (((#pHsMx_MQ2 AND #MQ2_Arriba) OR NOT #pHsMx_MQ2) AND #Selec_Salida_MQ1) OR (((#pHsMx_MQ1 AND #MQ1_Arriba) OR NOT #pHsMx_MQ1) AND #Selec_Salida_MQ2)) AND #Mx_ET02 AND #PTF_Mx_MSig AND NOT #FTF_Mx_MSig AND #EstadoVI.Descarga_Act AND NOT #EstadoZona.ParoBlando_CBx AND NOT #Mx_ET09 AND NOT #Mx_ET12 AND NOT #Mx_ET111 AND NOT #Mx_ET51 AND NOT #Mx_ET151 AND NOT #Simultaneo_Mx AND NOT #Selec_Entrada THEN
       #Mx_ET50 := TRUE;   // SR flip-flop
   END_IF;
   IF #Mx_ET51 THEN #Mx_ET50 := FALSE; END_IF;
END_REGION

REGION Network 23: ET02 - ESTADO DE REPOSO CARGADA
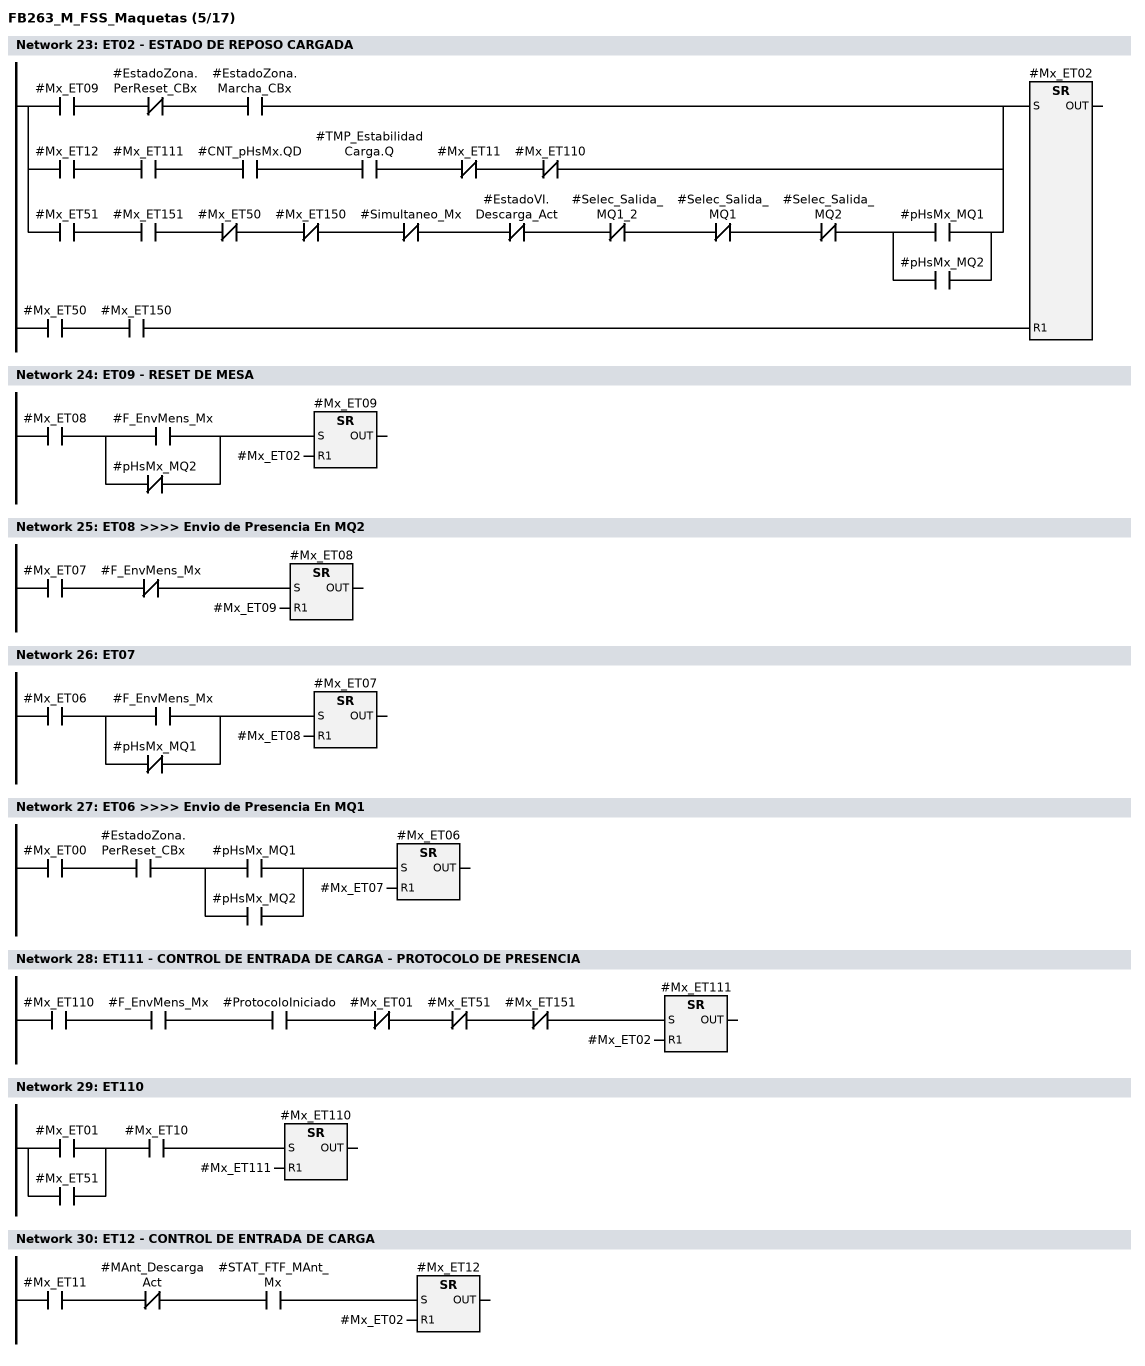
   RUNG wire#powerrail
      Contact( #Mx_ET09 )
      I_Contact( #EstadoZona.PerReset_CBx )
      Contact( #EstadoZona.Marcha_CBx )
      wire#w1
      S_SR(operand := #Mx_ET02, r1 := wire#w3)
   END_RUNG
   RUNG wire#powerrail
      Contact( #Mx_ET12 )
      Contact( #Mx_ET111 )
      Contact( #CNT_pHsMx.QD )
      Contact( #TMP_EstabilidadCarga.Q )
      I_Contact( #Mx_ET11 )
      I_Contact( #Mx_ET110 )
   END_RUNG wire#w1
   RUNG wire#powerrail
      Contact( #Mx_ET51 )
      Contact( #Mx_ET151 )
      I_Contact( #Mx_ET50 )
      I_Contact( #Mx_ET150 )
      I_Contact( #Simultaneo_Mx )
      I_Contact( #EstadoVI.Descarga_Act )
      I_Contact( #Selec_Salida_MQ1_2 )
      I_Contact( #Selec_Salida_MQ1 )
      I_Contact( #Selec_Salida_MQ2 )
      wire#w2
      Contact( #pHsMx_MQ1 )
   END_RUNG wire#w1
   RUNG wire#w2
      Contact( #pHsMx_MQ2 )
   END_RUNG wire#w1
   RUNG wire#powerrail
      Contact( #Mx_ET50 )
      Contact( #Mx_ET150 )
   END_RUNG wire#w3
   // the same network as SCL:
   IF (#Mx_ET09 AND NOT #EstadoZona.PerReset_CBx AND #EstadoZona.Marcha_CBx) OR (#Mx_ET12 AND #Mx_ET111 AND #CNT_pHsMx.QD AND #TMP_EstabilidadCarga.Q AND NOT #Mx_ET11 AND NOT #Mx_ET110) OR (#Mx_ET51 AND #Mx_ET151 AND NOT #Mx_ET50 AND NOT #Mx_ET150 AND NOT #Simultaneo_Mx AND NOT #EstadoVI.Descarga_Act AND NOT #Selec_Salida_MQ1_2 AND NOT #Selec_Salida_MQ1 AND NOT #Selec_Salida_MQ2 AND (#pHsMx_MQ1 OR #pHsMx_MQ2)) THEN
       #Mx_ET02 := TRUE;   // SR flip-flop
   END_IF;
   IF #Mx_ET50 AND #Mx_ET150 THEN #Mx_ET02 := FALSE; END_IF;
END_REGION

REGION Network 24: ET09 - RESET DE MESA
   RUNG wire#powerrail
      Contact( #Mx_ET08 )
      wire#w1
      Contact( #F_EnvMens_Mx )
      wire#w2
      S_SR(operand := #Mx_ET09, r1 := #Mx_ET02)
   END_RUNG
   RUNG wire#w1
      I_Contact( #pHsMx_MQ2 )
   END_RUNG wire#w2
   // the same network as SCL:
   IF #Mx_ET08 AND (#F_EnvMens_Mx OR NOT #pHsMx_MQ2) THEN
       #Mx_ET09 := TRUE;   // SR flip-flop
   END_IF;
   IF #Mx_ET02 THEN #Mx_ET09 := FALSE; END_IF;
END_REGION

REGION Network 25: ET08 >>>> Envio de Presencia En MQ2
   RUNG wire#powerrail
      Contact( #Mx_ET07 )
      I_Contact( #F_EnvMens_Mx )
      S_SR(operand := #Mx_ET08, r1 := #Mx_ET09)
   END_RUNG
   // the same network as SCL:
   IF #Mx_ET07 AND NOT #F_EnvMens_Mx THEN
       #Mx_ET08 := TRUE;   // SR flip-flop
   END_IF;
   IF #Mx_ET09 THEN #Mx_ET08 := FALSE; END_IF;
END_REGION

REGION Network 26: ET07
   RUNG wire#powerrail
      Contact( #Mx_ET06 )
      wire#w1
      Contact( #F_EnvMens_Mx )
      wire#w2
      S_SR(operand := #Mx_ET07, r1 := #Mx_ET08)
   END_RUNG
   RUNG wire#w1
      I_Contact( #pHsMx_MQ1 )
   END_RUNG wire#w2
   // the same network as SCL:
   IF #Mx_ET06 AND (#F_EnvMens_Mx OR NOT #pHsMx_MQ1) THEN
       #Mx_ET07 := TRUE;   // SR flip-flop
   END_IF;
   IF #Mx_ET08 THEN #Mx_ET07 := FALSE; END_IF;
END_REGION

REGION Network 27: ET06 >>>> Envio de Presencia En MQ1
   RUNG wire#powerrail
      Contact( #Mx_ET00 )
      Contact( #EstadoZona.PerReset_CBx )
      wire#w1
      Contact( #pHsMx_MQ1 )
      wire#w2
      S_SR(operand := #Mx_ET06, r1 := #Mx_ET07)
   END_RUNG
   RUNG wire#w1
      Contact( #pHsMx_MQ2 )
   END_RUNG wire#w2
   // the same network as SCL:
   IF #Mx_ET00 AND #EstadoZona.PerReset_CBx AND (#pHsMx_MQ1 OR #pHsMx_MQ2) THEN
       #Mx_ET06 := TRUE;   // SR flip-flop
   END_IF;
   IF #Mx_ET07 THEN #Mx_ET06 := FALSE; END_IF;
END_REGION

REGION Network 28: ET111 - CONTROL DE ENTRADA DE CARGA - PROTOCOLO DE PRESENCIA
   RUNG wire#powerrail
      Contact( #Mx_ET110 )
      Contact( #F_EnvMens_Mx )
      Contact( #ProtocoloIniciado )
      I_Contact( #Mx_ET01 )
      I_Contact( #Mx_ET51 )
      I_Contact( #Mx_ET151 )
      S_SR(operand := #Mx_ET111, r1 := #Mx_ET02)
   END_RUNG
   // the same network as SCL:
   IF #Mx_ET110 AND #F_EnvMens_Mx AND #ProtocoloIniciado AND NOT #Mx_ET01 AND NOT #Mx_ET51 AND NOT #Mx_ET151 THEN
       #Mx_ET111 := TRUE;   // SR flip-flop
   END_IF;
   IF #Mx_ET02 THEN #Mx_ET111 := FALSE; END_IF;
END_REGION

REGION Network 29: ET110
   RUNG wire#powerrail
      Contact( #Mx_ET01 )
      wire#w1
      Contact( #Mx_ET10 )
      S_SR(operand := #Mx_ET110, r1 := #Mx_ET111)
   END_RUNG
   RUNG wire#powerrail
      Contact( #Mx_ET51 )
   END_RUNG wire#w1
   // the same network as SCL:
   IF (#Mx_ET01 OR #Mx_ET51) AND #Mx_ET10 THEN
       #Mx_ET110 := TRUE;   // SR flip-flop
   END_IF;
   IF #Mx_ET111 THEN #Mx_ET110 := FALSE; END_IF;
END_REGION

REGION Network 30: ET12 - CONTROL DE ENTRADA DE CARGA
   RUNG wire#powerrail
      Contact( #Mx_ET11 )
      I_Contact( #MAnt_DescargaAct )
      Contact( #STAT_FTF_MAnt_Mx )
      S_SR(operand := #Mx_ET12, r1 := #Mx_ET02)
   END_RUNG
   // the same network as SCL:
   IF #Mx_ET11 AND NOT #MAnt_DescargaAct AND #STAT_FTF_MAnt_Mx THEN
       #Mx_ET12 := TRUE;   // SR flip-flop
   END_IF;
   IF #Mx_ET02 THEN #Mx_ET12 := FALSE; END_IF;
END_REGION

REGION Network 31: ET11
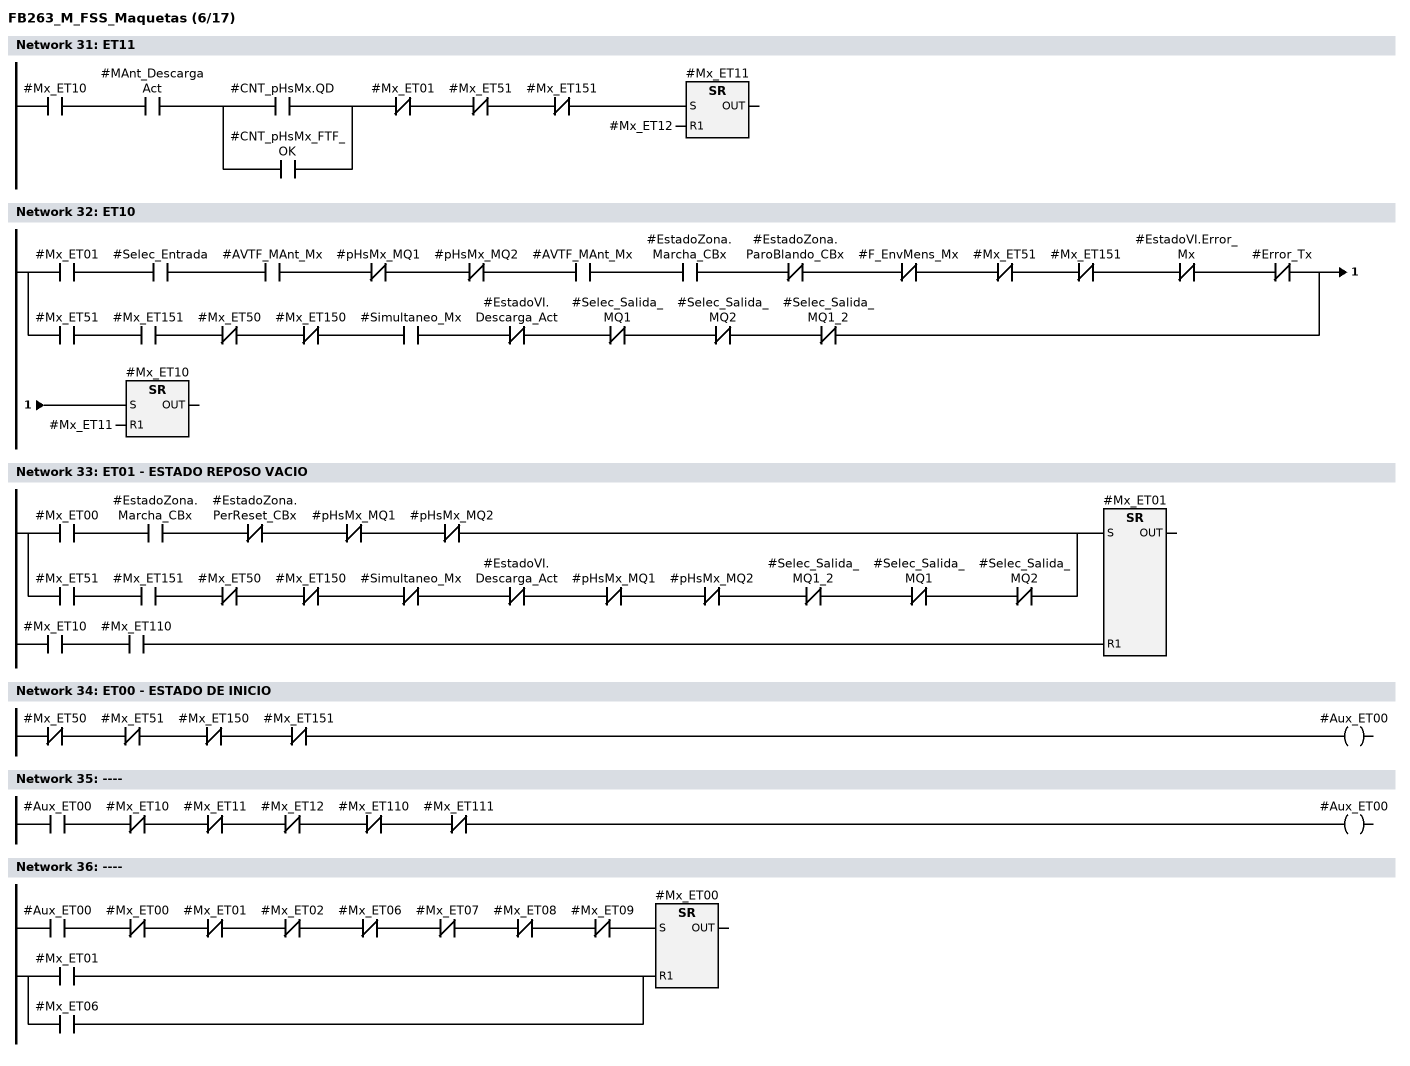
   RUNG wire#powerrail
      Contact( #Mx_ET10 )
      Contact( #MAnt_DescargaAct )
      wire#w1
      Contact( #CNT_pHsMx.QD )
      wire#w2
      I_Contact( #Mx_ET01 )
      I_Contact( #Mx_ET51 )
      I_Contact( #Mx_ET151 )
      S_SR(operand := #Mx_ET11, r1 := #Mx_ET12)
   END_RUNG
   RUNG wire#w1
      Contact( #CNT_pHsMx_FTF_OK )
   END_RUNG wire#w2
   // the same network as SCL:
   IF #Mx_ET10 AND #MAnt_DescargaAct AND (#CNT_pHsMx.QD OR #CNT_pHsMx_FTF_OK) AND NOT #Mx_ET01 AND NOT #Mx_ET51 AND NOT #Mx_ET151 THEN
       #Mx_ET11 := TRUE;   // SR flip-flop
   END_IF;
   IF #Mx_ET12 THEN #Mx_ET11 := FALSE; END_IF;
END_REGION

REGION Network 32: ET10
   RUNG wire#powerrail
      Contact( #Mx_ET01 )
      Contact( #Selec_Entrada )
      Contact( #AVTF_MAnt_Mx )
      I_Contact( #pHsMx_MQ1 )
      I_Contact( #pHsMx_MQ2 )
      Contact( #AVTF_MAnt_Mx )
      Contact( #EstadoZona.Marcha_CBx )
      I_Contact( #EstadoZona.ParoBlando_CBx )
      I_Contact( #F_EnvMens_Mx )
      I_Contact( #Mx_ET51 )
      I_Contact( #Mx_ET151 )
      I_Contact( #EstadoVI.Error_Mx )
      I_Contact( #Error_Tx )
      wire#w1
      S_SR(operand := #Mx_ET10, r1 := #Mx_ET11)
   END_RUNG
   RUNG wire#powerrail
      Contact( #Mx_ET51 )
      Contact( #Mx_ET151 )
      I_Contact( #Mx_ET50 )
      I_Contact( #Mx_ET150 )
      Contact( #Simultaneo_Mx )
      I_Contact( #EstadoVI.Descarga_Act )
      I_Contact( #Selec_Salida_MQ1 )
      I_Contact( #Selec_Salida_MQ2 )
      I_Contact( #Selec_Salida_MQ1_2 )
   END_RUNG wire#w1
   // the same network as SCL:
   IF (#Mx_ET01 AND #Selec_Entrada AND #AVTF_MAnt_Mx AND NOT #pHsMx_MQ1 AND NOT #pHsMx_MQ2 AND #AVTF_MAnt_Mx AND #EstadoZona.Marcha_CBx AND NOT #EstadoZona.ParoBlando_CBx AND NOT #F_EnvMens_Mx AND NOT #Mx_ET51 AND NOT #Mx_ET151 AND NOT #EstadoVI.Error_Mx AND NOT #Error_Tx) OR (#Mx_ET51 AND #Mx_ET151 AND NOT #Mx_ET50 AND NOT #Mx_ET150 AND #Simultaneo_Mx AND NOT #EstadoVI.Descarga_Act AND NOT #Selec_Salida_MQ1 AND NOT #Selec_Salida_MQ2 AND NOT #Selec_Salida_MQ1_2) THEN
       #Mx_ET10 := TRUE;   // SR flip-flop
   END_IF;
   IF #Mx_ET11 THEN #Mx_ET10 := FALSE; END_IF;
END_REGION

